(* CODESYS project T620X_HMI_CR1076_SP19p4.project
   Author: AW
   Version: 3.0.0.7
   Description: T620X/Radial
   Title: MAIN_HMI
   Company: MTech
   CompileDateTime: 09:01:42,04-04-2025

Project tree, tasks and I/O mapping:
  Device : ecomatDisplay_64bit, ifm electronic, order no. 
      , version 3.5.16.55
    application Application
      libraries: CmpBitmapPool, * (System); MGSE_CAS_Common, 0.0.0.1 (MGSE); ifm_ecomatDisplay43inch_Cnt, 1.0.0.0 (ifm electronic); MemoryUtils, * (3S - Smart Software Solutions GmbH); SysSocket, * (System); Util, 3.5.19.0 (System); VisuDialogs, * (System); SysTimeRtc, * (System); ifmIOcommon, 2.4.0.0 (ifm electronic); ifmOutGroup, 2.1.3.0 (ifm electronic); ifmDevice_ecomatDisplay43inch, * (ifm electronic); SysProcess Implementation, * (System); CAA Memory, * (CAA Technical Workgroup); SysMem, * (System); StringUtils, 3.5.18.0 (System); MGSE_CAS_Common, 0.0.0.1 (MGSE); SysTarget, * (System); MGSE_CAS_Common, 0.0.0.1 (MGSE); UDP, * (3S - Smart Software Solutions GmbH); MGSE_CAS_Common, 0.0.0.1 (MGSE); CAA Net Base Services, * (CAA Technical Workgroup); SysDir, * (System); SysFile, * (System); MGSE_CAS_Common, 0.0.0.1 (MGSE); CmpIecTask, * (System); SLL Common, 0.0.0.1 (SLL); SLL_IFM_CRXXXX, 0.0.0.1 (SLL); SLL_IFM_Version, 0.0.0.2 (SLL); MGSE_CAS_Common, 0.0.0.1 (MGSE); PIL Master Library, 1.0.0 (Powerhouse IRL Ltd); SLL_IFM_IO, 0.0.1.0 (SLL); VisuDialogs Template, 4.3.0.1 (Examples)
      task MainTask (cyclic, interval 5 ms, priority 3, watchdog T#500MS x 1) calls HMI_KEYPAD, HMI_IO, PLC_PRG_MAIN, Nav, SECURITY_COM
      task AlarmManagerTask (cyclic, interval 50 ms, priority 31) calls Alarms_Task
      task VISU_TASK (cyclic, interval 50 ms, priority 15) calls Viz_Common, VisuElems.Visu_Prg
      task UDP_COMS_TX (cyclic, interval 10 ms, priority 1, watchdog T#500MS x 1) calls UDP_COMS_TX
      task UDP_COMS_RX (cyclic, interval 10 ms, priority 1, watchdog T#500MS x 1) calls UDP_COMS_RX
      App_Common/
        Alarms/
          program Alarms_Monitor [FBD]
          program Alarms_Task [FBD]
        System/
          program PLC_SYSTEM [FBD]: LoggerFilename, HeaderTimeUpdate
          program PLC_Setup_Info [FBD]
          program PLC_GET_SET_IP_ADDRESS [FBD]
          program SECURITY_COM [FBD]
          program PLC_LOGGING [FBD]
          program PLC_COMMON [FBD]: VersionsUpdate
        UDP/
          program UDP_COMS_RX [FBD]
          program UDP_COMS_TX [FBD]
        Vizualisations/
          Manager/
            image pool ImagePool
            image pool ifmImagePool
            text list TL_eKeyMapCodes
          DIAG_IO/
            visualisation Visualization_DIAG_IO_Op_G0
            visualisation Visualization_DIAG_IO_Ip_G1
            visualisation Visualization_DIAG_IO_Ip_G2
            visualisation Visualization_DIAG_IO_Op_G1
            visualisation Visualization_DIAG_IO_Op_G2
            visualisation Visualization_DIAG_IO_Ip_G0
            visualisation Visualization_DIAG_IO_AUX
            CR0403/
              visualisation Output_IFM_PLC_CR0403
              visualisation Visualization_CR0403_Op
              function block CR0403_Output_Display [ST]: Init
              function block OpCom_CR0403 [FBD]: uValue, Init
              data type CR0403_OUTPUTS_STATES
          Viz_Structures/
            data type Viz_Footer_Struct
            data type Viz_Misc_Status_Struct
            data type Viz_Sections
            data type Viz_Options_Struct
          Main/
            visualisation Visualization_Settings_Main
            visualisation Visualization_Alarms_Main
            visualisation Visualization_PLC_Versions
            Layout/
              visualisation Visualization_Footer
              visualisation Visualization_Keypad_PC_SIM
              visualisation Visualization_Template
              visualisation Visualization_Net_Background
              Simulation/
                visualisation Visualization_SIM_IO
                visualisation Visualization_SIM_IO_AUX
              visualisation Visualization_Main_Status_Common
              visualisation Visualization_Main_Status_Radial
              visualisation Visualization_Main_Status_Standard
            visualisation Visualization_Net_Status_Adv
            visualisation Visualization_Net_Status
            visualisation Visualization_Settings_Misc
            visualisation Visualization_PLC_Status
            visualisation Visualization_Settings_RTC
            visualisation Visualization_Settings_IO_Log
            visualisation Visualization_Settings_1
            visualisation Visualization_Main_1
            visualisation Visualization_Engine_1
            visualisation Visualization_Engine_2
            visualisation Visualization_Settings_2
            visualisation Visualization_Settings_4
            visualisation Visualization_Settings_3
            visualisation Visualization_Engine_3
        Nav/
          program Nav [FBD]: CLEAR_RET_STACK, HOME_RETURN, GOTO_PAGE, PUSH_RET_STACK, POP_RET_STACK
          data type TX_TO_MAIN_HMI_STRUCT
          Page Control/
            function block MoveArrow_1 [ST]
            function block MoveArrow_2 [ST]
            program Page_Ctrl [FBD]
            function block RotatingArrow [ST]
            program LED_Ctrl [ST]
            program AutoManSelButtons [FBD]
            function block RectIcon [FBD]
            function block PWM_Op_Status_FB [FBD]
            function block MoveArrow_Angle [ST]
            function block LED_Control_FB [ST]
        Machine/
          program Safety_Common [FBD]
          program SIREN_BEACONS [FBD]
          program APP_WARNINGS_ERRORS [ST]
        GVLS/
          Net UDP RX TX/
            declarations NVL_IO_CHASSIS
            global variables NVL_Outputs_States_Chassis
          global variables GVL_Versions
          global variables GVL_System
          global variables Machine_IO
          Viz/
            global variables GVL_Viz
            global variables NVL_Viz
          data type NV_Sys_Settings_Struct
          global variables GVL_Persistant_Defaults
          global variables GVL_Persistant
          global variables GVL_Machine
          data type T620X_SETTINGS
          global variables GVL_Engine
          global variables GVL_CAN_TX_AUX
          global variables GVL_J1939
          data type T620X_Running_Varaibles
        VIZ/
          program Viz_Common [FBD]
          program Viz_Footer [FBD]
          program Viz_Header [FBD]
      LIBS/
        IO Diagnostics/
          IO Page Templates/
            UDP/
              visualisation PLC_UDP_Info
            PLC_Status/
              visualisation PLC_Status_Info
            PLC_Version_Info/
              visualisation PLC_Version_Info
            CR0709/
              visualisation Visualization_CR0709_Op_G1
              visualisation Visualization_CR0709_Ip_G2
              visualisation Visualization_CR0709_Op_G0
              visualisation Visualization_CR0709_Op_G2
              visualisation Visualization_CR0709_Ip_G0
              visualisation Visualization_CR0709_Ip_G1
          function block CRXXXX_Input_Display [ST]: Init
          data type HMI_PLC_CR721S_IO
          data type HMI_PLC_CR0709_IO
          IO Page Objects/
            visualisation Output_Force
            visualisation Output_IFM_PLC_CRXXXX_TITLE
            visualisation Output_IFM_PLC_CRXXXX
            visualisation Input_IFM_PLC_CRXXXX
            visualisation Input_IFM_PLC_CRXXXX_TITLE
            visualisation Output_Group_IFM_PLC_CRXXXX
          function block CRXXXX_Output_Display [ST]: Init
          function block Diag_Ip_Freq_Pulse_FB [FBD]
          function block CRXXXX_Output_Group_Display [ST]: Init
          data type HMI_PLC_CR0403_IO
        Alarms/
          Functions/
            function Alarm_Log_Test_PRIME [ST]
            function block SLL_AlarmBit [ST]
            function Alarm_Log_Add [ST]
            function Alarm_ID_GetText [ST]
            function Alarm_Log_Clear_ALL [ST]
            function Alarm_Log_File_Write [ST]
            function block Alarm_Logger_Line_FB [ST]
            program Alarm_Table_Main [ST]
            function Alarm_Log_Count_Errors [ST]
            function Alarm_Log_Count_Warnings [ST]
            function Alarm_Log_Clear_ALL_Inactive [ST]
            function Alarm_Log_Count_Active_Hush [ST]
            function Alarm_Log_Update [ST]
            program Alarm_Log_Count_Errors_Hush [FBD]
          Viz/
            visualisation Alarm_Logger_Title
            visualisation Alarm_Logger_Line
            visualisation Alarm_Logger_Table
          Struct/
            data type SLL_LOGGER_ITEM_GROUP
            data type SLL_LOGGER_MAIN_SRUCT
            data type SLL_LOGGER_ITEM_UDP
            data type SLL_LOGGER_ITEM_FLAGS
            data type SLL_LOGGER_ITEM
            data type SENSOR_SCALE
        UDP/
          function block UDP_Info_Viz [ST]
        function print_formated_DINT_func [FBD]
        function block Convert_mm_to_in_ft [ST]
        Logging/
          function block Log_File_Read_Lines [ST]
          global variables GVL_Logging
          function Log_File_Append [ST]
        IO Common/
          function block OpCom [FBD]: Init
          function block IO_LogCom [ST]
          function block IpCom [FBD]: Init
          text list TextList_IFM_Diag_Codes
          function block OpGrpCom [FBD]: Dig, Init
          function block NodeComFB [FBD]
          function IFM_CODE_Text_Get [ST]
        function block SIMPLE_HB_CHECK_ONLINE [FBD]
        function print_BOOL_func [FBD]
        function TextList_GetText_Default [ST]
        function Mimic_IO_GetText [ST]
        HMI/
          data type HMI_TASKS_INFO_STRUCT
          global variables GVL_KeyList_RT
          data type HMI_TASK_INFO_STRUCT
          program Nav_SetupHalo [ST]
          global variables GVL_KeyList
          program RunLinuxCommand [FBD]
          program Nav_Get_Page_Name [FBD]
          global variables GVL_KeyList_FT
          function block Nav_Pages_Group_FB [FBD]
          program LCD_Brighness_Control [FBD]
          program HMI_Task_Info [ST]
          program CR1140_RTC_Edit [FBD]: ZonesDump
          program HMI_KEYPAD [FBD]: ACT_KeyList_FT, ACT_KeyList_RT
          program CloseDlgs [ST]
          program CheckDlgsOpen [ST]
        function print_formated_REAL_func [FBD]
        function block Convert_inches_to_in_ft [ST]
        function block Override_Timed [FBD]
      Symbols
      App_CODE_GEN/
        MAIN_CODE_GEN/
          App_CODE_GEN/
            Alarms/
              program Alarms_Monitor_App [ST]
              global variables GVL_Alarms
              program Alarms_Monitor_IO [ST]
            Diag_IO/
              program HMI_IO [FBD]: Update_Outputs, Init_Input_Links, Init_Output_Links, Update_Inputs
            Machine IO/
              Funcs/
                program Machine_Link_Outputs_Init [ST]
                program Machine_Link_Outputs [ST]
                program Machine_Scale_Inputs [FBD]
                program Machine_Link_Inputs_Init [ST]
                program Machine_Link_Inputs [ST]
              Structs/
                data type T620X_Radial_Outputs
                data type T620X_Radial_Inputs
        TEXT_LIST/
          text list AlarmGroup_IO
          text list AlarmGroup_App
          text list TextList_IO_Diag
      App_PLC/
        program PLC_EngineRun [FBD]
        program PLC_Alarms [FBD]
        function block fbSmoothing [ST]
        program PLC_FanCtrl [FBD]
        program PLC_SIM_MAIN [FBD]
        global variables SIM_APP
        global variables GVL_APP
        Control/
          program PLC_Auto_Sequence [FBD]
          program PLC_ManualSequence [FBD]
          program PLC_JackLegs_SideConv [FBD]
          program PLC_Tracking [FBD]
          program PLC_RadialMode [FBD]
          program PLC_Functions [FBD]
        Set Points/
          function block SP_Count_VAR [FBD]
        CAN Comms/
          Engine Comms/
            function block CounterChecksum [ST]
            function block PLC_DM1_Condition [FBD]
            function block fb_Extract_SPN [FBD]
            function block Pack2bits [ST]
            program PLC_J1939_COMS [FBD]: SCAN
            program PLC_J1939_TX_CUSTOM [FBD]
            program PLC_J1939_RX_DM1 [FBD]
            function HMI_Time_Remain_HHMM_Secs_In [ST]
          program CAN_TX_AUX_IO [FBD]
        program PLC_PRG_MAIN [FBD]
    Communication : Communication, ifm electronic, version 3.5.16.55
      Ethernet : Ethernet, ifm electronic, version 3.5.16.55
        Ethernet_ecomatDisplay4_3 : Ethernet_ecomatDisplay4.3, ifm electronic, version 1.0.0.0
            settings: IPAddress = [192,168,82,245]; SubnetMask = [255,255,255,0]; GatewayAddress = [192,168,82,1]; MACAddress = [16#00,16#02,16#01,16#10,16#3D,16#7D]; NetworkInterfaceName = 'eth0'; NetworkInterfaceName = "eth0"; SaveCommunicationSettings = FALSE
      CAN : CAN, ifm electronic, version 3.5.16.55
        CANbus_ecomatDisplay4_3 : CANbus_ecomatDisplay4.3, ifm electronic, version 1.0.0.0
            settings: NetID = 1
          J1939_Manager : J1939_Manager, 3S - Smart Software Solutions GmbH, version 4.1.0.0
            J1939_ECU : J1939_ECU, 3S - Smart Software Solutions GmbH, version 4.1.0.0
                settings: NAME = 16#0000000000000000; Communication Watchdog Timeout Period = 16#05DC ms; Activated PGs = 23; PG Offline Data.Name = "EEC1"; PG Offline Data.Description = "Electronic Engine Controller 1"; PG Online Data.PGN = 61444; PG Online Data.Length (Bytes) = 8; PG Transmission Settings.Destination Address = 255; PG Transmission Settings.CycleTimeFactor = 1; Signal Offline Data.SPN = 899; Signal Offline Data.Name = "EngTorqueMode"; Signal Offline Data.Description = "State signal which indicates which engine torque mode is currently generating, limiting, or controlling the torque."; Signal Offline Data.Unit = ""; Signal Offline Data.Min = 0; Signal Offline Data.Max = 15; Signal Online Data.BitSize = 4; Signal Online Data.BitPosition = 0; Convert Data.Flags = 3; Convert Data.pSigValue = 0; Convert Data.Scaling = 4607182418800017408; Convert Data.Offset = 0; Signal Offline Data.SPN = 4154; Signal Offline Data.Name = "ActlEngPrcntTrqueHighResolution"; Signal Offline Data.Description = "This parameter displays an additional torque in percent of the reference engine torque."; Signal Offline Data.Unit = "%"; Signal Offline Data.Min = 0; Signal Offline Data.Max = 0.875; Signal Online Data.BitSize = 4; Signal Online Data.BitPosition = 4; Convert Data.Flags = 3; Convert Data.pSigValue = 0; Convert Data.Scaling = 4593671619917905920; Convert Data.Offset = 0; Signal Offline Data.SPN = 512; Signal Offline Data.Name = "DriversDemandEngPercentTorque"; Signal Offline Data.Description = "The requested torque output of the engine by the driver."; Signal Offline Data.Unit = "%"; Signal Offline Data.Min = -125; Signal Offline Data.Max = 125; Signal Online Data.BitSize = 8;
                  Signal Online Data.BitPosition = 8; Convert Data.Flags = 3; Convert Data.pSigValue = 0; Convert Data.Scaling = 4607182418800017408; Convert Data.Offset = 13861868546813853696; Signal Offline Data.SPN = 513; Signal Offline Data.Name = "ActualEngPercentTorque"; Signal Offline Data.Description = "The calculated output torque of the engine."; Signal Offline Data.Unit = "%"; Signal Offline Data.Min = -125; Signal Offline Data.Max = 125; Signal Online Data.BitSize = 8; Signal Online Data.BitPosition = 16; Convert Data.Flags = 3; Convert Data.pSigValue = 0; Convert Data.Scaling = 4607182418800017408; Convert Data.Offset = 13861868546813853696; Signal Offline Data.SPN = 190; Signal Offline Data.Name = "EngSpeed"; Signal Offline Data.Unit = "rpm"; Signal Offline Data.Min = 0; Signal Offline Data.Max = 8031.875; Signal Online Data.BitSize = 16; Signal Online Data.BitPosition = 24; Convert Data.Flags = 3; Convert Data.pSigValue = 0; Convert Data.Scaling = 4593671619917905920; Convert Data.Offset = 0; Signal Offline Data.SPN = 1483; Signal Offline Data.Name = "SrcAddrssOfCtrllngDvcFrEngCntrl"; Signal Offline Data.Description = "The source address of the SAE J1939 device currently controlling the engine."; Signal Offline Data.Unit = ""; Signal Offline Data.Min = 0; Signal Offline Data.Max = 255; Signal Online Data.BitSize = 8; Signal Online Data.BitPosition = 40; Convert Data.Flags = 3; Convert Data.pSigValue = 0; Convert Data.Scaling = 4607182418800017408; Convert Data.Offset = 0;
                  Signal Offline Data.SPN = 1675; Signal Offline Data.Name = "EngStarterMode"; Signal Offline Data.Description = "There are several phases in a starting action and different reasons why a start cannot take place."; Signal Offline Data.Unit = ""; Signal Offline Data.Min = 0; Signal Offline Data.Max = 15; Signal Online Data.BitSize = 4; Signal Online Data.BitPosition = 48; Convert Data.Flags = 3; Convert Data.pSigValue = 0; Convert Data.Scaling = 4607182418800017408; Convert Data.Offset = 0; Signal Offline Data.SPN = 2432; Signal Offline Data.Name = "EngDemandPercentTorque"; Signal Offline Data.Unit = "%"; Signal Offline Data.Min = -125; Signal Offline Data.Max = 125; Signal Online Data.BitSize = 8; Signal Online Data.BitPosition = 56; Convert Data.Flags = 3; Convert Data.pSigValue = 0; Convert Data.Scaling = 4607182418800017408; Convert Data.Offset = 13861868546813853696; PG Offline Data.Name = "EEC2"; PG Offline Data.Description = "Electronic Engine Controller 2"; PG Online Data.PGN = 61443; PG Online Data.Length (Bytes) = 8; PG Transmission Settings.Destination Address = 255; PG Transmission Settings.CycleTimeFactor = 1; Signal Offline Data.SPN = 558; Signal Offline Data.Name = "AccelPedal1LowIdleSwitch"; Signal Offline Data.Description = "Switch signal which indicates the state of the accelerator pedal 1 low idle switch."; Signal Offline Data.Unit = ""; Signal Offline Data.Min = 0; Signal Offline Data.Max = 3; Signal Online Data.BitSize = 2; Signal Online Data.BitPosition = 0; Convert Data.Flags = 3; Convert Data.pSigValue = 0; Convert Data.Scaling = 4607182418800017408;
                  Convert Data.Offset = 0; Signal Offline Data.SPN = 559; Signal Offline Data.Name = "AccelPedalKickdownSwitch"; Signal Offline Data.Description = "Switch signal which indicates whether the accelerator pedal kickdown switch is opened or closed."; Signal Offline Data.Unit = ""; Signal Offline Data.Min = 0; Signal Offline Data.Max = 3; Signal Online Data.BitSize = 2; Signal Online Data.BitPosition = 2; Convert Data.Flags = 3; Convert Data.pSigValue = 0; Convert Data.Scaling = 4607182418800017408; Convert Data.Offset = 0; Signal Offline Data.SPN = 1437; Signal Offline Data.Name = "RoadSpeedLimitStatus"; Signal Offline Data.Description = "Status (active or not active) of the system used to limit maximum vehicle velocity."; Signal Offline Data.Unit = ""; Signal Offline Data.Min = 0; Signal Offline Data.Max = 3; Signal Online Data.BitSize = 2; Signal Online Data.BitPosition = 4; Convert Data.Flags = 3; Convert Data.pSigValue = 0; Convert Data.Scaling = 4607182418800017408; Convert Data.Offset = 0; Signal Offline Data.SPN = 2970; Signal Offline Data.Name = "AccelPedal2LowIdleSwitch"; Signal Offline Data.Description = "Switch signal which indicates the state of the accelerator pedal 2 low idle switch."; Signal Offline Data.Unit = ""; Signal Offline Data.Min = 0; Signal Offline Data.Max = 3; Signal Online Data.BitSize = 2; Signal Online Data.BitPosition = 6; Convert Data.Flags = 3; Convert Data.pSigValue = 0; Convert Data.Scaling = 4607182418800017408; Convert Data.Offset = 0; Signal Offline Data.SPN = 91; Signal Offline Data.Name = "AccelPedalPos1"; Signal Offline Data.Description = "The ratio of actual position of the analog engine speed/torque request input device (such as an accelerator pedal or";
                  Signal Offline Data.Unit = "%"; Signal Offline Data.Min = 0; Signal Offline Data.Max = 100; Signal Online Data.BitSize = 8; Signal Online Data.BitPosition = 8; Convert Data.Flags = 3; Convert Data.pSigValue = 0; Convert Data.Scaling = 4600877379321698714; Convert Data.Offset = 0; Signal Offline Data.SPN = 92; Signal Offline Data.Name = "EngPercentLoadAtCurrentSpeed"; Signal Offline Data.Unit = "%"; Signal Offline Data.Min = 0; Signal Offline Data.Max = 250; Signal Online Data.BitSize = 8; Signal Online Data.BitPosition = 16; Convert Data.Flags = 3; Convert Data.pSigValue = 0; Convert Data.Scaling = 4607182418800017408; Convert Data.Offset = 0; Signal Offline Data.SPN = 974; Signal Offline Data.Name = "RemoteAccelPedalPos"; Signal Offline Data.Unit = "%"; Signal Offline Data.Min = 0; Signal Offline Data.Max = 100; Signal Online Data.BitSize = 8; Signal Online Data.BitPosition = 24; Convert Data.Flags = 3; Convert Data.pSigValue = 0; Convert Data.Scaling = 4600877379321698714; Convert Data.Offset = 0; Signal Offline Data.SPN = 29; Signal Offline Data.Name = "AccelPedalPos2"; Signal Offline Data.Unit = "%"; Signal Offline Data.Min = 0; Signal Offline Data.Max = 100; Signal Online Data.BitSize = 8; Signal Online Data.BitPosition = 32; Convert Data.Flags = 3; Convert Data.pSigValue = 0;
                  Convert Data.Scaling = 4600877379321698714; Convert Data.Offset = 0; Signal Offline Data.SPN = 2979; Signal Offline Data.Name = "VhclAccelerationRateLimitStatus"; Signal Offline Data.Description = "Status (active or not active) of the system used to limit maximum forward vehicle acceleration."; Signal Offline Data.Unit = ""; Signal Offline Data.Min = 0; Signal Offline Data.Max = 3; Signal Online Data.BitSize = 2; Signal Online Data.BitPosition = 40; Convert Data.Flags = 3; Convert Data.pSigValue = 0; Convert Data.Scaling = 4607182418800017408; Convert Data.Offset = 0; Signal Offline Data.SPN = 5021; Signal Offline Data.Name = "MmntryEngMaxPowerEnableFeedback"; Signal Offline Data.Description = "Momentarily requesting Engine Maximum Power Enable - feature support feedback"; Signal Offline Data.Unit = ""; Signal Offline Data.Min = 0; Signal Offline Data.Max = 3; Signal Online Data.BitSize = 2; Signal Online Data.BitPosition = 42; Convert Data.Flags = 3; Convert Data.pSigValue = 0; Convert Data.Scaling = 4607182418800017408; Convert Data.Offset = 0; Signal Offline Data.SPN = 5399; Signal Offline Data.Name = "DPFThermalManagementActive"; Signal Offline Data.Unit = ""; Signal Offline Data.Min = 0; Signal Offline Data.Max = 3; Signal Online Data.BitSize = 2; Signal Online Data.BitPosition = 44; Convert Data.Flags = 3; Convert Data.pSigValue = 0; Convert Data.Scaling = 4607182418800017408; Convert Data.Offset = 0; Signal Offline Data.SPN = 5400; Signal Offline Data.Name = "SCRThermalManagementActive"; Signal Offline Data.Description = "Indicates that the exhaust temperatures have been elevated for regeneration of the SCR aftertreatment system or in";
                  Signal Offline Data.Unit = ""; Signal Offline Data.Min = 0; Signal Offline Data.Max = 3; Signal Online Data.BitSize = 2; Signal Online Data.BitPosition = 46; Convert Data.Flags = 3; Convert Data.pSigValue = 0; Convert Data.Scaling = 4607182418800017408; Convert Data.Offset = 0; Signal Offline Data.SPN = 3357; Signal Offline Data.Name = "ActlMxAvailableEngPercentTorque"; Signal Offline Data.Description = "This is the maximum amount of torque that the engine can immediately deliver as a percentage of the reference engine"; Signal Offline Data.Unit = "%"; Signal Offline Data.Min = 0; Signal Offline Data.Max = 100; Signal Online Data.BitSize = 8; Signal Online Data.BitPosition = 48; Convert Data.Flags = 3; Convert Data.pSigValue = 0; Convert Data.Scaling = 4600877379321698714; Convert Data.Offset = 0; Signal Offline Data.SPN = 5398; Signal Offline Data.Name = "EstPumpingPercentTorque"; Signal Offline Data.Description = "The calculated torque that indicates the estimated amount of torque loss due to the engine air handling system."; Signal Offline Data.Unit = "%"; Signal Offline Data.Min = -125; Signal Offline Data.Max = 125; Signal Online Data.BitSize = 8; Signal Online Data.BitPosition = 56; Convert Data.Flags = 3; Convert Data.pSigValue = 0; Convert Data.Scaling = 4607182418800017408; Convert Data.Offset = 13861868546813853696; PG Offline Data.Name = "EEC3"; PG Offline Data.Description = "Electronic Engine Controller 3"; PG Online Data.PGN = 65247; PG Online Data.Length (Bytes) = 8; PG Transmission Settings.Destination Address = 255; PG Transmission Settings.CycleTimeFactor = 1; Signal Offline Data.SPN = 514;
                  Signal Offline Data.Name = "NominalFrictionPercentTorque"; Signal Offline Data.Unit = "%"; Signal Offline Data.Min = -125; Signal Offline Data.Max = 125; Signal Online Data.BitSize = 8; Signal Online Data.BitPosition = 0; Convert Data.Flags = 3; Convert Data.pSigValue = 0; Convert Data.Scaling = 4607182418800017408; Convert Data.Offset = 13861868546813853696; Signal Offline Data.SPN = 515; Signal Offline Data.Name = "EngsDesiredOperatingSpeed"; Signal Offline Data.Description = "An indication by the engine of the optimal operating speed of the engine for the current existing conditions."; Signal Offline Data.Unit = "rpm"; Signal Offline Data.Min = 0; Signal Offline Data.Max = 8031.875; Signal Online Data.BitSize = 16; Signal Online Data.BitPosition = 8; Convert Data.Flags = 3; Convert Data.pSigValue = 0; Convert Data.Scaling = 4593671619917905920; Convert Data.Offset = 0; Signal Offline Data.SPN = 519; Signal Offline Data.Name = "EngsDsrdOprtngSpdAsymmtryAdjstmn"; Signal Offline Data.Unit = ""; Signal Offline Data.Min = 0; Signal Offline Data.Max = 250; Signal Online Data.BitSize = 8; Signal Online Data.BitPosition = 24; Convert Data.Flags = 3; Convert Data.pSigValue = 0; Convert Data.Scaling = 4607182418800017408; Convert Data.Offset = 0; Signal Offline Data.SPN = 2978; Signal Offline Data.Name = "EstEngPrsticLossesPercentTorque"; Signal Offline Data.Unit = "%"; Signal Offline Data.Min = -125; Signal Offline Data.Max = 125; Signal Online Data.BitSize = 8; Signal Online Data.BitPosition = 32;
                  Convert Data.Flags = 3; Convert Data.pSigValue = 0; Convert Data.Scaling = 4607182418800017408; Convert Data.Offset = 13861868546813853696; Signal Offline Data.SPN = 3236; Signal Offline Data.Name = "Aftrtratment1ExhaustGasMassFlow"; Signal Offline Data.Description = "Measured/calculated exhaust gas mass upstream of the aftertreatment system in exhaust bank 1 and 2."; Signal Offline Data.Unit = "kg/h"; Signal Offline Data.Min = 0; Signal Offline Data.Max = 12851; Signal Online Data.BitSize = 16; Signal Online Data.BitPosition = 40; Convert Data.Flags = 3; Convert Data.pSigValue = 0; Convert Data.Scaling = 4596373779694328218; Convert Data.Offset = 0; Signal Offline Data.SPN = 3237; Signal Offline Data.Name = "Aftertreatment1IntakeDewPoint"; Signal Offline Data.Unit = ""; Signal Offline Data.Min = 0; Signal Offline Data.Max = 3; Signal Online Data.BitSize = 2; Signal Online Data.BitPosition = 56; Convert Data.Flags = 3; Convert Data.pSigValue = 0; Convert Data.Scaling = 4607182418800017408; Convert Data.Offset = 0; Signal Offline Data.SPN = 3238; Signal Offline Data.Name = "Aftertreatment1ExhaustDewPoint"; Signal Offline Data.Unit = ""; Signal Offline Data.Min = 0; Signal Offline Data.Max = 3; Signal Online Data.BitSize = 2; Signal Online Data.BitPosition = 58; Convert Data.Flags = 3; Convert Data.pSigValue = 0; Convert Data.Scaling = 4607182418800017408; Convert Data.Offset = 0; Signal Offline Data.SPN = 3239; Signal Offline Data.Name = "Aftertreatment2IntakeDewPoint";
                  Signal Offline Data.Unit = ""; Signal Offline Data.Min = 0; Signal Offline Data.Max = 3; Signal Online Data.BitSize = 2; Signal Online Data.BitPosition = 60; Convert Data.Flags = 3; Convert Data.pSigValue = 0; Convert Data.Scaling = 4607182418800017408; Convert Data.Offset = 0; Signal Offline Data.SPN = 3240; Signal Offline Data.Name = "Aftertreatment2ExhaustDewPoint"; Signal Offline Data.Unit = ""; Signal Offline Data.Min = 0; Signal Offline Data.Max = 3; Signal Online Data.BitSize = 2; Signal Online Data.BitPosition = 62; Convert Data.Flags = 3; Convert Data.pSigValue = 0; Convert Data.Scaling = 4607182418800017408; Convert Data.Offset = 0; PG Offline Data.Name = "EEC5"; PG Offline Data.Description = "Electronic Engine Controller 5"; PG Online Data.PGN = 64981; PG Online Data.Length (Bytes) = 8; PG Transmission Settings.Destination Address = 255; PG Transmission Settings.CycleTimeFactor = 1; Signal Offline Data.SPN = 2789; Signal Offline Data.Name = "EngTrb1ClcltedTurbineIntakeTemp"; Signal Offline Data.Description = "Calculated value of turbine intake temperature based on engine operating conditions, such as intake manifold"; Signal Offline Data.Unit = "deg C"; Signal Offline Data.Min = -273; Signal Offline Data.Max = 1734.96875; Signal Online Data.BitSize = 16; Signal Online Data.BitPosition = 0; Convert Data.Flags = 3; Convert Data.pSigValue = 0; Convert Data.Scaling = 4584664420663164928; Convert Data.Offset = 13866882319836512256; Signal Offline Data.SPN = 2790; Signal Offline Data.Name = "EngTrb1ClcltedTurbineOutletTemp";
                  Signal Offline Data.Description = "Calculated value of turbocharger compressor outlet air temperature."; Signal Offline Data.Unit = "deg C"; Signal Offline Data.Min = -273; Signal Offline Data.Max = 1734.96875; Signal Online Data.BitSize = 16; Signal Online Data.BitPosition = 16; Convert Data.Flags = 3; Convert Data.pSigValue = 0; Convert Data.Scaling = 4584664420663164928; Convert Data.Offset = 13866882319836512256; Signal Offline Data.SPN = 2791; Signal Offline Data.Name = "EngExhstGsRcrculation1ValveCtrl"; Signal Offline Data.Description = "Desired percentage of maximum Exhaust Gas Recirculation (EGR) valve opening."; Signal Offline Data.Unit = "%"; Signal Offline Data.Min = 0; Signal Offline Data.Max = 160.6375; Signal Online Data.BitSize = 16; Signal Online Data.BitPosition = 32; Convert Data.Flags = 3; Convert Data.pSigValue = 0; Convert Data.Scaling = 4567911030049346683; Convert Data.Offset = 0; Signal Offline Data.SPN = 2792; Signal Offline Data.Name = "EngVrblGmtryTrbArCtrlShtffValve"; Signal Offline Data.Description = "Isolates vehicle brake air from the Variable Geometry Turbocharger (VGT) system when engine is not running."; Signal Offline Data.Unit = ""; Signal Offline Data.Min = 0; Signal Offline Data.Max = 3; Signal Online Data.BitSize = 2; Signal Online Data.BitPosition = 48; Convert Data.Flags = 3; Convert Data.pSigValue = 0; Convert Data.Scaling = 4607182418800017408; Convert Data.Offset = 0; Signal Offline Data.SPN = 5457; Signal Offline Data.Name = "EngVrableGeometryTurbo1CtrlMode"; Signal Offline Data.Description = "Indicates if the variable geometry turbocharger control status is either open loop or closed loop."; Signal Offline Data.Unit = ""; Signal Offline Data.Min = 0; Signal Offline Data.Max = 3;
                  Signal Online Data.BitSize = 2; Signal Online Data.BitPosition = 52; Convert Data.Flags = 3; Convert Data.pSigValue = 0; Convert Data.Scaling = 4607182418800017408; Convert Data.Offset = 0; Signal Offline Data.SPN = 2795; Signal Offline Data.Name = "EngVrblGometryTurbo1ActuatorPos"; Signal Offline Data.Description = "Sensor that measures the position of the variable geometry turbocharger actuator."; Signal Offline Data.Unit = "%"; Signal Offline Data.Min = 0; Signal Offline Data.Max = 100; Signal Online Data.BitSize = 8; Signal Online Data.BitPosition = 56; Convert Data.Flags = 3; Convert Data.pSigValue = 0; Convert Data.Scaling = 4600877379321698714; Convert Data.Offset = 0; PG Offline Data.Name = "ET1"; PG Offline Data.Description = "Engine Temperature 1"; PG Online Data.PGN = 65262; PG Online Data.Length (Bytes) = 8; PG Transmission Settings.Destination Address = 255; PG Transmission Settings.CycleTimeFactor = 1; Signal Offline Data.SPN = 110; Signal Offline Data.Name = "EngCoolantTemp"; Signal Offline Data.Description = "Temperature of liquid found in engine cooling system."; Signal Offline Data.Unit = "deg C"; Signal Offline Data.Min = -40; Signal Offline Data.Max = 210; Signal Online Data.BitSize = 8; Signal Online Data.BitPosition = 0; Convert Data.Flags = 3; Convert Data.pSigValue = 0; Convert Data.Scaling = 4607182418800017408; Convert Data.Offset = 13854198353698488320; Signal Offline Data.SPN = 174; Signal Offline Data.Name = "EngFuelTemp1"; Signal Offline Data.Description = "Temperature of fuel (or gas) passing through the first fuel control system."; Signal Offline Data.Unit = "deg C";
                  Signal Offline Data.Min = -40; Signal Offline Data.Max = 210; Signal Online Data.BitSize = 8; Signal Online Data.BitPosition = 8; Convert Data.Flags = 3; Convert Data.pSigValue = 0; Convert Data.Scaling = 4607182418800017408; Convert Data.Offset = 13854198353698488320; Signal Offline Data.SPN = 175; Signal Offline Data.Name = "EngOilTemp1"; Signal Offline Data.Description = "Temperature of the engine lubricant."; Signal Offline Data.Unit = "deg C"; Signal Offline Data.Min = -273; Signal Offline Data.Max = 1734.96875; Signal Online Data.BitSize = 16; Signal Online Data.BitPosition = 16; Convert Data.Flags = 3; Convert Data.pSigValue = 0; Convert Data.Scaling = 4584664420663164928; Convert Data.Offset = 13866882319836512256; Signal Offline Data.SPN = 176; Signal Offline Data.Name = "EngTurboOilTemp"; Signal Offline Data.Description = "Temperature of the turbocharger lubricant."; Signal Offline Data.Unit = "deg C"; Signal Offline Data.Min = -273; Signal Offline Data.Max = 1734.96875; Signal Online Data.BitSize = 16; Signal Online Data.BitPosition = 32; Convert Data.Flags = 3; Convert Data.pSigValue = 0; Convert Data.Scaling = 4584664420663164928; Convert Data.Offset = 13866882319836512256; Signal Offline Data.SPN = 52; Signal Offline Data.Name = "EngIntercoolerTemp"; Signal Offline Data.Description = "Temperature of liquid found in the intercooler located after the turbocharger."; Signal Offline Data.Unit = "deg C"; Signal Offline Data.Min = -40; Signal Offline Data.Max = 210; Signal Online Data.BitSize = 8; Signal Online Data.BitPosition = 48;
                  Convert Data.Flags = 3; Convert Data.pSigValue = 0; Convert Data.Scaling = 4607182418800017408; Convert Data.Offset = 13854198353698488320; Signal Offline Data.SPN = 1134; Signal Offline Data.Name = "EngIntercoolerThermostatOpening"; Signal Offline Data.Description = "The current position of the thermostat used to regulate the temperature of the engine intercooler."; Signal Offline Data.Unit = "%"; Signal Offline Data.Min = 0; Signal Offline Data.Max = 100; Signal Online Data.BitSize = 8; Signal Online Data.BitPosition = 56; Convert Data.Flags = 3; Convert Data.pSigValue = 0; Convert Data.Scaling = 4600877379321698714; Convert Data.Offset = 0; PG Offline Data.Name = "EFL_P1"; PG Offline Data.Description = "Engine Fluid Level/Pressure 1"; PG Online Data.PGN = 65263; PG Online Data.Length (Bytes) = 8; PG Transmission Settings.Destination Address = 255; PG Transmission Settings.CycleTimeFactor = 1; Signal Offline Data.SPN = 94; Signal Offline Data.Name = "EngFuelDeliveryPress"; Signal Offline Data.Description = "Gage pressure of fuel in system as delivered from supply pump to the injection pump."; Signal Offline Data.Unit = "kPa"; Signal Offline Data.Min = 0; Signal Offline Data.Max = 1000; Signal Online Data.BitSize = 8; Signal Online Data.BitPosition = 0; Convert Data.Flags = 3; Convert Data.pSigValue = 0; Convert Data.Scaling = 4616189618054758400; Convert Data.Offset = 0; Signal Offline Data.SPN = 22; Signal Offline Data.Name = "EngExCrankcaseBlowbyPress"; Signal Offline Data.Description = "Differential crankcase blow-by pressure as measured through a tube with a venturi."; Signal Offline Data.Unit = "kPa"; Signal Offline Data.Min = 0; Signal Offline Data.Max = 12.5;
                  Signal Online Data.BitSize = 8; Signal Online Data.BitPosition = 8; Convert Data.Flags = 3; Convert Data.pSigValue = 0; Convert Data.Scaling = 4587366580439587226; Convert Data.Offset = 0; Signal Offline Data.SPN = 98; Signal Offline Data.Name = "EngOilLevel"; Signal Offline Data.Description = "Ratio of current volume of engine sump oil to maximum required volume."; Signal Offline Data.Unit = "%"; Signal Offline Data.Min = 0; Signal Offline Data.Max = 100; Signal Online Data.BitSize = 8; Signal Online Data.BitPosition = 16; Convert Data.Flags = 3; Convert Data.pSigValue = 0; Convert Data.Scaling = 4600877379321698714; Convert Data.Offset = 0; Signal Offline Data.SPN = 100; Signal Offline Data.Name = "EngOilPress"; Signal Offline Data.Description = "Gage pressure of oil in engine lubrication system as provided by oil pump."; Signal Offline Data.Unit = "kPa"; Signal Offline Data.Min = 0; Signal Offline Data.Max = 1000; Signal Online Data.BitSize = 8; Signal Online Data.BitPosition = 24; Convert Data.Flags = 3; Convert Data.pSigValue = 0; Convert Data.Scaling = 4616189618054758400; Convert Data.Offset = 0; Signal Offline Data.SPN = 101; Signal Offline Data.Name = "EngCrankcasePress"; Signal Offline Data.Description = "Gage pressure inside engine crankcase."; Signal Offline Data.Unit = "kPa"; Signal Offline Data.Min = -250; Signal Offline Data.Max = 251.99; Signal Online Data.BitSize = 16; Signal Online Data.BitPosition = 32; Convert Data.Flags = 3; Convert Data.pSigValue = 0;
                  Convert Data.Scaling = 4575657221408423936; Convert Data.Offset = 13866372146441224192; Signal Offline Data.SPN = 109; Signal Offline Data.Name = "EngCoolantPress"; Signal Offline Data.Description = "Gage pressure of liquid found in engine cooling system."; Signal Offline Data.Unit = "kPa"; Signal Offline Data.Min = 0; Signal Offline Data.Max = 500; Signal Online Data.BitSize = 8; Signal Online Data.BitPosition = 48; Convert Data.Flags = 3; Convert Data.pSigValue = 0; Convert Data.Scaling = 4611686018427387904; Convert Data.Offset = 0; Signal Offline Data.SPN = 111; Signal Offline Data.Name = "EngCoolantLevel"; Signal Offline Data.Description = "Ratio of volume of liquid found in engine cooling system to total cooling system volume."; Signal Offline Data.Unit = "%"; Signal Offline Data.Min = 0; Signal Offline Data.Max = 100; Signal Online Data.BitSize = 8; Signal Online Data.BitPosition = 56; Convert Data.Flags = 3; Convert Data.pSigValue = 0; Convert Data.Scaling = 4600877379321698714; Convert Data.Offset = 0; PG Offline Data.Name = "EFL_P2"; PG Offline Data.Description = "Engine Fluid Level/Pressure 2"; PG Online Data.PGN = 65243; PG Online Data.Length (Bytes) = 8; PG Transmission Settings.Destination Address = 255; PG Transmission Settings.CycleTimeFactor = 1; Signal Offline Data.SPN = 164; Signal Offline Data.Name = "EngInjectionCtrlPress"; Signal Offline Data.Description = "The gage pressure of the engine oil in the hydraulic accumulator that powers an intensifier used for fuel injection."; Signal Offline Data.Unit = "MPa"; Signal Offline Data.Min = 0; Signal Offline Data.Max = 251; Signal Online Data.BitSize = 16; Signal Online Data.BitPosition = 0;
                  Convert Data.Flags = 3; Convert Data.pSigValue = 0; Convert Data.Scaling = 4571153621781053440; Convert Data.Offset = 0; Signal Offline Data.SPN = 157; Signal Offline Data.Name = "EngInjectorMeteringRail1Press"; Signal Offline Data.Unit = "MPa"; Signal Offline Data.Min = 0; Signal Offline Data.Max = 251; Signal Online Data.BitSize = 16; Signal Online Data.BitPosition = 16; Convert Data.Flags = 3; Convert Data.pSigValue = 0; Convert Data.Scaling = 4571153621781053440; Convert Data.Offset = 0; Signal Offline Data.SPN = 156; Signal Offline Data.Name = "EngInjectorTimingRail1Press"; Signal Offline Data.Description = "The gage pressure of fuel in the timing rail delivered from the supply pump to the injector timing intake."; Signal Offline Data.Unit = "MPa"; Signal Offline Data.Min = 0; Signal Offline Data.Max = 251; Signal Online Data.BitSize = 16; Signal Online Data.BitPosition = 32; Convert Data.Flags = 3; Convert Data.pSigValue = 0; Convert Data.Scaling = 4571153621781053440; Convert Data.Offset = 0; Signal Offline Data.SPN = 1349; Signal Offline Data.Name = "EngInjectorMeteringRail2Press"; Signal Offline Data.Description = "The gage pressure of fuel in the metering rail #2 as delivered from the supply pump to the injector metering intake."; Signal Offline Data.Unit = "MPa"; Signal Offline Data.Min = 0; Signal Offline Data.Max = 251; Signal Online Data.BitSize = 16; Signal Online Data.BitPosition = 48; Convert Data.Flags = 3; Convert Data.pSigValue = 0; Convert Data.Scaling = 4571153621781053440; Convert Data.Offset = 0; PG Offline Data.Name = "LFC";
                  PG Offline Data.Description = "Fuel Consumption (Liquid)"; PG Online Data.PGN = 65257; PG Online Data.Length (Bytes) = 8; PG Transmission Settings.Destination Address = 255; PG Transmission Settings.CycleTimeFactor = 1; Signal Offline Data.SPN = 182; Signal Offline Data.Name = "EngTripFuel"; Signal Offline Data.Description = "Fuel consumed during all or part of a journey."; Signal Offline Data.Unit = "L"; Signal Offline Data.Min = 0; Signal Offline Data.Max = 2105540607.5; Signal Online Data.BitSize = 32; Signal Online Data.BitPosition = 0; Convert Data.Flags = 3; Convert Data.pSigValue = 0; Convert Data.Scaling = 4602678819172646912; Convert Data.Offset = 0; Signal Offline Data.SPN = 250; Signal Offline Data.Name = "EngTotalFuelUsed"; Signal Offline Data.Description = "Accumulated amount of fuel used during vehicle operation."; Signal Offline Data.Unit = "L"; Signal Offline Data.Min = 0; Signal Offline Data.Max = 2105540607.5; Signal Online Data.BitSize = 32; Signal Online Data.BitPosition = 32; Convert Data.Flags = 3; Convert Data.pSigValue = 0; Convert Data.Scaling = 4602678819172646912; Convert Data.Offset = 0; PG Offline Data.Name = "AMB"; PG Offline Data.Description = "Ambient Conditions"; PG Online Data.PGN = 65269; PG Online Data.Length (Bytes) = 8; PG Transmission Settings.Destination Address = 255; PG Transmission Settings.CycleTimeFactor = 1; Signal Offline Data.SPN = 108; Signal Offline Data.Name = "BarometricPress"; Signal Offline Data.Description = "Absolute air pressure of the atmosphere."; Signal Offline Data.Unit = "kPa"; Signal Offline Data.Min = 0;
                  Signal Offline Data.Max = 125; Signal Online Data.BitSize = 8; Signal Online Data.BitPosition = 0; Convert Data.Flags = 3; Convert Data.pSigValue = 0; Convert Data.Scaling = 4602678819172646912; Convert Data.Offset = 0; Signal Offline Data.SPN = 170; Signal Offline Data.Name = "CabInteriorTemp"; Signal Offline Data.Description = "Temperature of air inside the part of the vehicle that encloses the driver and vehicle operating controls."; Signal Offline Data.Unit = "deg C"; Signal Offline Data.Min = -273; Signal Offline Data.Max = 1734.96875; Signal Online Data.BitSize = 16; Signal Online Data.BitPosition = 8; Convert Data.Flags = 3; Convert Data.pSigValue = 0; Convert Data.Scaling = 4584664420663164928; Convert Data.Offset = 13866882319836512256; Signal Offline Data.SPN = 171; Signal Offline Data.Name = "AmbientAirTemp"; Signal Offline Data.Description = "Temperature of air surrounding vehicle."; Signal Offline Data.Unit = "deg C"; Signal Offline Data.Min = -273; Signal Offline Data.Max = 1734.96875; Signal Online Data.BitSize = 16; Signal Online Data.BitPosition = 24; Convert Data.Flags = 3; Convert Data.pSigValue = 0; Convert Data.Scaling = 4584664420663164928; Convert Data.Offset = 13866882319836512256; Signal Offline Data.SPN = 172; Signal Offline Data.Name = "EngAirIntakeTemp"; Signal Offline Data.Description = "Temperature of air entering vehicle air induction system."; Signal Offline Data.Unit = "deg C"; Signal Offline Data.Min = -40; Signal Offline Data.Max = 210; Signal Online Data.BitSize = 8; Signal Online Data.BitPosition = 40; Convert Data.Flags = 3;
                  Convert Data.pSigValue = 0; Convert Data.Scaling = 4607182418800017408; Convert Data.Offset = 13854198353698488320; Signal Offline Data.SPN = 79; Signal Offline Data.Name = "RoadSurfaceTemp"; Signal Offline Data.Description = "Indicated temperature of road surface over which vehicle is operating."; Signal Offline Data.Unit = "deg C"; Signal Offline Data.Min = -273; Signal Offline Data.Max = 1734.96875; Signal Online Data.BitSize = 16; Signal Online Data.BitPosition = 48; Convert Data.Flags = 3; Convert Data.pSigValue = 0; Convert Data.Scaling = 4584664420663164928; Convert Data.Offset = 13866882319836512256; PG Offline Data.Name = "IC1"; PG Offline Data.Description = "Intake/Exhaust Conditions 1"; PG Online Data.PGN = 65270; PG Online Data.Length (Bytes) = 8; PG Transmission Settings.Destination Address = 255; PG Transmission Settings.CycleTimeFactor = 1; Signal Offline Data.SPN = 81; Signal Offline Data.Name = "EngDslPrtclateFilterIntakePress"; Signal Offline Data.Description = "Exhaust back pressure as a result of particle accumulation on filter media placed in the exhaust stream."; Signal Offline Data.Unit = "kPa"; Signal Offline Data.Min = 0; Signal Offline Data.Max = 125; Signal Online Data.BitSize = 8; Signal Online Data.BitPosition = 0; Convert Data.Flags = 3; Convert Data.pSigValue = 0; Convert Data.Scaling = 4602678819172646912; Convert Data.Offset = 0; Signal Offline Data.SPN = 102; Signal Offline Data.Name = "EngIntakeManifold1Press"; Signal Offline Data.Description = "The gage pressure measurement of the air intake manifold."; Signal Offline Data.Unit = "kPa"; Signal Offline Data.Min = 0; Signal Offline Data.Max = 500; Signal Online Data.BitSize = 8;
                  Signal Online Data.BitPosition = 8; Convert Data.Flags = 3; Convert Data.pSigValue = 0; Convert Data.Scaling = 4611686018427387904; Convert Data.Offset = 0; Signal Offline Data.SPN = 105; Signal Offline Data.Name = "EngIntakeManifold1Temp"; Signal Offline Data.Description = "Temperature of pre-combustion air found in intake manifold of engine air supply system."; Signal Offline Data.Unit = "deg C"; Signal Offline Data.Min = -40; Signal Offline Data.Max = 210; Signal Online Data.BitSize = 8; Signal Online Data.BitPosition = 16; Convert Data.Flags = 3; Convert Data.pSigValue = 0; Convert Data.Scaling = 4607182418800017408; Convert Data.Offset = 13854198353698488320; Signal Offline Data.SPN = 106; Signal Offline Data.Name = "EngAirIntakePress"; Signal Offline Data.Description = "Absolute air pressure at input port to intake manifold or air box."; Signal Offline Data.Unit = "kPa"; Signal Offline Data.Min = 0; Signal Offline Data.Max = 500; Signal Online Data.BitSize = 8; Signal Online Data.BitPosition = 24; Convert Data.Flags = 3; Convert Data.pSigValue = 0; Convert Data.Scaling = 4611686018427387904; Convert Data.Offset = 0; Signal Offline Data.SPN = 107; Signal Offline Data.Name = "EngAirFilter1DiffPress"; Signal Offline Data.Unit = "kPa"; Signal Offline Data.Min = 0; Signal Offline Data.Max = 12.5; Signal Online Data.BitSize = 8; Signal Online Data.BitPosition = 32; Convert Data.Flags = 3; Convert Data.pSigValue = 0; Convert Data.Scaling = 4587366580439587226; Convert Data.Offset = 0;
                  Signal Offline Data.SPN = 173; Signal Offline Data.Name = "EngExhaustGasTemp"; Signal Offline Data.Description = "Temperature of combustion byproducts leaving the engine."; Signal Offline Data.Unit = "deg C"; Signal Offline Data.Min = -273; Signal Offline Data.Max = 1734.96875; Signal Online Data.BitSize = 16; Signal Online Data.BitPosition = 40; Convert Data.Flags = 3; Convert Data.pSigValue = 0; Convert Data.Scaling = 4584664420663164928; Convert Data.Offset = 13866882319836512256; Signal Offline Data.SPN = 112; Signal Offline Data.Name = "EngCoolantFilterDiffPress"; Signal Offline Data.Unit = "kPa"; Signal Offline Data.Min = 0; Signal Offline Data.Max = 125; Signal Online Data.BitSize = 8; Signal Online Data.BitPosition = 56; Convert Data.Flags = 3; Convert Data.pSigValue = 0; Convert Data.Scaling = 4602678819172646912; Convert Data.Offset = 0; PG Offline Data.Name = "VEP1"; PG Offline Data.Description = "Vehicle Electrical Power 1"; PG Online Data.PGN = 65271; PG Online Data.Length (Bytes) = 8; PG Transmission Settings.Destination Address = 255; PG Transmission Settings.CycleTimeFactor = 1; Signal Offline Data.SPN = 114; Signal Offline Data.Name = "NetBatteryCurrent"; Signal Offline Data.Description = "Net flow of electrical current into/out of the battery or batteries."; Signal Offline Data.Unit = "A"; Signal Offline Data.Min = -125; Signal Offline Data.Max = 125; Signal Online Data.BitSize = 8; Signal Online Data.BitPosition = 0; Convert Data.Flags = 3; Convert Data.pSigValue = 0; Convert Data.Scaling = 4607182418800017408;
                  Convert Data.Offset = 13861868546813853696; Signal Offline Data.SPN = 115; Signal Offline Data.Name = "AltCurrent"; Signal Offline Data.Description = "Measure of electrical current flow from the alternator."; Signal Offline Data.Unit = "A"; Signal Offline Data.Min = 0; Signal Offline Data.Max = 250; Signal Online Data.BitSize = 8; Signal Online Data.BitPosition = 8; Convert Data.Flags = 3; Convert Data.pSigValue = 0; Convert Data.Scaling = 4607182418800017408; Convert Data.Offset = 0; Signal Offline Data.SPN = 167; Signal Offline Data.Name = "ChargingSystemPotential"; Signal Offline Data.Description = "Electrical potential measured at the charging system output."; Signal Offline Data.Unit = "V"; Signal Offline Data.Min = 0; Signal Offline Data.Max = 3212.75; Signal Online Data.BitSize = 16; Signal Online Data.BitPosition = 16; Convert Data.Flags = 3; Convert Data.pSigValue = 0; Convert Data.Scaling = 4587366580439587226; Convert Data.Offset = 0; Signal Offline Data.SPN = 168; Signal Offline Data.Name = "BatteryPotential_PowerInput1"; Signal Offline Data.Description = "This parameter measures the first source of battery potential as measured at the input of the ECM/actuator etc."; Signal Offline Data.Unit = "V"; Signal Offline Data.Min = 0; Signal Offline Data.Max = 3212.75; Signal Online Data.BitSize = 16; Signal Online Data.BitPosition = 32; Convert Data.Flags = 3; Convert Data.pSigValue = 0; Convert Data.Scaling = 4587366580439587226; Convert Data.Offset = 0; Signal Offline Data.SPN = 158; Signal Offline Data.Name = "KeyswitchBatteryPotential"; Signal Offline Data.Unit = "V";
                  Signal Offline Data.Min = 0; Signal Offline Data.Max = 3212.75; Signal Online Data.BitSize = 16; Signal Online Data.BitPosition = 48; Convert Data.Flags = 3; Convert Data.pSigValue = 0; Convert Data.Scaling = 4587366580439587226; Convert Data.Offset = 0; PG Offline Data.Name = "EFS"; PG Offline Data.Description = "Engine Fuel/lube systems"; PG Online Data.PGN = 65130; PG Online Data.Length (Bytes) = 7; PG Transmission Settings.Destination Address = 255; PG Transmission Settings.CycleTimeFactor = 1; Signal Offline Data.SPN = 1380; Signal Offline Data.Name = "EngOilLevelRemoteReservoir"; Signal Offline Data.Description = "Ratio of current volume of engine oil in a remote reservoir to the maximum required volume."; Signal Offline Data.Unit = "%"; Signal Offline Data.Min = 0; Signal Offline Data.Max = 100; Signal Online Data.BitSize = 8; Signal Online Data.BitPosition = 0; Convert Data.Flags = 3; Convert Data.pSigValue = 0; Convert Data.Scaling = 4600877379321698714; Convert Data.Offset = 0; Signal Offline Data.SPN = 1381; Signal Offline Data.Name = "EngFuelSupplyPumpIntakePress"; Signal Offline Data.Description = "Absolute pressure of fuel at the fuel supply pump intake."; Signal Offline Data.Unit = "kPa"; Signal Offline Data.Min = 0; Signal Offline Data.Max = 500; Signal Online Data.BitSize = 8; Signal Online Data.BitPosition = 8; Convert Data.Flags = 3; Convert Data.pSigValue = 0; Convert Data.Scaling = 4611686018427387904; Convert Data.Offset = 0; Signal Offline Data.SPN = 1382; Signal Offline Data.Name = "EngFuelFilterDiffPress";
                  Signal Offline Data.Description = "Differential pressure measured across the fuel filter located between the fuel tank and the supply pump."; Signal Offline Data.Unit = "kPa"; Signal Offline Data.Min = 0; Signal Offline Data.Max = 500; Signal Online Data.BitSize = 8; Signal Online Data.BitPosition = 16; Convert Data.Flags = 3; Convert Data.pSigValue = 0; Convert Data.Scaling = 4611686018427387904; Convert Data.Offset = 0; Signal Offline Data.SPN = 3548; Signal Offline Data.Name = "EngWasteOilReservoirLevel"; Signal Offline Data.Description = "Level of crankcase blowby emulsion collected by a container."; Signal Offline Data.Unit = "%"; Signal Offline Data.Min = 0; Signal Offline Data.Max = 100; Signal Online Data.BitSize = 8; Signal Online Data.BitPosition = 24; Convert Data.Flags = 3; Convert Data.pSigValue = 0; Convert Data.Scaling = 4600877379321698714; Convert Data.Offset = 0; Signal Offline Data.SPN = 3549; Signal Offline Data.Name = "EngOilFilterOutletPress"; Signal Offline Data.Description = "Oil pressure (gauge) measured just downstream of oil filter."; Signal Offline Data.Unit = "kPa"; Signal Offline Data.Min = 0; Signal Offline Data.Max = 1000; Signal Online Data.BitSize = 8; Signal Online Data.BitPosition = 32; Convert Data.Flags = 3; Convert Data.pSigValue = 0; Convert Data.Scaling = 4616189618054758400; Convert Data.Offset = 0; Signal Offline Data.SPN = 3550; Signal Offline Data.Name = "EngOilPrimingPumpSwitch"; Signal Offline Data.Description = "Switch input for activating the engine oil priming pump."; Signal Offline Data.Unit = ""; Signal Offline Data.Min = 0; Signal Offline Data.Max = 3;
                  Signal Online Data.BitSize = 2; Signal Online Data.BitPosition = 40; Convert Data.Flags = 3; Convert Data.pSigValue = 0; Convert Data.Scaling = 4607182418800017408; Convert Data.Offset = 0; Signal Offline Data.SPN = 3551; Signal Offline Data.Name = "EngOilPrimingState"; Signal Offline Data.Description = "Determination of whether or not the engine is (or has recently been) sufficiently lubricated for starting purposes."; Signal Offline Data.Unit = ""; Signal Offline Data.Min = 0; Signal Offline Data.Max = 3; Signal Online Data.BitSize = 2; Signal Online Data.BitPosition = 42; Convert Data.Flags = 3; Convert Data.pSigValue = 0; Convert Data.Scaling = 4607182418800017408; Convert Data.Offset = 0; Signal Offline Data.SPN = 3552; Signal Offline Data.Name = "EngOilPreHeatedState"; Signal Offline Data.Description = "Indicates whether the engine oil pre-heated sufficiently for starting purposes."; Signal Offline Data.Unit = ""; Signal Offline Data.Min = 0; Signal Offline Data.Max = 3; Signal Online Data.BitSize = 2; Signal Online Data.BitPosition = 44; Convert Data.Flags = 3; Convert Data.pSigValue = 0; Convert Data.Scaling = 4607182418800017408; Convert Data.Offset = 0; Signal Offline Data.SPN = 3553; Signal Offline Data.Name = "EngCoolantPreheatedState"; Signal Offline Data.Description = "Indicates whether the engine coolant is pre-heated sufficiently for starting purposes."; Signal Offline Data.Unit = ""; Signal Offline Data.Min = 0; Signal Offline Data.Max = 3; Signal Online Data.BitSize = 2; Signal Online Data.BitPosition = 46; Convert Data.Flags = 3; Convert Data.pSigValue = 0;
                  Convert Data.Scaling = 4607182418800017408; Convert Data.Offset = 0; Signal Offline Data.SPN = 3554; Signal Offline Data.Name = "EngVentilationStatus"; Signal Offline Data.Description = "Engine ventilation control states."; Signal Offline Data.Unit = ""; Signal Offline Data.Min = 0; Signal Offline Data.Max = 7; Signal Online Data.BitSize = 3; Signal Online Data.BitPosition = 48; Convert Data.Flags = 3; Convert Data.pSigValue = 0; Convert Data.Scaling = 4607182418800017408; Convert Data.Offset = 0; Signal Offline Data.SPN = 4083; Signal Offline Data.Name = "FuelPumpPrimerStatus"; Signal Offline Data.Description = "Parameter used to transmit the actual status of the fuel priming system."; Signal Offline Data.Unit = ""; Signal Offline Data.Min = 0; Signal Offline Data.Max = 3; Signal Online Data.BitSize = 2; Signal Online Data.BitPosition = 51; Convert Data.Flags = 3; Convert Data.pSigValue = 0; Convert Data.Scaling = 4607182418800017408; Convert Data.Offset = 0; PG Offline Data.Name = "DPFC1"; PG Offline Data.Description = "Diesel Particulate Filter Control 1"; PG Online Data.PGN = 64892; PG Online Data.Length (Bytes) = 8; PG Transmission Settings.Destination Address = 255; PG Transmission Settings.CycleTimeFactor = 1; Signal Offline Data.SPN = 3697; Signal Offline Data.Name = "DieselParticulateFilterLampCmd"; Signal Offline Data.Description = "Command to control the diesel particulate filter lamp."; Signal Offline Data.Unit = ""; Signal Offline Data.Min = 0; Signal Offline Data.Max = 7; Signal Online Data.BitSize = 3; Signal Online Data.BitPosition = 0;
                  Convert Data.Flags = 3; Convert Data.pSigValue = 0; Convert Data.Scaling = 4607182418800017408; Convert Data.Offset = 0; Signal Offline Data.SPN = 3699; Signal Offline Data.Name = "DslPrtcltFltrPssvRgnrtionStatus"; Signal Offline Data.Description = "Indicates the state of diesel particulate filter passive regeneration."; Signal Offline Data.Unit = ""; Signal Offline Data.Min = 0; Signal Offline Data.Max = 3; Signal Online Data.BitSize = 2; Signal Online Data.BitPosition = 8; Convert Data.Flags = 3; Convert Data.pSigValue = 0; Convert Data.Scaling = 4607182418800017408; Convert Data.Offset = 0; Signal Offline Data.SPN = 3700; Signal Offline Data.Name = "DslPrtcltFltrActvRgnrtionStatus"; Signal Offline Data.Description = "Indicates the state of diesel particulate filter active regeneration."; Signal Offline Data.Unit = ""; Signal Offline Data.Min = 0; Signal Offline Data.Max = 3; Signal Online Data.BitSize = 2; Signal Online Data.BitPosition = 10; Convert Data.Flags = 3; Convert Data.pSigValue = 0; Convert Data.Scaling = 4607182418800017408; Convert Data.Offset = 0; Signal Offline Data.SPN = 3701; Signal Offline Data.Name = "DieselParticulateFilterStatus"; Signal Offline Data.Description = "Indicates the state of the diesel particulate filter regeneration need and urgency."; Signal Offline Data.Unit = ""; Signal Offline Data.Min = 0; Signal Offline Data.Max = 7; Signal Online Data.BitSize = 3; Signal Online Data.BitPosition = 12; Convert Data.Flags = 3; Convert Data.pSigValue = 0; Convert Data.Scaling = 4607182418800017408; Convert Data.Offset = 0;
                  Signal Offline Data.SPN = 3702; Signal Offline Data.Name = "DslPrtcltFltrActvRgnrtnInhbtdStt"; Signal Offline Data.Description = "Indicates the state of diesel particulate filter active regeneration inhibition."; Signal Offline Data.Unit = ""; Signal Offline Data.Min = 0; Signal Offline Data.Max = 3; Signal Online Data.BitSize = 2; Signal Online Data.BitPosition = 16; Convert Data.Flags = 3; Convert Data.pSigValue = 0; Convert Data.Scaling = 4607182418800017408; Convert Data.Offset = 0; Signal Offline Data.SPN = 3703; Signal Offline Data.Name = "DslPrtcltFltrActvRgnrtnInhbtdDTI"; Signal Offline Data.Unit = ""; Signal Offline Data.Min = 0; Signal Offline Data.Max = 3; Signal Online Data.BitSize = 2; Signal Online Data.BitPosition = 18; Convert Data.Flags = 3; Convert Data.pSigValue = 0; Convert Data.Scaling = 4607182418800017408; Convert Data.Offset = 0; Signal Offline Data.SPN = 3704; Signal Offline Data.Name = "DslPrtcltFltrActvRgnrtnInhbtdDTC"; Signal Offline Data.Description = "Indicates the state of diesel particulate filter active regeneration inhibition due to the clutch being disengaged."; Signal Offline Data.Unit = ""; Signal Offline Data.Min = 0; Signal Offline Data.Max = 3; Signal Online Data.BitSize = 2; Signal Online Data.BitPosition = 20; Convert Data.Flags = 3; Convert Data.pSigValue = 0; Convert Data.Scaling = 4607182418800017408; Convert Data.Offset = 0; Signal Offline Data.SPN = 3705; Signal Offline Data.Name = "DslPrtcltFltrActvRgnrtnInhb_0004"; Signal Offline Data.Unit = ""; Signal Offline Data.Min = 0; Signal Offline Data.Max = 3;
                  Signal Online Data.BitSize = 2; Signal Online Data.BitPosition = 22; Convert Data.Flags = 3; Convert Data.pSigValue = 0; Convert Data.Scaling = 4607182418800017408; Convert Data.Offset = 0; Signal Offline Data.SPN = 3706; Signal Offline Data.Name = "DslPrtcltFltrActvRgnrtnInhb_0003"; Signal Offline Data.Description = "Indicates the state of diesel particulate filter active regeneration inhibition due to the PTO being active."; Signal Offline Data.Unit = ""; Signal Offline Data.Min = 0; Signal Offline Data.Max = 3; Signal Online Data.BitSize = 2; Signal Online Data.BitPosition = 24; Convert Data.Flags = 3; Convert Data.pSigValue = 0; Convert Data.Scaling = 4607182418800017408; Convert Data.Offset = 0; Signal Offline Data.SPN = 3707; Signal Offline Data.Name = "DslPrtcltFltrActvRgnrtnInhbtdDTA"; Signal Offline Data.Unit = ""; Signal Offline Data.Min = 0; Signal Offline Data.Max = 3; Signal Online Data.BitSize = 2; Signal Online Data.BitPosition = 26; Convert Data.Flags = 3; Convert Data.pSigValue = 0; Convert Data.Scaling = 4607182418800017408; Convert Data.Offset = 0; Signal Offline Data.SPN = 3708; Signal Offline Data.Name = "DslPrtcltFltrActvRgnrtnInhbtdDTO"; Signal Offline Data.Unit = ""; Signal Offline Data.Min = 0; Signal Offline Data.Max = 3; Signal Online Data.BitSize = 2; Signal Online Data.BitPosition = 28; Convert Data.Flags = 3; Convert Data.pSigValue = 0; Convert Data.Scaling = 4607182418800017408; Convert Data.Offset = 0;
                  Signal Offline Data.SPN = 3709; Signal Offline Data.Name = "DslPrtcltFltrActvRgnrtnInhb_0002"; Signal Offline Data.Description = "Speed"; Signal Offline Data.Unit = ""; Signal Offline Data.Min = 0; Signal Offline Data.Max = 3; Signal Online Data.BitSize = 2; Signal Online Data.BitPosition = 30; Convert Data.Flags = 3; Convert Data.pSigValue = 0; Convert Data.Scaling = 4607182418800017408; Convert Data.Offset = 0; Signal Offline Data.SPN = 3710; Signal Offline Data.Name = "DslPrtcltFltrActvRgnrtnInhb_0001"; Signal Offline Data.Unit = ""; Signal Offline Data.Min = 0; Signal Offline Data.Max = 3; Signal Online Data.BitSize = 2; Signal Online Data.BitPosition = 32; Convert Data.Flags = 3; Convert Data.pSigValue = 0; Convert Data.Scaling = 4607182418800017408; Convert Data.Offset = 0; Signal Offline Data.SPN = 3711; Signal Offline Data.Name = "DslPrtcltFltrActvRgnrtnInhbtdDTL"; Signal Offline Data.Unit = ""; Signal Offline Data.Min = 0; Signal Offline Data.Max = 3; Signal Online Data.BitSize = 2; Signal Online Data.BitPosition = 34; Convert Data.Flags = 3; Convert Data.pSigValue = 0; Convert Data.Scaling = 4607182418800017408; Convert Data.Offset = 0; Signal Offline Data.SPN = 3712; Signal Offline Data.Name = "DslPrtcltFltrActvRgnrtnInhb_0000"; Signal Offline Data.Description = "Indicates the state of diesel particulate filter active regeneration inhibition due to a system fault being active."; Signal Offline Data.Unit = ""; Signal Offline Data.Min = 0; Signal Offline Data.Max = 3;
                  Signal Online Data.BitSize = 2; Signal Online Data.BitPosition = 36; Convert Data.Flags = 3; Convert Data.pSigValue = 0; Convert Data.Scaling = 4607182418800017408; Convert Data.Offset = 0; Signal Offline Data.SPN = 3713; Signal Offline Data.Name = "DslPrtcltFltrActvRgnrtnInhbtdDTS"; Signal Offline Data.Description = "Indicates the state of diesel particulate filter active regeneration inhibition due to a system timeout."; Signal Offline Data.Unit = ""; Signal Offline Data.Min = 0; Signal Offline Data.Max = 3; Signal Online Data.BitSize = 2; Signal Online Data.BitPosition = 38; Convert Data.Flags = 3; Convert Data.pSigValue = 0; Convert Data.Scaling = 4607182418800017408; Convert Data.Offset = 0; Signal Offline Data.SPN = 3714; Signal Offline Data.Name = "DslPrtcltFltrActvRgnrtnInhbtdDTT"; Signal Offline Data.Description = "Indicates the state of diesel particulate filter active regeneration inhibition due to a temporary system lockout."; Signal Offline Data.Unit = ""; Signal Offline Data.Min = 0; Signal Offline Data.Max = 3; Signal Online Data.BitSize = 2; Signal Online Data.BitPosition = 40; Convert Data.Flags = 3; Convert Data.pSigValue = 0; Convert Data.Scaling = 4607182418800017408; Convert Data.Offset = 0; Signal Offline Data.SPN = 3715; Signal Offline Data.Name = "DslPrtcltFltrActvRgnrtnInhbtdDTP"; Signal Offline Data.Description = "Indicates the state of diesel particulate filter active regeneration inhibition due to a permanent system lockout."; Signal Offline Data.Unit = ""; Signal Offline Data.Min = 0; Signal Offline Data.Max = 3; Signal Online Data.BitSize = 2; Signal Online Data.BitPosition = 42; Convert Data.Flags = 3; Convert Data.pSigValue = 0;
                  Convert Data.Scaling = 4607182418800017408; Convert Data.Offset = 0; Signal Offline Data.SPN = 3716; Signal Offline Data.Name = "DslPrtcltFltrActvRgnrtnInhbtdDTE"; Signal Offline Data.Unit = ""; Signal Offline Data.Min = 0; Signal Offline Data.Max = 3; Signal Online Data.BitSize = 2; Signal Online Data.BitPosition = 44; Convert Data.Flags = 3; Convert Data.pSigValue = 0; Convert Data.Scaling = 4607182418800017408; Convert Data.Offset = 0; Signal Offline Data.SPN = 3717; Signal Offline Data.Name = "DslPrtcltFltrActvRgnrtnInhbtdDTV"; Signal Offline Data.Description = "Speed"; Signal Offline Data.Unit = ""; Signal Offline Data.Min = 0; Signal Offline Data.Max = 3; Signal Online Data.BitSize = 2; Signal Online Data.BitPosition = 46; Convert Data.Flags = 3; Convert Data.pSigValue = 0; Convert Data.Scaling = 4607182418800017408; Convert Data.Offset = 0; Signal Offline Data.SPN = 3718; Signal Offline Data.Name = "DslPrtcltFltrAtmtcActvRgnrtnIntt"; Signal Offline Data.Description = "Indicates the configuration of diesel particulate filter active regeneration automatic initiation."; Signal Offline Data.Unit = ""; Signal Offline Data.Min = 0; Signal Offline Data.Max = 3; Signal Online Data.BitSize = 2; Signal Online Data.BitPosition = 48; Convert Data.Flags = 3; Convert Data.pSigValue = 0; Convert Data.Scaling = 4607182418800017408; Convert Data.Offset = 0; Signal Offline Data.SPN = 3698; Signal Offline Data.Name = "ExhaustSystemHighTempLampCmd"; Signal Offline Data.Description = "Command to control the exhaust system high temperature lamp.";
                  Signal Offline Data.Unit = ""; Signal Offline Data.Min = 0; Signal Offline Data.Max = 7; Signal Online Data.BitSize = 3; Signal Online Data.BitPosition = 50; Convert Data.Flags = 3; Convert Data.pSigValue = 0; Convert Data.Scaling = 4607182418800017408; Convert Data.Offset = 0; Signal Offline Data.SPN = 4175; Signal Offline Data.Name = "DslPrtcltFltrActvRgnrtnFrcdStts"; Signal Offline Data.Description = "Indicates the forced execution status of diesel particulate filter regeneration."; Signal Offline Data.Unit = ""; Signal Offline Data.Min = 0; Signal Offline Data.Max = 7; Signal Online Data.BitSize = 3; Signal Online Data.BitPosition = 53; Convert Data.Flags = 3; Convert Data.pSigValue = 0; Convert Data.Scaling = 4607182418800017408; Convert Data.Offset = 0; PG Offline Data.Name = "AT1IG2"; PG Offline Data.Description = "Aftertreatment 1 Intake Gas 2"; PG Online Data.PGN = 64948; PG Online Data.Length (Bytes) = 8; PG Transmission Settings.Destination Address = 255; PG Transmission Settings.CycleTimeFactor = 1; Signal Offline Data.SPN = 3241; Signal Offline Data.Name = "Aftertreatment1ExhaustGasTemp1"; Signal Offline Data.Unit = "deg C"; Signal Offline Data.Min = -273; Signal Offline Data.Max = 1734.96875; Signal Online Data.BitSize = 16; Signal Online Data.BitPosition = 0; Convert Data.Flags = 3; Convert Data.pSigValue = 0; Convert Data.Scaling = 4584664420663164928; Convert Data.Offset = 13866882319836512256; Signal Offline Data.SPN = 3242; Signal Offline Data.Name = "Aftrtrtmnt1DslPrtcltFltrInt_0000";
                  Signal Offline Data.Description = "Temperature of engine combustion byproducts entering the diesel particulate filter in exhaust bank 1."; Signal Offline Data.Unit = "deg C"; Signal Offline Data.Min = -273; Signal Offline Data.Max = 1734.96875; Signal Online Data.BitSize = 16; Signal Online Data.BitPosition = 16; Convert Data.Flags = 3; Convert Data.pSigValue = 0; Convert Data.Scaling = 4584664420663164928; Convert Data.Offset = 13866882319836512256; Signal Offline Data.SPN = 3243; Signal Offline Data.Name = "Aftrtrtmnt1ExhstGsTmp1PrlmnryFMI"; Signal Offline Data.Description = "Used to identify the applicable J1939-73 FMI detected in the exhaust gas temperature 1 sensor by the manufacturer$'s"; Signal Offline Data.Unit = ""; Signal Offline Data.Min = 0; Signal Offline Data.Max = 31; Signal Online Data.BitSize = 5; Signal Online Data.BitPosition = 32; Convert Data.Flags = 3; Convert Data.pSigValue = 0; Convert Data.Scaling = 4607182418800017408; Convert Data.Offset = 0; Signal Offline Data.SPN = 3244; Signal Offline Data.Name = "Aftrtrtmnt1DslPrtcltFltrIntkGsTm"; Signal Offline Data.Unit = ""; Signal Offline Data.Min = 0; Signal Offline Data.Max = 31; Signal Online Data.BitSize = 5; Signal Online Data.BitPosition = 40; Convert Data.Flags = 3; Convert Data.pSigValue = 0; Convert Data.Scaling = 4607182418800017408; Convert Data.Offset = 0; PG Offline Data.Name = "AT1T1I"; PG Offline Data.Description = "Aftertreatment 1 SCR Reagent Tank 1 Information"; PG Online Data.PGN = 65110; PG Online Data.Length (Bytes) = 8; PG Transmission Settings.Destination Address = 255; PG Transmission Settings.CycleTimeFactor = 1; Signal Offline Data.SPN = 1761;
                  Signal Offline Data.Name = "Aftrtrtmnt1SCRCatalystTankLevel"; Signal Offline Data.Description = "A special catalyst uses a chemical reagent to reach legal requirement for NOX emissions."; Signal Offline Data.Unit = "%"; Signal Offline Data.Min = 0; Signal Offline Data.Max = 100; Signal Online Data.BitSize = 8; Signal Online Data.BitPosition = 0; Convert Data.Flags = 3; Convert Data.pSigValue = 0; Convert Data.Scaling = 4600877379321698714; Convert Data.Offset = 0; Signal Offline Data.SPN = 3031; Signal Offline Data.Name = "Aftrtrtment1SCRCatalystTankTemp"; Signal Offline Data.Description = "Temperature of the reagent in the storage tank."; Signal Offline Data.Unit = "deg C"; Signal Offline Data.Min = -40; Signal Offline Data.Max = 210; Signal Online Data.BitSize = 8; Signal Online Data.BitPosition = 8; Convert Data.Flags = 3; Convert Data.pSigValue = 0; Convert Data.Scaling = 4607182418800017408; Convert Data.Offset = 13854198353698488320; Signal Offline Data.SPN = 3517; Signal Offline Data.Name = "Aftrtrtmnt1SCRCtalystTankLevel2"; Signal Offline Data.Description = "The measure of the reagent level in the catalyst tank."; Signal Offline Data.Unit = "mm"; Signal Offline Data.Min = 0; Signal Offline Data.Max = 6425.5; Signal Online Data.BitSize = 16; Signal Online Data.BitPosition = 16; Convert Data.Flags = 3; Convert Data.pSigValue = 0; Convert Data.Scaling = 4591870180066957722; Convert Data.Offset = 0; Signal Offline Data.SPN = 3532; Signal Offline Data.Name = "Aftrtrtmnt1SCRCtlystTnkLvlPrlmnr"; Signal Offline Data.Unit = ""; Signal Offline Data.Min = 0; Signal Offline Data.Max = 31;
                  Signal Online Data.BitSize = 5; Signal Online Data.BitPosition = 32; Convert Data.Flags = 3; Convert Data.pSigValue = 0; Convert Data.Scaling = 4607182418800017408; Convert Data.Offset = 0; Signal Offline Data.SPN = 5245; Signal Offline Data.Name = "Aftrtrtmnt1DEFTnkLwLvlIndicator"; Signal Offline Data.Description = "The desired illumination of the driver$'s warning indicator for diesel exhaust fluid (DEF) tank low level."; Signal Offline Data.Unit = ""; Signal Offline Data.Min = 0; Signal Offline Data.Max = 7; Signal Online Data.BitSize = 3; Signal Online Data.BitPosition = 37; Convert Data.Flags = 3; Convert Data.pSigValue = 0; Convert Data.Scaling = 4607182418800017408; Convert Data.Offset = 0; Signal Offline Data.SPN = 4365; Signal Offline Data.Name = "Aftrtrtmnt1SCRCtlystRgntTnk1TmpP"; Signal Offline Data.Description = "Used to identify the applicable J1939-73 FMI detected in the SCR catalyst reagent tank 1 temperature, by the"; Signal Offline Data.Unit = ""; Signal Offline Data.Min = 0; Signal Offline Data.Max = 31; Signal Online Data.BitSize = 5; Signal Online Data.BitPosition = 40; Convert Data.Flags = 3; Convert Data.pSigValue = 0; Convert Data.Scaling = 4607182418800017408; Convert Data.Offset = 0; Signal Offline Data.SPN = 5246; Signal Offline Data.Name = "AftrtrtmntSCROprtrIndcmntSvrity"; Signal Offline Data.Description = "The severity of operator inducement for anomolies with the SCR system, such as tampering, low DEF quality, and DEF"; Signal Offline Data.Unit = ""; Signal Offline Data.Min = 0; Signal Offline Data.Max = 7; Signal Online Data.BitSize = 3; Signal Online Data.BitPosition = 45; Convert Data.Flags = 3; Convert Data.pSigValue = 0;
                  Convert Data.Scaling = 4607182418800017408; Convert Data.Offset = 0; Signal Offline Data.SPN = 3363; Signal Offline Data.Name = "Aftrtrtmnt1SCRCtalystTankHeater"; Signal Offline Data.Description = "Percentage of heating applied to the aftertreatment 1 catalyst tank heater."; Signal Offline Data.Unit = "%"; Signal Offline Data.Min = 0; Signal Offline Data.Max = 100; Signal Online Data.BitSize = 8; Signal Online Data.BitPosition = 48; Convert Data.Flags = 3; Convert Data.pSigValue = 0; Convert Data.Scaling = 4600877379321698714; Convert Data.Offset = 0; Signal Offline Data.SPN = 4366; Signal Offline Data.Name = "Aftrtrtmnt1SCRCtlystRgntTnk1HtrP"; Signal Offline Data.Unit = ""; Signal Offline Data.Min = 0; Signal Offline Data.Max = 31; Signal Online Data.BitSize = 5; Signal Online Data.BitPosition = 56; Convert Data.Flags = 3; Convert Data.pSigValue = 0; Convert Data.Scaling = 4607182418800017408; Convert Data.Offset = 0; PG Offline Data.Name = "A1SCRDSI1"; PG Offline Data.Description = "Aftertreatment 1 SCR Dosing System Information 1"; PG Online Data.PGN = 61475; PG Online Data.Length (Bytes) = 8; PG Transmission Settings.Destination Address = 255; PG Transmission Settings.CycleTimeFactor = 1; Signal Offline Data.SPN = 4331; Signal Offline Data.Name = "Aftrtrtmnt1SCRActlDsngRgntQntty"; Signal Offline Data.Description = "Actual reducing agent quantity of SCR-system"; Signal Offline Data.Unit = "g/h"; Signal Offline Data.Min = 0; Signal Offline Data.Max = 19276.5; Signal Online Data.BitSize = 16; Signal Online Data.BitPosition = 0; Convert Data.Flags = 3;
                  Convert Data.pSigValue = 0; Convert Data.Scaling = 4599075939470750515; Convert Data.Offset = 0; Signal Offline Data.SPN = 4332; Signal Offline Data.Name = "Aftertreatment1SCRSystemState"; Signal Offline Data.Description = "Actual state of SCR system"; Signal Offline Data.Unit = ""; Signal Offline Data.Min = 0; Signal Offline Data.Max = 15; Signal Online Data.BitSize = 4; Signal Online Data.BitPosition = 16; Convert Data.Flags = 3; Convert Data.pSigValue = 0; Convert Data.Scaling = 4607182418800017408; Convert Data.Offset = 0; Signal Offline Data.SPN = 4333; Signal Offline Data.Name = "Aftrtrtmnt1SCRActlRgntQnttyOfInt"; Signal Offline Data.Description = "The SCR requested reagent integrator total quantity for aftertreatment system 1 (exhaust bank 1)."; Signal Offline Data.Unit = "g"; Signal Offline Data.Min = 0; Signal Offline Data.Max = 6425.5; Signal Online Data.BitSize = 16; Signal Online Data.BitPosition = 24; Convert Data.Flags = 3; Convert Data.pSigValue = 0; Convert Data.Scaling = 4591870180066957722; Convert Data.Offset = 0; Signal Offline Data.SPN = 4334; Signal Offline Data.Name = "Aftrtrtmnt1SCRDsngRgentAbsPress"; Signal Offline Data.Description = "The SCR dosing reagent absolute pressure (measured closest to dosing valve) for aftertreatment system 1 (exhaust bank"; Signal Offline Data.Unit = "kPa"; Signal Offline Data.Min = 0; Signal Offline Data.Max = 2000; Signal Online Data.BitSize = 8; Signal Online Data.BitPosition = 40; Convert Data.Flags = 3; Convert Data.pSigValue = 0; Convert Data.Scaling = 4620693217682128896; Convert Data.Offset = 0; PG Offline Data.Name = "AT1T1I";
                  PG Offline Data.Description = "Aftertreatment 1 SCR Reagent Tank 1 Information"; PG Online Data.PGN = 65110; PG Online Data.Length (Bytes) = 8; PG Transmission Settings.Destination Address = 255; PG Transmission Settings.CycleTimeFactor = 1; Signal Offline Data.SPN = 1761; Signal Offline Data.Name = "Aftrtrtmnt1SCRCatalystTankLevel"; Signal Offline Data.Description = "A special catalyst uses a chemical reagent to reach legal requirement for NOX emissions."; Signal Offline Data.Unit = "%"; Signal Offline Data.Min = 0; Signal Offline Data.Max = 100; Signal Online Data.BitSize = 8; Signal Online Data.BitPosition = 0; Convert Data.Flags = 3; Convert Data.pSigValue = 0; Convert Data.Scaling = 4600877379321698714; Convert Data.Offset = 0; Signal Offline Data.SPN = 3031; Signal Offline Data.Name = "Aftrtrtment1SCRCatalystTankTemp"; Signal Offline Data.Description = "Temperature of the reagent in the storage tank."; Signal Offline Data.Unit = "deg C"; Signal Offline Data.Min = -40; Signal Offline Data.Max = 210; Signal Online Data.BitSize = 8; Signal Online Data.BitPosition = 8; Convert Data.Flags = 3; Convert Data.pSigValue = 0; Convert Data.Scaling = 4607182418800017408; Convert Data.Offset = 13854198353698488320; Signal Offline Data.SPN = 3517; Signal Offline Data.Name = "Aftrtrtmnt1SCRCtalystTankLevel2"; Signal Offline Data.Description = "The measure of the reagent level in the catalyst tank."; Signal Offline Data.Unit = "mm"; Signal Offline Data.Min = 0; Signal Offline Data.Max = 6425.5; Signal Online Data.BitSize = 16; Signal Online Data.BitPosition = 16; Convert Data.Flags = 3; Convert Data.pSigValue = 0; Convert Data.Scaling = 4591870180066957722;
                  Convert Data.Offset = 0; Signal Offline Data.SPN = 3532; Signal Offline Data.Name = "Aftrtrtmnt1SCRCtlystTnkLvlPrlmnr"; Signal Offline Data.Unit = ""; Signal Offline Data.Min = 0; Signal Offline Data.Max = 31; Signal Online Data.BitSize = 5; Signal Online Data.BitPosition = 32; Convert Data.Flags = 3; Convert Data.pSigValue = 0; Convert Data.Scaling = 4607182418800017408; Convert Data.Offset = 0; Signal Offline Data.SPN = 5245; Signal Offline Data.Name = "Aftrtrtmnt1DEFTnkLwLvlIndicator"; Signal Offline Data.Description = "The desired illumination of the driver$'s warning indicator for diesel exhaust fluid (DEF) tank low level."; Signal Offline Data.Unit = ""; Signal Offline Data.Min = 0; Signal Offline Data.Max = 7; Signal Online Data.BitSize = 3; Signal Online Data.BitPosition = 37; Convert Data.Flags = 3; Convert Data.pSigValue = 0; Convert Data.Scaling = 4607182418800017408; Convert Data.Offset = 0; Signal Offline Data.SPN = 4365; Signal Offline Data.Name = "Aftrtrtmnt1SCRCtlystRgntTnk1TmpP"; Signal Offline Data.Description = "Used to identify the applicable J1939-73 FMI detected in the SCR catalyst reagent tank 1 temperature, by the"; Signal Offline Data.Unit = ""; Signal Offline Data.Min = 0; Signal Offline Data.Max = 31; Signal Online Data.BitSize = 5; Signal Online Data.BitPosition = 40; Convert Data.Flags = 3; Convert Data.pSigValue = 0; Convert Data.Scaling = 4607182418800017408; Convert Data.Offset = 0; Signal Offline Data.SPN = 5246; Signal Offline Data.Name = "AftrtrtmntSCROprtrIndcmntSvrity"; Signal Offline Data.Description = "The severity of operator inducement for anomolies with the SCR system, such as tampering, low DEF quality, and DEF"; Signal Offline Data.Unit = "";
                  Signal Offline Data.Min = 0; Signal Offline Data.Max = 7; Signal Online Data.BitSize = 3; Signal Online Data.BitPosition = 45; Convert Data.Flags = 3; Convert Data.pSigValue = 0; Convert Data.Scaling = 4607182418800017408; Convert Data.Offset = 0; Signal Offline Data.SPN = 3363; Signal Offline Data.Name = "Aftrtrtmnt1SCRCtalystTankHeater"; Signal Offline Data.Description = "Percentage of heating applied to the aftertreatment 1 catalyst tank heater."; Signal Offline Data.Unit = "%"; Signal Offline Data.Min = 0; Signal Offline Data.Max = 100; Signal Online Data.BitSize = 8; Signal Online Data.BitPosition = 48; Convert Data.Flags = 3; Convert Data.pSigValue = 0; Convert Data.Scaling = 4600877379321698714; Convert Data.Offset = 0; Signal Offline Data.SPN = 4366; Signal Offline Data.Name = "Aftrtrtmnt1SCRCtlystRgntTnk1HtrP"; Signal Offline Data.Unit = ""; Signal Offline Data.Min = 0; Signal Offline Data.Max = 31; Signal Online Data.BitSize = 5; Signal Online Data.BitPosition = 56; Convert Data.Flags = 3; Convert Data.pSigValue = 0; Convert Data.Scaling = 4607182418800017408; Convert Data.Offset = 0; PG Offline Data.Name = "A1SCREGT"; PG Offline Data.Description = "Aftertreatment 1 SCR Exhaust Gas Temperature"; PG Online Data.PGN = 64830; PG Online Data.Length (Bytes) = 8; PG Transmission Settings.Destination Address = 255; PG Transmission Settings.CycleTimeFactor = 1; Signal Offline Data.SPN = 4360; Signal Offline Data.Name = "Aftrtrtmnt1SCRCtlystIntkGasTemp"; Signal Offline Data.Description = "Temperature of engine combustion byproducts entering the SCR catalyst in exhaust bank 1.";
                  Signal Offline Data.Unit = "deg C"; Signal Offline Data.Min = -273; Signal Offline Data.Max = 1734.96875; Signal Online Data.BitSize = 16; Signal Online Data.BitPosition = 0; Convert Data.Flags = 3; Convert Data.pSigValue = 0; Convert Data.Scaling = 4584664420663164928; Convert Data.Offset = 13866882319836512256; Signal Offline Data.SPN = 4361; Signal Offline Data.Name = "Aftrtrtmnt1SCRCtlystIntkGsTmpPrl"; Signal Offline Data.Description = "Used to identify the applicable J1939-73 FMI detected in the SCR catalyst intake gas temperature sensor by the"; Signal Offline Data.Unit = ""; Signal Offline Data.Min = 0; Signal Offline Data.Max = 31; Signal Online Data.BitSize = 5; Signal Online Data.BitPosition = 16; Convert Data.Flags = 3; Convert Data.pSigValue = 0; Convert Data.Scaling = 4607182418800017408; Convert Data.Offset = 0; Signal Offline Data.SPN = 4363; Signal Offline Data.Name = "Aftrtrtmnt1SCRCtlystOtltGasTemp"; Signal Offline Data.Description = "Temperature of engine combustion byproducts leaving the SCR catalyst exhaust in exhaust bank 1."; Signal Offline Data.Unit = "deg C"; Signal Offline Data.Min = -273; Signal Offline Data.Max = 1734.96875; Signal Online Data.BitSize = 16; Signal Online Data.BitPosition = 24; Convert Data.Flags = 3; Convert Data.pSigValue = 0; Convert Data.Scaling = 4584664420663164928; Convert Data.Offset = 13866882319836512256; Signal Offline Data.SPN = 4362; Signal Offline Data.Name = "Aftrtrtmnt1SCRCtlystOtltGsTmpPrl"; Signal Offline Data.Description = "Used to identify the applicable J1939-73 FMI detected in the SCR catalyst outlet gas temperature sensor by the"; Signal Offline Data.Unit = ""; Signal Offline Data.Min = 0; Signal Offline Data.Max = 31; Signal Online Data.BitSize = 5;
                  Signal Online Data.BitPosition = 40; Convert Data.Flags = 3; Convert Data.pSigValue = 0; Convert Data.Scaling = 4607182418800017408; Convert Data.Offset = 0; PG Offline Data.Name = "A1DOC"; PG Offline Data.Description = "Aftertreatment 1 Diesel Oxidation Catalyst"; PG Online Data.PGN = 64800; PG Online Data.Length (Bytes) = 8; PG Transmission Settings.Destination Address = 255; PG Transmission Settings.CycleTimeFactor = 1; Signal Offline Data.SPN = 4765; Signal Offline Data.Name = "Aftrtrtmnt1DslOxdtnCtlystIn_0000"; Signal Offline Data.Description = "Temperature of engine combustion byproducts entering the diesel oxidation catalyst in exhaust bank 1."; Signal Offline Data.Unit = "deg C"; Signal Offline Data.Min = -273; Signal Offline Data.Max = 1734.96875; Signal Online Data.BitSize = 16; Signal Online Data.BitPosition = 0; Convert Data.Flags = 3; Convert Data.pSigValue = 0; Convert Data.Scaling = 4584664420663164928; Convert Data.Offset = 13866882319836512256; Signal Offline Data.SPN = 4766; Signal Offline Data.Name = "Aftrtrtmnt1DslOxdtnCtlystOt_0000"; Signal Offline Data.Description = "Temperature of engine combustion byproducts leaving the diesel oxidation catalyst exhaust in exhaust bank 1."; Signal Offline Data.Unit = "deg C"; Signal Offline Data.Min = -273; Signal Offline Data.Max = 1734.96875; Signal Online Data.BitSize = 16; Signal Online Data.BitPosition = 16; Convert Data.Flags = 3; Convert Data.pSigValue = 0; Convert Data.Scaling = 4584664420663164928; Convert Data.Offset = 13866882319836512256; Signal Offline Data.SPN = 4767; Signal Offline Data.Name = "Aftrtrtmnt1DslOxdtnCtlystDffPrss"; Signal Offline Data.Unit = "kPa"; Signal Offline Data.Min = 0; Signal Offline Data.Max = 6425.5;
                  Signal Online Data.BitSize = 16; Signal Online Data.BitPosition = 32; Convert Data.Flags = 3; Convert Data.pSigValue = 0; Convert Data.Scaling = 4591870180066957722; Convert Data.Offset = 0; Signal Offline Data.SPN = 4768; Signal Offline Data.Name = "Aftrtrtmnt1DslOxdtnCtlystIntkGsT"; Signal Offline Data.Unit = ""; Signal Offline Data.Min = 0; Signal Offline Data.Max = 31; Signal Online Data.BitSize = 5; Signal Online Data.BitPosition = 48; Convert Data.Flags = 3; Convert Data.pSigValue = 0; Convert Data.Scaling = 4607182418800017408; Convert Data.Offset = 0; Signal Offline Data.SPN = 4769; Signal Offline Data.Name = "Aftrtrtmnt1DslOxdtnCtlystOtltGsT"; Signal Offline Data.Unit = ""; Signal Offline Data.Min = 0; Signal Offline Data.Max = 31; Signal Online Data.BitSize = 5; Signal Online Data.BitPosition = 53; Convert Data.Flags = 3; Convert Data.pSigValue = 0; Convert Data.Scaling = 4607182418800017408; Convert Data.Offset = 0; Signal Offline Data.SPN = 4770; Signal Offline Data.Name = "Aftrtrtmnt1DslOxdtnCtlystDf_0000"; Signal Offline Data.Unit = ""; Signal Offline Data.Min = 0; Signal Offline Data.Max = 31; Signal Online Data.BitSize = 5; Signal Online Data.BitPosition = 58; Convert Data.Flags = 3; Convert Data.pSigValue = 0; Convert Data.Scaling = 4607182418800017408; Convert Data.Offset = 0; PG Offline Data.Name = "WFI";
                  PG Offline Data.Description = "Water in Fuel Indicator"; PG Online Data.PGN = 65279; PG Online Data.Length (Bytes) = 8; PG Transmission Settings.Destination Address = 255; PG Transmission Settings.CycleTimeFactor = 1; Signal Offline Data.SPN = 97; Signal Offline Data.Name = "WaterInFuelIndicator"; Signal Offline Data.Description = "Signal which indicates the presence of water in the fuel."; Signal Offline Data.Unit = ""; Signal Offline Data.Min = 0; Signal Offline Data.Max = 3; Signal Online Data.BitSize = 2; Signal Online Data.BitPosition = 0; Convert Data.Flags = 3; Convert Data.pSigValue = 0; Convert Data.Scaling = 4607182418800017408; Convert Data.Offset = 0; PG Offline Data.Name = "DLCC1"; PG Offline Data.Description = "Direct Lamp Control Command 1"; PG Online Data.PGN = 64775; PG Online Data.Length (Bytes) = 8; PG Transmission Settings.Destination Address = 255; PG Transmission Settings.CycleTimeFactor = 1; Signal Offline Data.SPN = 5077; Signal Offline Data.Name = "EngProtectLampCmd"; Signal Offline Data.Description = "Command signal directly controlling the Engine Protect Lamp"; Signal Offline Data.Unit = ""; Signal Offline Data.Min = 0; Signal Offline Data.Max = 3; Signal Online Data.BitSize = 2; Signal Online Data.BitPosition = 0; Convert Data.Flags = 3; Convert Data.pSigValue = 0; Convert Data.Scaling = 4607182418800017408; Convert Data.Offset = 0; Signal Offline Data.SPN = 5078; Signal Offline Data.Name = "EngAmberWarningLampCmd"; Signal Offline Data.Description = "Command signal directly controlling the Engine Amber Warning Lamp"; Signal Offline Data.Unit = ""; Signal Offline Data.Min = 0;
                  Signal Offline Data.Max = 3; Signal Online Data.BitSize = 2; Signal Online Data.BitPosition = 2; Convert Data.Flags = 3; Convert Data.pSigValue = 0; Convert Data.Scaling = 4607182418800017408; Convert Data.Offset = 0; Signal Offline Data.SPN = 5079; Signal Offline Data.Name = "EngRedStopLampCmd"; Signal Offline Data.Description = "Command signal directly controlling the Engine Red Stop Lamp"; Signal Offline Data.Unit = ""; Signal Offline Data.Min = 0; Signal Offline Data.Max = 3; Signal Online Data.BitSize = 2; Signal Online Data.BitPosition = 4; Convert Data.Flags = 3; Convert Data.pSigValue = 0; Convert Data.Scaling = 4607182418800017408; Convert Data.Offset = 0; Signal Offline Data.SPN = 5080; Signal Offline Data.Name = "OBDMalfunctionIndicatorLampCmd"; Signal Offline Data.Description = "Command signal directly controlling the OBD Malfunction Indicator Lamp"; Signal Offline Data.Unit = ""; Signal Offline Data.Min = 0; Signal Offline Data.Max = 3; Signal Online Data.BitSize = 2; Signal Online Data.BitPosition = 6; Convert Data.Flags = 3; Convert Data.pSigValue = 0; Convert Data.Scaling = 4607182418800017408; Convert Data.Offset = 0; Signal Offline Data.SPN = 5081; Signal Offline Data.Name = "EngBrakeActiveLampCmd"; Signal Offline Data.Description = "Command signal directly controlling the Engine Brake Active Lamp"; Signal Offline Data.Unit = ""; Signal Offline Data.Min = 0; Signal Offline Data.Max = 3; Signal Online Data.BitSize = 2; Signal Online Data.BitPosition = 8; Convert Data.Flags = 3;
                  Convert Data.pSigValue = 0; Convert Data.Scaling = 4607182418800017408; Convert Data.Offset = 0; Signal Offline Data.SPN = 3987; Signal Offline Data.Name = "CmprssnBrkEnblSwtchIndctrLmpCmd"; Signal Offline Data.Description = "Command signal directly controlling Compression Brake Enable Switch Indicator Lamp."; Signal Offline Data.Unit = ""; Signal Offline Data.Min = 0; Signal Offline Data.Max = 3; Signal Online Data.BitSize = 2; Signal Online Data.BitPosition = 10; Convert Data.Flags = 3; Convert Data.pSigValue = 0; Convert Data.Scaling = 4607182418800017408; Convert Data.Offset = 0; Signal Offline Data.SPN = 5082; Signal Offline Data.Name = "EngOilPressLowLampCmd"; Signal Offline Data.Description = "Command signal directly controlling the Engine Oil Pressure Low Lamp"; Signal Offline Data.Unit = ""; Signal Offline Data.Min = 0; Signal Offline Data.Max = 3; Signal Online Data.BitSize = 2; Signal Online Data.BitPosition = 12; Convert Data.Flags = 3; Convert Data.pSigValue = 0; Convert Data.Scaling = 4607182418800017408; Convert Data.Offset = 0; Signal Offline Data.SPN = 5083; Signal Offline Data.Name = "EngCoolantTempHighLampCmd"; Signal Offline Data.Description = "Command signal directly controlling the Engine Coolant Temperature High Lamp"; Signal Offline Data.Unit = ""; Signal Offline Data.Min = 0; Signal Offline Data.Max = 3; Signal Online Data.BitSize = 2; Signal Online Data.BitPosition = 14; Convert Data.Flags = 3; Convert Data.pSigValue = 0; Convert Data.Scaling = 4607182418800017408; Convert Data.Offset = 0; Signal Offline Data.SPN = 5084;
                  Signal Offline Data.Name = "EngCoolantLevelLowLampCmd"; Signal Offline Data.Description = "Command signal directly controlling the Engine Coolant Level Low Lamp"; Signal Offline Data.Unit = ""; Signal Offline Data.Min = 0; Signal Offline Data.Max = 3; Signal Online Data.BitSize = 2; Signal Online Data.BitPosition = 16; Convert Data.Flags = 3; Convert Data.pSigValue = 0; Convert Data.Scaling = 4607182418800017408; Convert Data.Offset = 0; Signal Offline Data.SPN = 5085; Signal Offline Data.Name = "EngIdleManagementActiveLampCmd"; Signal Offline Data.Description = "Command signal directly controlling the Engine Idle Management Active Lamp"; Signal Offline Data.Unit = ""; Signal Offline Data.Min = 0; Signal Offline Data.Max = 3; Signal Online Data.BitSize = 2; Signal Online Data.BitPosition = 18; Convert Data.Flags = 3; Convert Data.pSigValue = 0; Convert Data.Scaling = 4607182418800017408; Convert Data.Offset = 0; Signal Offline Data.SPN = 5086; Signal Offline Data.Name = "EngAirFilterRestrictionLampCmd"; Signal Offline Data.Description = "Command signal directly controlling the Engine Air Filter Restriction Lamp."; Signal Offline Data.Unit = ""; Signal Offline Data.Min = 0; Signal Offline Data.Max = 3; Signal Online Data.BitSize = 2; Signal Online Data.BitPosition = 20; Convert Data.Flags = 3; Convert Data.pSigValue = 0; Convert Data.Scaling = 4607182418800017408; Convert Data.Offset = 0; Signal Offline Data.SPN = 5469; Signal Offline Data.Name = "EngFuelFilterRestrictedLampCmd"; Signal Offline Data.Description = "Command signal directly controlling the Vehicle Fuel Filter Restricted Lamp."; Signal Offline Data.Unit = ""; Signal Offline Data.Min = 0;
                  Signal Offline Data.Max = 3; Signal Online Data.BitSize = 2; Signal Online Data.BitPosition = 22; Convert Data.Flags = 3; Convert Data.pSigValue = 0; Convert Data.Scaling = 4607182418800017408; Convert Data.Offset = 0; PG Offline Data.Name = "DLCD1"; PG Offline Data.Description = "Direct Lamp Control Data 1"; PG Online Data.PGN = 64773; PG Online Data.Length (Bytes) = 8; PG Transmission Settings.Destination Address = 255; PG Transmission Settings.CycleTimeFactor = 1; Signal Offline Data.SPN = 5093; Signal Offline Data.Name = "EngProtectLampData"; Signal Offline Data.Description = "This parameter provides measured data from the Engine Protect Lamp."; Signal Offline Data.Unit = ""; Signal Offline Data.Min = 0; Signal Offline Data.Max = 3; Signal Online Data.BitSize = 2; Signal Online Data.BitPosition = 0; Convert Data.Flags = 3; Convert Data.pSigValue = 0; Convert Data.Scaling = 4607182418800017408; Convert Data.Offset = 0; Signal Offline Data.SPN = 5094; Signal Offline Data.Name = "EngAmberWarningLampData"; Signal Offline Data.Description = "This parameter provides measured data from the Engine Amber Warning Lamp."; Signal Offline Data.Unit = ""; Signal Offline Data.Min = 0; Signal Offline Data.Max = 3; Signal Online Data.BitSize = 2; Signal Online Data.BitPosition = 2; Convert Data.Flags = 3; Convert Data.pSigValue = 0; Convert Data.Scaling = 4607182418800017408; Convert Data.Offset = 0; Signal Offline Data.SPN = 5095; Signal Offline Data.Name = "EngRedStopLampData"; Signal Offline Data.Description = "This parameter provides measured data from the Engine Red Stop Lamp.";
                  Signal Offline Data.Unit = ""; Signal Offline Data.Min = 0; Signal Offline Data.Max = 3; Signal Online Data.BitSize = 2; Signal Online Data.BitPosition = 4; Convert Data.Flags = 3; Convert Data.pSigValue = 0; Convert Data.Scaling = 4607182418800017408; Convert Data.Offset = 0; Signal Offline Data.SPN = 5096; Signal Offline Data.Name = "OBDMalfunctionIndicatorLampData"; Signal Offline Data.Description = "This parameter provides measured data from the OBD Malfunction Indicator Lamp."; Signal Offline Data.Unit = ""; Signal Offline Data.Min = 0; Signal Offline Data.Max = 3; Signal Online Data.BitSize = 2; Signal Online Data.BitPosition = 6; Convert Data.Flags = 3; Convert Data.pSigValue = 0; Convert Data.Scaling = 4607182418800017408; Convert Data.Offset = 0; Signal Offline Data.SPN = 5097; Signal Offline Data.Name = "EngBrakeActiveLampData"; Signal Offline Data.Description = "This parameter provides measured data from the Engine Brake Active Lamp."; Signal Offline Data.Unit = ""; Signal Offline Data.Min = 0; Signal Offline Data.Max = 3; Signal Online Data.BitSize = 2; Signal Online Data.BitPosition = 8; Convert Data.Flags = 3; Convert Data.pSigValue = 0; Convert Data.Scaling = 4607182418800017408; Convert Data.Offset = 0; Signal Offline Data.SPN = 5098; Signal Offline Data.Name = "CmprssnBrkEnblSwtchIndctrLmpDta"; Signal Offline Data.Description = "This parameter provides measured data from the Compression Brake Enable Switch Indicator Lamp."; Signal Offline Data.Unit = ""; Signal Offline Data.Min = 0; Signal Offline Data.Max = 3; Signal Online Data.BitSize = 2;
                  Signal Online Data.BitPosition = 10; Convert Data.Flags = 3; Convert Data.pSigValue = 0; Convert Data.Scaling = 4607182418800017408; Convert Data.Offset = 0; Signal Offline Data.SPN = 5099; Signal Offline Data.Name = "EngOilPressLowLampData"; Signal Offline Data.Description = "This parameter provides measured data from the Engine Oil Pressure Low Lamp."; Signal Offline Data.Unit = ""; Signal Offline Data.Min = 0; Signal Offline Data.Max = 3; Signal Online Data.BitSize = 2; Signal Online Data.BitPosition = 12; Convert Data.Flags = 3; Convert Data.pSigValue = 0; Convert Data.Scaling = 4607182418800017408; Convert Data.Offset = 0; Signal Offline Data.SPN = 5100; Signal Offline Data.Name = "EngCoolantTempHighLampData"; Signal Offline Data.Description = "This parameter provides measured data from the Engine Coolant Temperature High Lamp."; Signal Offline Data.Unit = ""; Signal Offline Data.Min = 0; Signal Offline Data.Max = 3; Signal Online Data.BitSize = 2; Signal Online Data.BitPosition = 14; Convert Data.Flags = 3; Convert Data.pSigValue = 0; Convert Data.Scaling = 4607182418800017408; Convert Data.Offset = 0; Signal Offline Data.SPN = 5101; Signal Offline Data.Name = "EngCoolantLevelLowLampData"; Signal Offline Data.Description = "This parameter provides measured data from the Engine Coolant Level Low Lamp."; Signal Offline Data.Unit = ""; Signal Offline Data.Min = 0; Signal Offline Data.Max = 3; Signal Online Data.BitSize = 2; Signal Online Data.BitPosition = 16; Convert Data.Flags = 3; Convert Data.pSigValue = 0; Convert Data.Scaling = 4607182418800017408;
                  Convert Data.Offset = 0; Signal Offline Data.SPN = 5102; Signal Offline Data.Name = "EngIdleManagementActiveLampData"; Signal Offline Data.Description = "This parameter provides measured data from the Engine Idle Management Active Lamp."; Signal Offline Data.Unit = ""; Signal Offline Data.Min = 0; Signal Offline Data.Max = 3; Signal Online Data.BitSize = 2; Signal Online Data.BitPosition = 18; Convert Data.Flags = 3; Convert Data.pSigValue = 0; Convert Data.Scaling = 4607182418800017408; Convert Data.Offset = 0; Signal Offline Data.SPN = 5103; Signal Offline Data.Name = "EngAirFilterRestrictionLampData"; Signal Offline Data.Description = "This parameter provides measured data from the Engine Air Filter Restriction Lamp."; Signal Offline Data.Unit = ""; Signal Offline Data.Min = 0; Signal Offline Data.Max = 3; Signal Online Data.BitSize = 2; Signal Online Data.BitPosition = 20; Convert Data.Flags = 3; Convert Data.pSigValue = 0; Convert Data.Scaling = 4607182418800017408; Convert Data.Offset = 0; Signal Offline Data.SPN = 5470; Signal Offline Data.Name = "EngFuelFilterRestrictedLampData"; Signal Offline Data.Description = "Command signal directly controlling the Vehicle Fuel Filter Restricted Lamp."; Signal Offline Data.Unit = ""; Signal Offline Data.Min = 0; Signal Offline Data.Max = 3; Signal Online Data.BitSize = 2; Signal Online Data.BitPosition = 22; Convert Data.Flags = 3; Convert Data.pSigValue = 0; Convert Data.Scaling = 4607182418800017408; Convert Data.Offset = 0; Signal Offline Data.SPN = 5416; Signal Offline Data.Name = "EngWaitToStartLampData"; Signal Offline Data.Description = "This parameter provides measured data from the Engine Wait To Start Lamp.";
                  Signal Offline Data.Unit = ""; Signal Offline Data.Min = 0; Signal Offline Data.Max = 3; Signal Online Data.BitSize = 2; Signal Online Data.BitPosition = 62; Convert Data.Flags = 3; Convert Data.pSigValue = 0; Convert Data.Scaling = 4607182418800017408; Convert Data.Offset = 0; PG Offline Data.Name = "HOURS"; PG Offline Data.Description = "Engine Hours, Revolutions"; PG Online Data.PGN = 65253; PG Online Data.Length (Bytes) = 8; PG Transmission Settings.Destination Address = 255; PG Transmission Settings.CycleTimeFactor = 1; Signal Offline Data.SPN = 247; Signal Offline Data.Name = "EngTotalHoursOfOperation"; Signal Offline Data.Description = "Accumulated time of operation of engine."; Signal Offline Data.Unit = "hr"; Signal Offline Data.Min = 0; Signal Offline Data.Max = 210554060.75; Signal Online Data.BitSize = 32; Signal Online Data.BitPosition = 0; Convert Data.Flags = 3; Convert Data.pSigValue = 0; Convert Data.Scaling = 4587366580439587226; Convert Data.Offset = 0; Signal Offline Data.SPN = 249; Signal Offline Data.Name = "EngTotalRevolutions"; Signal Offline Data.Description = "Accumulated number of revolutions of engine crankshaft during its operation."; Signal Offline Data.Unit = "r"; Signal Offline Data.Min = 0; Signal Offline Data.Max = 4211081215000; Signal Online Data.BitSize = 32; Signal Online Data.BitPosition = 32; Convert Data.Flags = 3; Convert Data.pSigValue = 0; Convert Data.Scaling = 4652007308841189376; Convert Data.Offset = 0; Activated PGs = 0
                input  Application.GVL_J1939.EEC1_ActualEngPercentTorque : INT  // ActualEngPercentTorque
                input  Application.GVL_J1939.EEC1_EngSpeed : REAL  // EngSpeed
                input  Application.GVL_J1939.EEC2_EngPercentLoadAtCurrentSpeed : USINT  // EngPercentLoadAtCurrentSpeed
                input  Application.GVL_J1939.EEC2_SCRThermalManagementActive : USINT  // SCRThermalManagementActive
                input  Application.GVL_J1939.EEC2_ActlMxAvailableEngPercentTorque : REAL  // ActlMxAvailableEngPercentTorque
                input  Application.GVL_J1939.EEC3_NominalFrictionPercentTorque : INT  // NominalFrictionPercentTorque
                input  Application.GVL_J1939.EEC3_EngsDesiredOperatingSpeed : REAL  // EngsDesiredOperatingSpeed
                input  Application.GVL_J1939.EEC5_EngExhstGsRcrculation1ValveCtrl : REAL  // EngExhstGsRcrculation1ValveCtrl
                input  Application.GVL_J1939.ET1_EngCoolantTemp : INT  // EngCoolantTemp
                input  Application.GVL_J1939.ET1_EngFuelTemp1 : INT  // EngFuelTemp1
                input  Application.GVL_J1939.EFL_P1_EngOilPress : UINT  // EngOilPress
                input  Application.GVL_J1939.EFL_P1_EngCoolantLevel : REAL  // EngCoolantLevel
                input  Application.GVL_J1939.EFL_P2_EngInjectorMeteringRail1Press : LREAL  // EngInjectorMeteringRail1Press
                input  Application.GVL_J1939.LFC_EngTotalFuelUsed : REAL  // EngTotalFuelUsed
                input  Application.GVL_J1939.AMB_BarometricPress : REAL  // BarometricPress
                input  Application.GVL_J1939.AMB_AmbientAirTemp : REAL  // AmbientAirTemp
                input  Application.GVL_J1939.AMB_EngAirIntakeTemp : INT  // EngAirIntakeTemp
                input  Application.GVL_J1939.IC1_EngIntakeManifold1Press : UINT  // EngIntakeManifold1Press
                input  Application.GVL_J1939.IC1_EngIntakeManifold1Temp : INT  // EngIntakeManifold1Temp
                input  Application.GVL_J1939.IC1_EngAirIntakePress : UINT  // EngAirIntakePress
                input  Application.GVL_J1939.VEP1_BatteryPotential_PowerInput1 : REAL  // BatteryPotential_PowerInput1
                input  Application.GVL_J1939.VEP1_KeyswitchBatteryPotential : REAL  // KeyswitchBatteryPotential
                input  Application.GVL_J1939.EFS_EngOilPrimingState : USINT  // EngOilPrimingState
                input  Application.GVL_J1939.EFS_FuelPumpPrimerStatus : USINT  // FuelPumpPrimerStatus
                input  Application.GVL_J1939.DPFC1_DieselParticulateFilterLampCmd : USINT  // DieselParticulateFilterLampCmd
                input  Application.GVL_J1939.DPFC1_DslPrtcltFltrActvRgnrtionStatus : USINT  // DslPrtcltFltrActvRgnrtionStatus
                input  Application.GVL_J1939.DPFC1_DieselParticulateFilterStatus : USINT  // DieselParticulateFilterStatus
                input  Application.GVL_J1939.DPFC1_DslPrtcltFltrActvRgnrtnInhbtdDTI : USINT  // DslPrtcltFltrActvRgnrtnInhbtdDTI
                input  Application.GVL_J1939.DPFC1_DslPrtcltFltrActvRgnrtnInhbtdDTT : USINT  // DslPrtcltFltrActvRgnrtnInhbtdDTT
                input  Application.GVL_J1939.DPFC1_DslPrtcltFltrActvRgnrtnInhbtdDTP : USINT  // DslPrtcltFltrActvRgnrtnInhbtdDTP
                input  Application.GVL_J1939.AT1IG2_Aftrtrtmnt1DslPrtcltFltrInt_0000 : REAL  // Aftrtrtmnt1DslPrtcltFltrInt_0000
                input  Application.GVL_J1939.AT1T1I_Aftrtrtmnt1SCRCatalystTankLevel : REAL  // Aftrtrtmnt1SCRCatalystTankLevel
                input  Application.GVL_J1939.AT1T1I_Aftrtrtment1SCRCatalystTankTemp : INT  // Aftrtrtment1SCRCatalystTankTemp
                input  Application.GVL_J1939.AT1T1I_Aftrtrtmnt1DEFTnkLwLvlIndicator : USINT  // Aftrtrtmnt1DEFTnkLwLvlIndicator
                input  Application.GVL_J1939.AT1T1I_AftrtrtmntSCROprtrIndcmntSvrity : USINT  // AftrtrtmntSCROprtrIndcmntSvrity
                input  Application.GVL_J1939.A1SCRDSI1_Aftertreatment1SCRSystemState : USINT  // Aftertreatment1SCRSystemState
                input  Application.GVL_J1939.A1SCREGT_Aftrtrtmnt1SCRCtlystIntkGasTemp : REAL  // Aftrtrtmnt1SCRCtlystIntkGasTemp
                input  Application.GVL_J1939.A1DOC_Aftrtrtmnt1DslOxdtnCtlystIn_0000 : REAL  // Aftrtrtmnt1DslOxdtnCtlystIn_0000
                input  Application.GVL_J1939.WFI_WaterInFuelIndicator : USINT  // WaterInFuelIndicator
                input  Application.GVL_J1939.DLCC1_EngAirFilterRestrictionLampCmd : USINT  // EngAirFilterRestrictionLampCmd
                input  Application.GVL_J1939.DLCD1_EngOilPressLowLampData : USINT  // EngOilPressLowLampData
                input  Application.GVL_J1939.DLCD1_EngCoolantLevelLowLampData : USINT  // EngCoolantLevelLowLampData
                input  Application.GVL_J1939.HOURS_EngTotalHoursOfOperation : REAL  // EngTotalHoursOfOperation
                unmapped channels: EngTorqueMode, ActlEngPrcntTrqueHighResolution, DriversDemandEngPercentTorque, SrcAddrssOfCtrllngDvcFrEngCntrl, EngStarterMode, EngDemandPercentTorque, AccelPedal1LowIdleSwitch, AccelPedalKickdownSwitch, RoadSpeedLimitStatus, AccelPedal2LowIdleSwitch, AccelPedalPos1, RemoteAccelPedalPos, AccelPedalPos2, VhclAccelerationRateLimitStatus, MmntryEngMaxPowerEnableFeedback, DPFThermalManagementActive, EstPumpingPercentTorque, EngsDsrdOprtngSpdAsymmtryAdjstmn, EstEngPrsticLossesPercentTorque, Aftrtratment1ExhaustGasMassFlow, Aftertreatment1IntakeDewPoint, Aftertreatment1ExhaustDewPoint, Aftertreatment2IntakeDewPoint, Aftertreatment2ExhaustDewPoint, EngTrb1ClcltedTurbineIntakeTemp, EngTrb1ClcltedTurbineOutletTemp, EngVrblGmtryTrbArCtrlShtffValve, EngVrableGeometryTurbo1CtrlMode, EngVrblGometryTurbo1ActuatorPos, EngOilTemp1, EngTurboOilTemp, EngIntercoolerTemp, EngIntercoolerThermostatOpening, EngFuelDeliveryPress, EngExCrankcaseBlowbyPress, EngOilLevel, EngCrankcasePress, EngCoolantPress, EngInjectionCtrlPress, EngInjectorTimingRail1Press,
                  EngInjectorMeteringRail2Press, EngTripFuel, CabInteriorTemp, RoadSurfaceTemp, EngDslPrtclateFilterIntakePress, EngAirFilter1DiffPress, EngExhaustGasTemp, EngCoolantFilterDiffPress, NetBatteryCurrent, AltCurrent, ChargingSystemPotential, EngOilLevelRemoteReservoir, EngFuelSupplyPumpIntakePress, EngFuelFilterDiffPress, EngWasteOilReservoirLevel, EngOilFilterOutletPress, EngOilPrimingPumpSwitch, EngOilPreHeatedState, EngCoolantPreheatedState, EngVentilationStatus, DslPrtcltFltrPssvRgnrtionStatus, DslPrtcltFltrActvRgnrtnInhbtdStt, DslPrtcltFltrActvRgnrtnInhbtdDTC, DslPrtcltFltrActvRgnrtnInhb_0004, DslPrtcltFltrActvRgnrtnInhb_0003, DslPrtcltFltrActvRgnrtnInhbtdDTA, DslPrtcltFltrActvRgnrtnInhbtdDTO, DslPrtcltFltrActvRgnrtnInhb_0002, DslPrtcltFltrActvRgnrtnInhb_0001, DslPrtcltFltrActvRgnrtnInhbtdDTL, DslPrtcltFltrActvRgnrtnInhb_0000, DslPrtcltFltrActvRgnrtnInhbtdDTS, DslPrtcltFltrActvRgnrtnInhbtdDTE, DslPrtcltFltrActvRgnrtnInhbtdDTV, DslPrtcltFltrAtmtcActvRgnrtnIntt, ExhaustSystemHighTempLampCmd, DslPrtcltFltrActvRgnrtnFrcdStts, Aftertreatment1ExhaustGasTemp1, Aftrtrtmnt1ExhstGsTmp1PrlmnryFMI, Aftrtrtmnt1DslPrtcltFltrIntkGsTm,
                  Aftrtrtmnt1SCRCtalystTankLevel2, Aftrtrtmnt1SCRCtlystTnkLvlPrlmnr, Aftrtrtmnt1SCRCtlystRgntTnk1TmpP, Aftrtrtmnt1SCRCtalystTankHeater, Aftrtrtmnt1SCRCtlystRgntTnk1HtrP, Aftrtrtmnt1SCRActlDsngRgntQntty, Aftrtrtmnt1SCRActlRgntQnttyOfInt, Aftrtrtmnt1SCRDsngRgentAbsPress, Aftrtrtmnt1SCRCatalystTankLevel, Aftrtrtment1SCRCatalystTankTemp, Aftrtrtmnt1SCRCtalystTankLevel2, Aftrtrtmnt1SCRCtlystTnkLvlPrlmnr, Aftrtrtmnt1DEFTnkLwLvlIndicator, Aftrtrtmnt1SCRCtlystRgntTnk1TmpP, AftrtrtmntSCROprtrIndcmntSvrity, Aftrtrtmnt1SCRCtalystTankHeater, Aftrtrtmnt1SCRCtlystRgntTnk1HtrP, Aftrtrtmnt1SCRCtlystIntkGsTmpPrl, Aftrtrtmnt1SCRCtlystOtltGasTemp, Aftrtrtmnt1SCRCtlystOtltGsTmpPrl, Aftrtrtmnt1DslOxdtnCtlystOt_0000, Aftrtrtmnt1DslOxdtnCtlystDffPrss, Aftrtrtmnt1DslOxdtnCtlystIntkGsT, Aftrtrtmnt1DslOxdtnCtlystOtltGsT, Aftrtrtmnt1DslOxdtnCtlystDf_0000, EngProtectLampCmd, EngAmberWarningLampCmd, EngRedStopLampCmd, OBDMalfunctionIndicatorLampCmd, EngBrakeActiveLampCmd, CmprssnBrkEnblSwtchIndctrLmpCmd, EngOilPressLowLampCmd, EngCoolantTempHighLampCmd, EngCoolantLevelLowLampCmd, EngIdleManagementActiveLampCmd, EngFuelFilterRestrictedLampCmd, EngProtectLampData, EngAmberWarningLampData, EngRedStopLampData, OBDMalfunctionIndicatorLampData,
                  EngBrakeActiveLampData, CmprssnBrkEnblSwtchIndctrLmpDta, EngCoolantTempHighLampData, EngIdleManagementActiveLampData, EngAirFilterRestrictionLampData, EngFuelFilterRestrictedLampData, EngWaitToStartLampData, EngTotalRevolutions
  libraries: AlarmManager, * (Intern)
  global variables GVL
  text list GlobalTextList
  GlobalImagePool
  5ce3da45-db07-42e7-a21c-a00fff4ed8f6|C:\Users\a.werner\Documents\background.jpg
  5ce3da45-db07-42e7-a21c-a00fff4ed8f6|..\LIBS\images\Page_nav_right.png
  5ce3da45-db07-42e7-a21c-a00fff4ed8f6|warning_32_32.bmp
  5ce3da45-db07-42e7-a21c-a00fff4ed8f6|D:\dev_plc\SLL\SLL_Truck_Demo\LIBS\images\CR1076_240_200.png
  5ce3da45-db07-42e7-a21c-a00fff4ed8f6|..\LIBS\images\home_32_32_white.png
  5ce3da45-db07-42e7-a21c-a00fff4ed8f6|C:\Dev\Boeing_CT6000\Software\LIBS\images\circle_34_32.png
  5ce3da45-db07-42e7-a21c-a00fff4ed8f6|images\settings_32_32_white.png
  5ce3da45-db07-42e7-a21c-a00fff4ed8f6|..\LIBS\images\Page_nav_left.png
  5ce3da45-db07-42e7-a21c-a00fff4ed8f6|..\LIBS\images\settings_32_32_white.png
  5ce3da45-db07-42e7-a21c-a00fff4ed8f6|C:\Dev\Boeing_Rnd\Software\LIBS\images\Truck_iso_rl.png
  5ce3da45-db07-42e7-a21c-a00fff4ed8f6|C:\Dev\Boeing_Rnd\Software\LIBS\images\Truck_iso_rl_inv.png
  5ce3da45-db07-42e7-a21c-a00fff4ed8f6|C:\Dev\Boeing_Rnd\Software\LIBS\images\Truck_iso_rr_inv.png
  5ce3da45-db07-42e7-a21c-a00fff4ed8f6|C:\Dev\Boeing_Rnd\Software\LIBS\images\Truck_iso_fl_inv.png
  5ce3da45-db07-42e7-a21c-a00fff4ed8f6|C:\Dev\Boeing_Rnd\Software\LIBS\images\Truck_iso_fr_inv.png
  5ce3da45-db07-42e7-a21c-a00fff4ed8f6|C:\Dev\Boeing_Rnd\Software\LIBS\images\Truck_iso_rl_inv_better.png
  5ce3da45-db07-42e7-a21c-a00fff4ed8f6|C:\Dev\Boeing_Rnd\Software\LIBS\images\Page_nav_left.png
  5ce3da45-db07-42e7-a21c-a00fff4ed8f6|C:\Dev\Boeing_Rnd\Software\LIBS\images\Page_nav_right.png
  text list System
  5ce3da45-db07-42e7-a21c-a00fff4ed8f6|images\radial_50_50.png
  5ce3da45-db07-42e7-a21c-a00fff4ed8f6|..\LIBS\images\settings_32_32_white.png
  5ce3da45-db07-42e7-a21c-a00fff4ed8f6|..\LIBS\images\Truck_iso_fl_inv.png
  5ce3da45-db07-42e7-a21c-a00fff4ed8f6|..\LIBS\images\home_32_32_white.png
  5ce3da45-db07-42e7-a21c-a00fff4ed8f6|..\LIBS\images\Hazard_31_28.png
  5ce3da45-db07-42e7-a21c-a00fff4ed8f6|C:\Dev\Boeing_Rnd\Software\LIBS\images\net_switch.png
  5ce3da45-db07-42e7-a21c-a00fff4ed8f6|..\LIBS\images\home_32_32_white.png
  5ce3da45-db07-42e7-a21c-a00fff4ed8f6|C:\Dev\Boeing_Rnd\Software\LIBS\images\scissor_B_170_125.png
  5ce3da45-db07-42e7-a21c-a00fff4ed8f6|C:\Dev\Boeing_Rnd\Software\LIBS\images\net_cr721s.png
  splash
  5ce3da45-db07-42e7-a21c-a00fff4ed8f6|C:\Dev\Boeing_Rnd\Software\LIBS\images\net_cr0709.png
  5ce3da45-db07-42e7-a21c-a00fff4ed8f6|C:\Dev\Boeing_Rnd\Software\LIBS\images\net_o3m.png
  Project Information/
    function GetCompany [ST]
    function GetTitle [ST]
    function GetVersion [ST]
    function GetTextProperty [ST]
    function GetTextProperty2 [ST]
    function GetNumberProperty [ST]
    function GetBooleanProperty [ST]
    function GetVersionProperty [ST]
  5ce3da45-db07-42e7-a21c-a00fff4ed8f6|C:\Dev\Boeing_CT6000\Software\LIBS\images\circle.png
  5ce3da45-db07-42e7-a21c-a00fff4ed8f6|C:\Dev\Boeing_Rnd\Software\LIBS\images\main_truck_613_404.png
  5ce3da45-db07-42e7-a21c-a00fff4ed8f6|..\LIBS\images\settings_32_32_white.png
  5ce3da45-db07-42e7-a21c-a00fff4ed8f6|..\LIBS\images\settings_32_32_white.png
  5ce3da45-db07-42e7-a21c-a00fff4ed8f6|C:\Dev\Boeing_Rnd\Software\LIBS\images\main_truck_400_264.png
  5ce3da45-db07-42e7-a21c-a00fff4ed8f6|C:\Dev\Boeing_Rnd\Software\LIBS\images\scissor_A_170_125.png
  5ce3da45-db07-42e7-a21c-a00fff4ed8f6|C:\Dev\Boeing_Rnd\Software\LIBS\images\net_cr1140.png
  5ce3da45-db07-42e7-a21c-a00fff4ed8f6|C:\Dev\Boeing_Rnd\Software\LIBS\images\settings_32_32_green.png
  5ce3da45-db07-42e7-a21c-a00fff4ed8f6|C:\Dev\Boeing_Rnd\Software\LIBS\images\main_cabin.png
  5ce3da45-db07-42e7-a21c-a00fff4ed8f6|C:\Dev\Boeing_Rnd\Software\LIBS\images\main_cabin_platform_out.png
  5ce3da45-db07-42e7-a21c-a00fff4ed8f6|C:\Dev\Boeing_Rnd\Software\LIBS\images\main_cabin_platform_in.png
  5ce3da45-db07-42e7-a21c-a00fff4ed8f6|..\LIBS\images\warning_28_28.png
  5ce3da45-db07-42e7-a21c-a00fff4ed8f6|C:\Users\adam.watson\Downloads\Codesys_Logo.svg
  5ce3da45-db07-42e7-a21c-a00fff4ed8f6|..\LIBS\images\website.bmp
  5ce3da45-db07-42e7-a21c-a00fff4ed8f6|C:\Dev\Boeing_CT6000\Software\LIBS\images\Header_Beacon.png
  5ce3da45-db07-42e7-a21c-a00fff4ed8f6|C:\Dev\Boeing_CT6000\Software\LIBS\images\Header_Siren.png
  5ce3da45-db07-42e7-a21c-a00fff4ed8f6|C:\Dev\CT6000_Flex_MAIN\Software\LIBS\images\home_32_32_green.png
  00000000-0000-0000-0000-000000000000|D:\dev_plc\SLL\SLL_Truck_Demo\DASH_CR1140_HMI\splash.png
  5ce3da45-db07-42e7-a21c-a00fff4ed8f6|C:\Dev\Boeing_CT6000\Software\LIBS\images\red-cross.png
  5ce3da45-db07-42e7-a21c-a00fff4ed8f6|..\LIBS\images\Page_nav_left.png
  5ce3da45-db07-42e7-a21c-a00fff4ed8f6|..\LIBS\images\Truck_iso_fr_inv.png
  5ce3da45-db07-42e7-a21c-a00fff4ed8f6|..\LIBS\images\Truck_iso_rl_inv.png
  5ce3da45-db07-42e7-a21c-a00fff4ed8f6|..\LIBS\images\Truck_iso_rl_inv_better.png
  5ce3da45-db07-42e7-a21c-a00fff4ed8f6|..\LIBS\images\Truck_iso_rr_inv.png
  5ce3da45-db07-42e7-a21c-a00fff4ed8f6|..\LIBS\images\Page_nav_left.png
  5ce3da45-db07-42e7-a21c-a00fff4ed8f6|..\LIBS\images\Page_nav_right.png
  5ce3da45-db07-42e7-a21c-a00fff4ed8f6|..\LIBS\images\Hazard_31_28.png
  5ce3da45-db07-42e7-a21c-a00fff4ed8f6|..\LIBS\images\warning_28_28.png
  5ce3da45-db07-42e7-a21c-a00fff4ed8f6|..\LIBS\images\CAS Demo.png
  5ce3da45-db07-42e7-a21c-a00fff4ed8f6|..\LIBS\images\CAS Demo2.png
  5ce3da45-db07-42e7-a21c-a00fff4ed8f6|..\LIBS\images\website.bmp
  5ce3da45-db07-42e7-a21c-a00fff4ed8f6|C:\Dev\Boeing_Rnd\Software\LIBS\images\net_cr0709.png
  5ce3da45-db07-42e7-a21c-a00fff4ed8f6|C:\Dev\Boeing_Rnd\Software\LIBS\images\net_cr721s.png
  5ce3da45-db07-42e7-a21c-a00fff4ed8f6|C:\Dev\Boeing_Rnd\Software\LIBS\images\net_o3m.png
  5ce3da45-db07-42e7-a21c-a00fff4ed8f6|C:\Dev\Boeing_Rnd\Software\LIBS\images\net_switch.png
  5ce3da45-db07-42e7-a21c-a00fff4ed8f6|C:\Dev\Boeing_Rnd\Software\LIBS\images\net_cr1140.png
  5ce3da45-db07-42e7-a21c-a00fff4ed8f6|C:\Dev\Boeing_Rnd\Software\LIBS\images\settings_32_32_green.png
  5ce3da45-db07-42e7-a21c-a00fff4ed8f6|C:\Dev\Boeing_Rnd\Software\LIBS\images\main_truck.png
  5ce3da45-db07-42e7-a21c-a00fff4ed8f6|C:\Dev\Boeing_Rnd\Software\LIBS\images\scissor_A_208_15.png
  5ce3da45-db07-42e7-a21c-a00fff4ed8f6|C:\Dev\Boeing_Rnd\Software\LIBS\images\scissor_B_208_15.png
  5ce3da45-db07-42e7-a21c-a00fff4ed8f6|C:\Dev\Boeing_Rnd\Software\LIBS\images\power_ac.png
  5ce3da45-db07-42e7-a21c-a00fff4ed8f6|C:\Dev\Boeing_Rnd\Software\LIBS\images\power_dc.png
  5ce3da45-db07-42e7-a21c-a00fff4ed8f6|C:\Dev\Boeing_Rnd\Software\LIBS\images\power_pto.png
  5ce3da45-db07-42e7-a21c-a00fff4ed8f6|C:\Users\adam.watson\Downloads\Codesys_Logo.svg
  5ce3da45-db07-42e7-a21c-a00fff4ed8f6|C:\Dev\Boeing_Rnd\Software\LIBS\images\CAS_Red_Arrow_Down.png
  5ce3da45-db07-42e7-a21c-a00fff4ed8f6|C:\Dev\Boeing_Rnd\Software\LIBS\images\CAS_Red_Arrow_Up.png
  5ce3da45-db07-42e7-a21c-a00fff4ed8f6|C:\Dev\Boeing_Rnd\Software\LIBS\images\CAS_Red_Circle.png
  5ce3da45-db07-42e7-a21c-a00fff4ed8f6|C:\Dev\Boeing_Rnd\Software\LIBS\images\CAS_Red_Square.png
  5ce3da45-db07-42e7-a21c-a00fff4ed8f6|C:\Dev\Boeing_Rnd\Software\LIBS\images\CAS_Error.png
  5ce3da45-db07-42e7-a21c-a00fff4ed8f6|C:\Dev\Boeing_Rnd\Software\LIBS\images\CAS_Hazard.png
  5ce3da45-db07-42e7-a21c-a00fff4ed8f6|C:\Dev\Boeing_Rnd\Software\LIBS\images\CAS_Key.png
  5ce3da45-db07-42e7-a21c-a00fff4ed8f6|C:\Dev\Boeing_Rnd\Software\LIBS\images\CAS_LockOut.png
  5ce3da45-db07-42e7-a21c-a00fff4ed8f6|C:\Dev\Boeing_Rnd\Software\LIBS\images\CAS_Snail.png
  5ce3da45-db07-42e7-a21c-a00fff4ed8f6|C:\Dev\Boeing_Rnd\Software\LIBS\images\CAS_Buzzer.png
  5ce3da45-db07-42e7-a21c-a00fff4ed8f6|C:\Dev\Boeing_Rnd\Software\LIBS\images\CAS_Buzzer_Black.png
  5ce3da45-db07-42e7-a21c-a00fff4ed8f6|C:\Dev\Boeing_CT6000\Software\LIBS\images\Header_Beacon.png
  5ce3da45-db07-42e7-a21c-a00fff4ed8f6|C:\Dev\Boeing_CT6000\Software\LIBS\images\Header_Siren.png
  5ce3da45-db07-42e7-a21c-a00fff4ed8f6|C:\Dev\Boeing_CT6000\Software\LIBS\images\red-cross.png
  5ce3da45-db07-42e7-a21c-a00fff4ed8f6|C:\Dev\Boeing_CT6000\Software\LIBS\images\main_cabin_platform_only.png
  5ce3da45-db07-42e7-a21c-a00fff4ed8f6|C:\Dev\Boeing_CT6000\Software\LIBS\images\main_cabin_no_platform.png
  5ce3da45-db07-42e7-a21c-a00fff4ed8f6|C:\Dev\Boeing_CT6000\Software\LIBS\images\circle.png
  5ce3da45-db07-42e7-a21c-a00fff4ed8f6|C:\Dev\Boeing_CT6000\Software\LIBS\images\circle_34_32.png
  5ce3da45-db07-42e7-a21c-a00fff4ed8f6|C:\Dev\Boeing_CT6000\Software\LIBS\images\main_pump_running_ok.png
  5ce3da45-db07-42e7-a21c-a00fff4ed8f6|C:\Dev\Boeing_CT6000\Software\LIBS\images\mains_phases_ok.png
  5ce3da45-db07-42e7-a21c-a00fff4ed8f6|C:\Dev\Boeing_CT6000\Software\LIBS\images\ac_mains_lead_ok.png
  5ce3da45-db07-42e7-a21c-a00fff4ed8f6|C:\Dev\Boeing_CT6000\Software\LIBS\images\power_pto_engine_green.png
  5ce3da45-db07-42e7-a21c-a00fff4ed8f6|C:\Dev\Boeing_CT6000\Software\LIBS\images\power_dc_green.png
  5ce3da45-db07-42e7-a21c-a00fff4ed8f6|..\LIBS\images\settings_32_32_white.png
  5ce3da45-db07-42e7-a21c-a00fff4ed8f6|..\LIBS\images\home_32_32_white.png
  5ce3da45-db07-42e7-a21c-a00fff4ed8f6|..\LIBS\images\Truck_iso_fl_inv.png
  5ce3da45-db07-42e7-a21c-a00fff4ed8f6|..\LIBS\images\Truck_iso_fr_inv.png
  5ce3da45-db07-42e7-a21c-a00fff4ed8f6|..\LIBS\images\Truck_iso_rl_inv.png
  5ce3da45-db07-42e7-a21c-a00fff4ed8f6|..\LIBS\images\Truck_iso_rl_inv_better.png
  5ce3da45-db07-42e7-a21c-a00fff4ed8f6|..\LIBS\images\Truck_iso_rr_inv.png
  5ce3da45-db07-42e7-a21c-a00fff4ed8f6|..\LIBS\images\Page_nav_left.png
  5ce3da45-db07-42e7-a21c-a00fff4ed8f6|..\LIBS\images\Page_nav_right.png
  5ce3da45-db07-42e7-a21c-a00fff4ed8f6|..\LIBS\images\Hazard_31_28.png
  5ce3da45-db07-42e7-a21c-a00fff4ed8f6|..\LIBS\images\warning_28_28.png
  5ce3da45-db07-42e7-a21c-a00fff4ed8f6|..\LIBS\images\CAS Demo.png
  5ce3da45-db07-42e7-a21c-a00fff4ed8f6|..\LIBS\images\CAS Demo2.png
  5ce3da45-db07-42e7-a21c-a00fff4ed8f6|..\LIBS\images\website.bmp
  5ce3da45-db07-42e7-a21c-a00fff4ed8f6|C:\Dev\Boeing_Rnd\Software\LIBS\images\net_cr0709.png
  5ce3da45-db07-42e7-a21c-a00fff4ed8f6|C:\Dev\Boeing_Rnd\Software\LIBS\images\net_cr721s.png
  5ce3da45-db07-42e7-a21c-a00fff4ed8f6|C:\Dev\Boeing_Rnd\Software\LIBS\images\net_o3m.png
  5ce3da45-db07-42e7-a21c-a00fff4ed8f6|C:\Dev\Boeing_Rnd\Software\LIBS\images\net_switch.png
  5ce3da45-db07-42e7-a21c-a00fff4ed8f6|C:\Dev\Boeing_Rnd\Software\LIBS\images\net_cr1140.png
  5ce3da45-db07-42e7-a21c-a00fff4ed8f6|C:\Dev\Boeing_Rnd\Software\LIBS\images\settings_32_32_green.png
  5ce3da45-db07-42e7-a21c-a00fff4ed8f6|C:\Dev\Boeing_Rnd\Software\LIBS\images\main_truck.png
  5ce3da45-db07-42e7-a21c-a00fff4ed8f6|C:\Dev\Boeing_Rnd\Software\LIBS\images\scissor_A_208_15.png
  5ce3da45-db07-42e7-a21c-a00fff4ed8f6|C:\Dev\Boeing_Rnd\Software\LIBS\images\scissor_B_208_15.png
  5ce3da45-db07-42e7-a21c-a00fff4ed8f6|C:\Dev\Boeing_Rnd\Software\LIBS\images\power_ac.png
  5ce3da45-db07-42e7-a21c-a00fff4ed8f6|C:\Dev\Boeing_Rnd\Software\LIBS\images\power_dc.png
  5ce3da45-db07-42e7-a21c-a00fff4ed8f6|C:\Dev\Boeing_Rnd\Software\LIBS\images\power_pto.png
  5ce3da45-db07-42e7-a21c-a00fff4ed8f6|C:\Users\adam.watson\Downloads\Codesys_Logo.svg
  5ce3da45-db07-42e7-a21c-a00fff4ed8f6|C:\Dev\Boeing_Rnd\Software\LIBS\images\CAS_Red_Arrow_Down.png
  5ce3da45-db07-42e7-a21c-a00fff4ed8f6|C:\Dev\Boeing_Rnd\Software\LIBS\images\CAS_Red_Arrow_Up.png
  5ce3da45-db07-42e7-a21c-a00fff4ed8f6|C:\Dev\Boeing_Rnd\Software\LIBS\images\CAS_Red_Circle.png
  5ce3da45-db07-42e7-a21c-a00fff4ed8f6|C:\Dev\Boeing_Rnd\Software\LIBS\images\CAS_Red_Square.png
  5ce3da45-db07-42e7-a21c-a00fff4ed8f6|C:\Dev\Boeing_Rnd\Software\LIBS\images\CAS_Error.png
  5ce3da45-db07-42e7-a21c-a00fff4ed8f6|C:\Dev\Boeing_Rnd\Software\LIBS\images\CAS_Hazard.png
  5ce3da45-db07-42e7-a21c-a00fff4ed8f6|C:\Dev\Boeing_Rnd\Software\LIBS\images\CAS_Key.png
  5ce3da45-db07-42e7-a21c-a00fff4ed8f6|C:\Dev\Boeing_Rnd\Software\LIBS\images\CAS_LockOut.png
  5ce3da45-db07-42e7-a21c-a00fff4ed8f6|C:\Dev\Boeing_Rnd\Software\LIBS\images\CAS_Snail.png
  5ce3da45-db07-42e7-a21c-a00fff4ed8f6|C:\Dev\Boeing_Rnd\Software\LIBS\images\CAS_Tortoise.png
  5ce3da45-db07-42e7-a21c-a00fff4ed8f6|C:\Dev\Boeing_Rnd\Software\LIBS\images\CAS_Buzzer.png
  5ce3da45-db07-42e7-a21c-a00fff4ed8f6|C:\Dev\Boeing_Rnd\Software\LIBS\images\CAS_Buzzer_Black.png
  5ce3da45-db07-42e7-a21c-a00fff4ed8f6|C:\Dev\Boeing_CT6000\Software\LIBS\images\Header_Beacon.png
  5ce3da45-db07-42e7-a21c-a00fff4ed8f6|C:\Dev\Boeing_CT6000\Software\LIBS\images\Header_Siren.png
  5ce3da45-db07-42e7-a21c-a00fff4ed8f6|C:\Dev\Boeing_CT6000\Software\LIBS\images\red-cross.png
  5ce3da45-db07-42e7-a21c-a00fff4ed8f6|C:\Dev\Boeing_CT6000\Software\LIBS\images\main_cabin_platform_only.png
  5ce3da45-db07-42e7-a21c-a00fff4ed8f6|C:\Dev\Boeing_CT6000\Software\LIBS\images\main_cabin_no_platform.png
  5ce3da45-db07-42e7-a21c-a00fff4ed8f6|C:\Dev\Boeing_CT6000\Software\LIBS\images\circle.png
  5ce3da45-db07-42e7-a21c-a00fff4ed8f6|C:\Dev\Boeing_CT6000\Software\LIBS\images\circle_34_32.png
  5ce3da45-db07-42e7-a21c-a00fff4ed8f6|C:\Dev\Boeing_CT6000\Software\LIBS\images\main_pump_running_ok.png
  5ce3da45-db07-42e7-a21c-a00fff4ed8f6|C:\Dev\Boeing_CT6000\Software\LIBS\images\mains_phases_ok.png
  5ce3da45-db07-42e7-a21c-a00fff4ed8f6|C:\Dev\Boeing_CT6000\Software\LIBS\images\ac_mains_lead_ok.png
  5ce3da45-db07-42e7-a21c-a00fff4ed8f6|C:\Dev\Boeing_CT6000\Software\LIBS\images\power_pto_engine_green.png
  5ce3da45-db07-42e7-a21c-a00fff4ed8f6|C:\Dev\Boeing_CT6000\Software\LIBS\images\power_dc_green.png
  5ce3da45-db07-42e7-a21c-a00fff4ed8f6|..\LIBS\images\home_32_32_white.png
  5ce3da45-db07-42e7-a21c-a00fff4ed8f6|..\LIBS\images\Truck_iso_fl_inv.png
  5ce3da45-db07-42e7-a21c-a00fff4ed8f6|..\LIBS\images\Truck_iso_fr_inv.png
  5ce3da45-db07-42e7-a21c-a00fff4ed8f6|..\LIBS\images\Truck_iso_rl_inv.png
  5ce3da45-db07-42e7-a21c-a00fff4ed8f6|..\LIBS\images\Truck_iso_rl_inv_better.png
  5ce3da45-db07-42e7-a21c-a00fff4ed8f6|..\LIBS\images\Truck_iso_rr_inv.png
  5ce3da45-db07-42e7-a21c-a00fff4ed8f6|..\LIBS\images\Page_nav_left.png
  5ce3da45-db07-42e7-a21c-a00fff4ed8f6|..\LIBS\images\Page_nav_right.png
  5ce3da45-db07-42e7-a21c-a00fff4ed8f6|..\LIBS\images\Hazard_31_28.png
  5ce3da45-db07-42e7-a21c-a00fff4ed8f6|..\LIBS\images\warning_28_28.png
  5ce3da45-db07-42e7-a21c-a00fff4ed8f6|..\LIBS\images\CAS Demo.png
  5ce3da45-db07-42e7-a21c-a00fff4ed8f6|..\LIBS\images\CAS Demo2.png
  5ce3da45-db07-42e7-a21c-a00fff4ed8f6|..\LIBS\images\website.bmp
  5ce3da45-db07-42e7-a21c-a00fff4ed8f6|C:\Dev\Boeing_Rnd\Software\LIBS\images\net_cr0709.png
  5ce3da45-db07-42e7-a21c-a00fff4ed8f6|C:\Dev\Boeing_Rnd\Software\LIBS\images\net_cr721s.png
  5ce3da45-db07-42e7-a21c-a00fff4ed8f6|C:\Dev\Boeing_Rnd\Software\LIBS\images\net_o3m.png
  5ce3da45-db07-42e7-a21c-a00fff4ed8f6|C:\Dev\Boeing_Rnd\Software\LIBS\images\net_switch.png
  5ce3da45-db07-42e7-a21c-a00fff4ed8f6|C:\Dev\Boeing_Rnd\Software\LIBS\images\net_cr1140.png
  5ce3da45-db07-42e7-a21c-a00fff4ed8f6|C:\Dev\Boeing_Rnd\Software\LIBS\images\settings_32_32_green.png
  5ce3da45-db07-42e7-a21c-a00fff4ed8f6|C:\Dev\Boeing_Rnd\Software\LIBS\images\main_truck.png
  5ce3da45-db07-42e7-a21c-a00fff4ed8f6|C:\Dev\Boeing_Rnd\Software\LIBS\images\scissor_A_208_15.png
  5ce3da45-db07-42e7-a21c-a00fff4ed8f6|C:\Dev\Boeing_Rnd\Software\LIBS\images\scissor_B_208_15.png
  5ce3da45-db07-42e7-a21c-a00fff4ed8f6|C:\Dev\Boeing_Rnd\Software\LIBS\images\power_ac.png
  5ce3da45-db07-42e7-a21c-a00fff4ed8f6|C:\Dev\Boeing_Rnd\Software\LIBS\images\power_dc.png
  5ce3da45-db07-42e7-a21c-a00fff4ed8f6|C:\Dev\Boeing_Rnd\Software\LIBS\images\power_pto.png
  5ce3da45-db07-42e7-a21c-a00fff4ed8f6|C:\Users\adam.watson\Downloads\Codesys_Logo.svg
  5ce3da45-db07-42e7-a21c-a00fff4ed8f6|C:\Dev\Boeing_Rnd\Software\LIBS\images\CAS_Red_Arrow_Down.png
  5ce3da45-db07-42e7-a21c-a00fff4ed8f6|C:\Dev\Boeing_Rnd\Software\LIBS\images\CAS_Red_Arrow_Up.png
  5ce3da45-db07-42e7-a21c-a00fff4ed8f6|C:\Dev\Boeing_Rnd\Software\LIBS\images\CAS_Red_Circle.png
  5ce3da45-db07-42e7-a21c-a00fff4ed8f6|C:\Dev\Boeing_Rnd\Software\LIBS\images\CAS_Red_Square.png
  5ce3da45-db07-42e7-a21c-a00fff4ed8f6|C:\Dev\Boeing_Rnd\Software\LIBS\images\CAS_Error.png
  5ce3da45-db07-42e7-a21c-a00fff4ed8f6|C:\Dev\Boeing_Rnd\Software\LIBS\images\CAS_Hazard.png
  5ce3da45-db07-42e7-a21c-a00fff4ed8f6|C:\Dev\Boeing_Rnd\Software\LIBS\images\CAS_Key.png
  5ce3da45-db07-42e7-a21c-a00fff4ed8f6|C:\Dev\Boeing_Rnd\Software\LIBS\images\CAS_LockOut.png
  5ce3da45-db07-42e7-a21c-a00fff4ed8f6|C:\Dev\Boeing_Rnd\Software\LIBS\images\CAS_Snail.png
  5ce3da45-db07-42e7-a21c-a00fff4ed8f6|C:\Dev\Boeing_Rnd\Software\LIBS\images\CAS_Tortoise.png
  5ce3da45-db07-42e7-a21c-a00fff4ed8f6|C:\Dev\Boeing_Rnd\Software\LIBS\images\CAS_Buzzer.png
  5ce3da45-db07-42e7-a21c-a00fff4ed8f6|C:\Dev\Boeing_Rnd\Software\LIBS\images\CAS_Buzzer_Black.png
  5ce3da45-db07-42e7-a21c-a00fff4ed8f6|C:\Dev\Boeing_CT6000\Software\LIBS\images\Header_Beacon.png
  5ce3da45-db07-42e7-a21c-a00fff4ed8f6|C:\Dev\Boeing_CT6000\Software\LIBS\images\Header_Siren.png
  5ce3da45-db07-42e7-a21c-a00fff4ed8f6|C:\Dev\Boeing_CT6000\Software\LIBS\images\red-cross.png
  5ce3da45-db07-42e7-a21c-a00fff4ed8f6|C:\Dev\Boeing_CT6000\Software\LIBS\images\main_cabin_platform_only.png
  5ce3da45-db07-42e7-a21c-a00fff4ed8f6|C:\Dev\Boeing_CT6000\Software\LIBS\images\main_cabin_no_platform.png
  5ce3da45-db07-42e7-a21c-a00fff4ed8f6|C:\Dev\Boeing_CT6000\Software\LIBS\images\circle.png
  5ce3da45-db07-42e7-a21c-a00fff4ed8f6|C:\Dev\Boeing_CT6000\Software\LIBS\images\circle_34_32.png
  5ce3da45-db07-42e7-a21c-a00fff4ed8f6|C:\Dev\Boeing_CT6000\Software\LIBS\images\main_pump_running_ok.png
  5ce3da45-db07-42e7-a21c-a00fff4ed8f6|C:\Dev\Boeing_CT6000\Software\LIBS\images\mains_phases_ok.png
  5ce3da45-db07-42e7-a21c-a00fff4ed8f6|C:\Dev\Boeing_CT6000\Software\LIBS\images\ac_mains_lead_ok.png
  5ce3da45-db07-42e7-a21c-a00fff4ed8f6|C:\Dev\Boeing_CT6000\Software\LIBS\images\power_pto_engine_green.png
  5ce3da45-db07-42e7-a21c-a00fff4ed8f6|C:\Dev\Boeing_CT6000\Software\LIBS\images\power_dc_green.png
  5ce3da45-db07-42e7-a21c-a00fff4ed8f6|..\LIBS\images\Page_nav_right.png
  5ce3da45-db07-42e7-a21c-a00fff4ed8f6|..\LIBS\images\Hazard_31_28.png
  5ce3da45-db07-42e7-a21c-a00fff4ed8f6|images\Track_50_50.png
  5ce3da45-db07-42e7-a21c-a00fff4ed8f6|C:\Dev\Boeing_CT6000\Software\LIBS\images\Hazard_31_28_dull.png
  5ce3da45-db07-42e7-a21c-a00fff4ed8f6|C:\Dev\CT6000_Flex_Compare\Software\LIBS\images\hydraulic_oil_0_0.png
  5ce3da45-db07-42e7-a21c-a00fff4ed8f6|C:\Dev\CT6000_Flex_Compare\Software\LIBS\images\hydraulic_oil_0_1.png
  5ce3da45-db07-42e7-a21c-a00fff4ed8f6|C:\Users\indongpa\Downloads\Visu_Global_BG_ecomatDisplay43Inch_V1\Visu_Global_BG_WithKeys_ecomatDisplay43Inch.png
  5ce3da45-db07-42e7-a21c-a00fff4ed8f6|\\DESKTOP-U06DLQD\Projects\Project Bitmaps\2024_Images\batteryREDonBlack60pixel.png
  5ce3da45-db07-42e7-a21c-a00fff4ed8f6|\\DESKTOP-U06DLQD\Projects\Project Bitmaps\2024_Images\HOL60pixel.png
  5ce3da45-db07-42e7-a21c-a00fff4ed8f6|\\DESKTOP-U06DLQD\Projects\Project Bitmaps\2024_Images\HydOilTemp60pixel.png
  5ce3da45-db07-42e7-a21c-a00fff4ed8f6|\\DESKTOP-U06DLQD\Projects\Project Bitmaps\2024_Images\temperatureREDonBlack60pixel.png
  5ce3da45-db07-42e7-a21c-a00fff4ed8f6|\\DESKTOP-U06DLQD\Projects\Project Bitmaps\2024_Images\OilCanREDonBlack60pixel.png
  5ce3da45-db07-42e7-a21c-a00fff4ed8f6|\\DESKTOP-U06DLQD\Projects\Project Bitmaps\2024_Images\EmmStop60pixel.png
  5ce3da45-db07-42e7-a21c-a00fff4ed8f6|\\DESKTOP-U06DLQD\Projects\Project Bitmaps\2024_Images\DPF Icon 60pixel.png
  5ce3da45-db07-42e7-a21c-a00fff4ed8f6|\\DESKTOP-U06DLQD\Projects\Project Bitmaps\2024_Images\DPF Disabled Lamp60pixel.png
  5ce3da45-db07-42e7-a21c-a00fff4ed8f6|\\DESKTOP-U06DLQD\Projects\Project Bitmaps\2024_Images\Dpf Regen Active60pixel.png
  5ce3da45-db07-42e7-a21c-a00fff4ed8f6|\\DESKTOP-U06DLQD\Projects\Project Bitmaps\2024_Images\DPF Icon2_60pixel.png
  5ce3da45-db07-42e7-a21c-a00fff4ed8f6|\\DESKTOP-U06DLQD\Projects\Project Bitmaps\Stop 60x60.bmp
  5ce3da45-db07-42e7-a21c-a00fff4ed8f6|\\DESKTOP-U06DLQD\Projects\Project Bitmaps\2024_Images\Engine IconAmber60pixel.png
  5ce3da45-db07-42e7-a21c-a00fff4ed8f6|\\DESKTOP-U06DLQD\Projects\Project Bitmaps\2024_Images\Engine IconRed60pixel.png
  5ce3da45-db07-42e7-a21c-a00fff4ed8f6|\\DESKTOP-U06DLQD\Projects\Project Bitmaps\2024_Images\Right Arrow Simple 30 pixel wide.png
  5ce3da45-db07-42e7-a21c-a00fff4ed8f6|\\DESKTOP-U06DLQD\Projects\Project Bitmaps\2024_Images\Right Arrow Simple Green 30pixel.png
  5ce3da45-db07-42e7-a21c-a00fff4ed8f6|\\DESKTOP-U06DLQD\Projects\Project Bitmaps\2024_Images\Rotating Arrow30pixel.png
  5ce3da45-db07-42e7-a21c-a00fff4ed8f6|\\DESKTOP-U06DLQD\Projects\Project Bitmaps\2024_Images\Engine Icon90pixel.png
  5ce3da45-db07-42e7-a21c-a00fff4ed8f6|C:\Project Briefcase\Project Bitmaps\Petrol Pump60pixel.png
  5ce3da45-db07-42e7-a21c-a00fff4ed8f6|C:\Project Briefcase\Project Bitmaps\Petrol PumpRed60pixel.png
  5ce3da45-db07-42e7-a21c-a00fff4ed8f6|\\DESKTOP-U06DLQD\Projects\Project Bitmaps\2024_Images\arrow2_60pixel.png
  5ce3da45-db07-42e7-a21c-a00fff4ed8f6|\\DESKTOP-U06DLQD\Projects\Project Bitmaps\2024_Images\arrow60pixel.png
  5ce3da45-db07-42e7-a21c-a00fff4ed8f6|\\DESKTOP-U06DLQD\Projects\Project Bitmaps\2024_Images\start50pixel.png
  5ce3da45-db07-42e7-a21c-a00fff4ed8f6|\\DESKTOP-U06DLQD\Projects\Project Bitmaps\2024_Images\EngineInfo_7inch.png
  5ce3da45-db07-42e7-a21c-a00fff4ed8f6|\\DESKTOP-U06DLQD\Projects\Project Bitmaps\2024_Images\ArrowLeft50pixel.png
  5ce3da45-db07-42e7-a21c-a00fff4ed8f6|\\DESKTOP-U06DLQD\Projects\Project Bitmaps\2024_Images\ArrowRight50pixel.png
  5ce3da45-db07-42e7-a21c-a00fff4ed8f6|\\DESKTOP-U06DLQD\Projects\Project Bitmaps\2024_Images\DPF Man Regen 50 pixelhigh.png
  5ce3da45-db07-42e7-a21c-a00fff4ed8f6|\\DESKTOP-U06DLQD\Projects\Project Bitmaps\2024_Images\Hand50pixel.png
  5ce3da45-db07-42e7-a21c-a00fff4ed8f6|\\DESKTOP-U06DLQD\Projects\Project Bitmaps\2024_Images\LeverValve50pixel.png
  5ce3da45-db07-42e7-a21c-a00fff4ed8f6|\\DESKTOP-U06DLQD\Projects\Project Bitmaps\2024_Images\speedometer50pixel.png
  5ce3da45-db07-42e7-a21c-a00fff4ed8f6|\\DESKTOP-U06DLQD\Projects\Project Bitmaps\2024_Images\Engine Icon50pixel.png
  5ce3da45-db07-42e7-a21c-a00fff4ed8f6|\\DESKTOP-U06DLQD\Projects\Project Bitmaps\2024_Images\Maintenance50pixel.png
  5ce3da45-db07-42e7-a21c-a00fff4ed8f6|\\DESKTOP-U06DLQD\Projects\Project Bitmaps\2024_Images\AdBlue Icon On Black60pixel.png
  5ce3da45-db07-42e7-a21c-a00fff4ed8f6|\\DESKTOP-U06DLQD\Projects\Project Bitmaps\2024_Images\Stop Button50pixel.png
  5ce3da45-db07-42e7-a21c-a00fff4ed8f6|\\DESKTOP-U06DLQD\Projects\Project Bitmaps\2024_Images\padlock_JPG.jpg
  5ce3da45-db07-42e7-a21c-a00fff4ed8f6|\\DESKTOP-U06DLQD\Projects\Project Bitmaps\2024_Images\padlockOpen_JPG.jpg
  5ce3da45-db07-42e7-a21c-a00fff4ed8f6|\\DESKTOP-U06DLQD\Projects\Project Bitmaps\HydOil Warning 60 pixel.bmp
  5ce3da45-db07-42e7-a21c-a00fff4ed8f6|\\DESKTOP-U06DLQD\Projects\Project Bitmaps\2024_Images\mtech_800480.jpg
  5ce3da45-db07-42e7-a21c-a00fff4ed8f6|C:\Dev\Boeing_Rnd\Software\LIBS\images\net_cr0709.png
  5ce3da45-db07-42e7-a21c-a00fff4ed8f6|images\engine_hours.png
  5ce3da45-db07-42e7-a21c-a00fff4ed8f6|images\Battery.png
  5ce3da45-db07-42e7-a21c-a00fff4ed8f6|images\engine_temp.png
  5ce3da45-db07-42e7-a21c-a00fff4ed8f6|images\oil.png
  5ce3da45-db07-42e7-a21c-a00fff4ed8f6|C:\Dev\Boeing_Rnd\Software\LIBS\images\net_cr721s.png
  5ce3da45-db07-42e7-a21c-a00fff4ed8f6|C:\Dev\Boeing_Rnd\Software\LIBS\images\net_o3m.png
  5ce3da45-db07-42e7-a21c-a00fff4ed8f6|C:\Dev\Boeing_Rnd\Software\LIBS\images\net_switch.png
  5ce3da45-db07-42e7-a21c-a00fff4ed8f6|C:\Dev\Boeing_Rnd\Software\LIBS\images\net_cr1140.png
  5ce3da45-db07-42e7-a21c-a00fff4ed8f6|C:\Dev\Boeing_Rnd\Software\LIBS\images\settings_32_32_green.png
  5ce3da45-db07-42e7-a21c-a00fff4ed8f6|C:\Users\adam.watson\Downloads\Codesys_Logo.svg
  5ce3da45-db07-42e7-a21c-a00fff4ed8f6|C:\Dev\Boeing_CT6000\Software\LIBS\images\Header_Beacon.png
  5ce3da45-db07-42e7-a21c-a00fff4ed8f6|C:\Dev\Boeing_CT6000\Software\LIBS\images\Header_Siren.png
  5ce3da45-db07-42e7-a21c-a00fff4ed8f6|C:\Dev\Boeing_CT6000\Software\LIBS\images\red-cross.png
  5ce3da45-db07-42e7-a21c-a00fff4ed8f6|C:\Dev\Boeing_CT6000\Software\LIBS\images\circle.png
  5ce3da45-db07-42e7-a21c-a00fff4ed8f6|C:\Dev\Boeing_CT6000\Software\LIBS\images\circle_34_32.png
  5ce3da45-db07-42e7-a21c-a00fff4ed8f6|C:\Dev\Boeing_CT6000\Software\LIBS\images\warning_28_28_dull.png
  5ce3da45-db07-42e7-a21c-a00fff4ed8f6|C:\Dev\Boeing_CT6000\Software\LIBS\images\Hazard_31_28_dull.png
  5ce3da45-db07-42e7-a21c-a00fff4ed8f6|C:\Dev\CT6000_Flex_Compare\Software\LIBS\images\hydraulic_oil_0_0.png
  5ce3da45-db07-42e7-a21c-a00fff4ed8f6|C:\Dev\CT6000_Flex_Compare\Software\LIBS\images\hydraulic_oil_0_1.png
  5ce3da45-db07-42e7-a21c-a00fff4ed8f6|C:\Dev\CT6000_Flex_MAIN\Software\LIBS\images\home_32_32_green.png
  5ce3da45-db07-42e7-a21c-a00fff4ed8f6|D:\dev_plc\SLL\SLL_Truck_Demo\LIBS\images\CR1076_240_200.png
  5ce3da45-db07-42e7-a21c-a00fff4ed8f6|..\LIBS\images\settings_32_32_white.png
  5ce3da45-db07-42e7-a21c-a00fff4ed8f6|..\LIBS\images\home_32_32_white.png
  5ce3da45-db07-42e7-a21c-a00fff4ed8f6|..\LIBS\images\Page_nav_left.png
  5ce3da45-db07-42e7-a21c-a00fff4ed8f6|..\LIBS\images\Page_nav_right.png
  5ce3da45-db07-42e7-a21c-a00fff4ed8f6|..\LIBS\images\Hazard_31_28.png
  5ce3da45-db07-42e7-a21c-a00fff4ed8f6|..\LIBS\images\warning_28_28.png
  5ce3da45-db07-42e7-a21c-a00fff4ed8f6|..\LIBS\images\website.bmp
  5ce3da45-db07-42e7-a21c-a00fff4ed8f6|C:\Dev\Boeing_Rnd\Software\LIBS\images\net_cr0709.png
  5ce3da45-db07-42e7-a21c-a00fff4ed8f6|C:\Dev\Boeing_Rnd\Software\LIBS\images\net_cr721s.png
  5ce3da45-db07-42e7-a21c-a00fff4ed8f6|C:\Dev\Boeing_Rnd\Software\LIBS\images\net_o3m.png
  5ce3da45-db07-42e7-a21c-a00fff4ed8f6|C:\Dev\Boeing_Rnd\Software\LIBS\images\net_switch.png
  5ce3da45-db07-42e7-a21c-a00fff4ed8f6|C:\Dev\Boeing_Rnd\Software\LIBS\images\net_cr1140.png
  5ce3da45-db07-42e7-a21c-a00fff4ed8f6|C:\Dev\Boeing_Rnd\Software\LIBS\images\settings_32_32_green.png
  5ce3da45-db07-42e7-a21c-a00fff4ed8f6|C:\Users\adam.watson\Downloads\Codesys_Logo.svg
  5ce3da45-db07-42e7-a21c-a00fff4ed8f6|C:\Dev\Boeing_CT6000\Software\LIBS\images\Header_Beacon.png
  5ce3da45-db07-42e7-a21c-a00fff4ed8f6|C:\Dev\Boeing_CT6000\Software\LIBS\images\Header_Siren.png
  5ce3da45-db07-42e7-a21c-a00fff4ed8f6|C:\Dev\Boeing_CT6000\Software\LIBS\images\red-cross.png
  5ce3da45-db07-42e7-a21c-a00fff4ed8f6|C:\Dev\Boeing_CT6000\Software\LIBS\images\circle.png
  5ce3da45-db07-42e7-a21c-a00fff4ed8f6|C:\Dev\Boeing_CT6000\Software\LIBS\images\circle_34_32.png
  5ce3da45-db07-42e7-a21c-a00fff4ed8f6|C:\Dev\Boeing_CT6000\Software\LIBS\images\warning_28_28_dull.png
  5ce3da45-db07-42e7-a21c-a00fff4ed8f6|C:\Dev\Boeing_CT6000\Software\LIBS\images\Hazard_31_28_dull.png
  5ce3da45-db07-42e7-a21c-a00fff4ed8f6|C:\Dev\CT6000_Flex_Compare\Software\LIBS\images\hydraulic_oil_0_0.png
  5ce3da45-db07-42e7-a21c-a00fff4ed8f6|C:\Dev\CT6000_Flex_Compare\Software\LIBS\images\hydraulic_oil_0_1.png
  5ce3da45-db07-42e7-a21c-a00fff4ed8f6|C:\Dev\CT6000_Flex_MAIN\Software\LIBS\images\home_32_32_green.png
  5ce3da45-db07-42e7-a21c-a00fff4ed8f6|D:\dev_plc\SLL\SLL_Truck_Demo\LIBS\images\CR1076_240_200.png
  5ce3da45-db07-42e7-a21c-a00fff4ed8f6|C:\Users\indongpa\Downloads\Visu_Global_BG_ecomatDisplay43Inch_V1\Visu_Global_BG_WithKeys_ecomatDisplay43Inch.png
  5ce3da45-db07-42e7-a21c-a00fff4ed8f6|\\DESKTOP-U06DLQD\Projects\Project Bitmaps\2024_Images\batteryREDonBlack60pixel.png
  5ce3da45-db07-42e7-a21c-a00fff4ed8f6|\\DESKTOP-U06DLQD\Projects\Project Bitmaps\2024_Images\HOL60pixel.png
  5ce3da45-db07-42e7-a21c-a00fff4ed8f6|\\DESKTOP-U06DLQD\Projects\Project Bitmaps\2024_Images\HydOilTemp60pixel.png
  5ce3da45-db07-42e7-a21c-a00fff4ed8f6|\\DESKTOP-U06DLQD\Projects\Project Bitmaps\2024_Images\temperatureREDonBlack60pixel.png
  5ce3da45-db07-42e7-a21c-a00fff4ed8f6|\\DESKTOP-U06DLQD\Projects\Project Bitmaps\2024_Images\OilCanREDonBlack60pixel.png
  5ce3da45-db07-42e7-a21c-a00fff4ed8f6|\\DESKTOP-U06DLQD\Projects\Project Bitmaps\2024_Images\EmmStop60pixel.png
  5ce3da45-db07-42e7-a21c-a00fff4ed8f6|\\DESKTOP-U06DLQD\Projects\Project Bitmaps\2024_Images\DPF Icon 60pixel.png
  5ce3da45-db07-42e7-a21c-a00fff4ed8f6|\\DESKTOP-U06DLQD\Projects\Project Bitmaps\2024_Images\DPF Disabled Lamp60pixel.png
  5ce3da45-db07-42e7-a21c-a00fff4ed8f6|\\DESKTOP-U06DLQD\Projects\Project Bitmaps\2024_Images\Dpf Regen Active60pixel.png
  5ce3da45-db07-42e7-a21c-a00fff4ed8f6|\\DESKTOP-U06DLQD\Projects\Project Bitmaps\2024_Images\DPF Icon2_60pixel.png
  5ce3da45-db07-42e7-a21c-a00fff4ed8f6|\\DESKTOP-U06DLQD\Projects\Project Bitmaps\Stop 60x60.bmp
  5ce3da45-db07-42e7-a21c-a00fff4ed8f6|\\DESKTOP-U06DLQD\Projects\Project Bitmaps\2024_Images\Engine IconAmber60pixel.png
  5ce3da45-db07-42e7-a21c-a00fff4ed8f6|\\DESKTOP-U06DLQD\Projects\Project Bitmaps\2024_Images\Engine IconRed60pixel.png
  5ce3da45-db07-42e7-a21c-a00fff4ed8f6|\\DESKTOP-U06DLQD\Projects\Project Bitmaps\2024_Images\Right Arrow Simple 30 pixel wide.png
  5ce3da45-db07-42e7-a21c-a00fff4ed8f6|\\DESKTOP-U06DLQD\Projects\Project Bitmaps\2024_Images\Right Arrow Simple Green 30pixel.png
  5ce3da45-db07-42e7-a21c-a00fff4ed8f6|\\DESKTOP-U06DLQD\Projects\Project Bitmaps\2024_Images\Rotating Arrow30pixel.png
  5ce3da45-db07-42e7-a21c-a00fff4ed8f6|\\DESKTOP-U06DLQD\Projects\Project Bitmaps\2024_Images\Engine Icon90pixel.png
  5ce3da45-db07-42e7-a21c-a00fff4ed8f6|C:\Project Briefcase\Project Bitmaps\Petrol Pump60pixel.png
  5ce3da45-db07-42e7-a21c-a00fff4ed8f6|C:\Project Briefcase\Project Bitmaps\Petrol PumpRed60pixel.png
  5ce3da45-db07-42e7-a21c-a00fff4ed8f6|\\DESKTOP-U06DLQD\Projects\MTech Solutions Ireland\297 - EzyStk TR620X Fully Auto Trommel\Technical Information\TR620X Images\TR620X Images\Trommel.png
  5ce3da45-db07-42e7-a21c-a00fff4ed8f6|\\DESKTOP-U06DLQD\Projects\Project Bitmaps\2024_Images\arrow2_60pixel.png
  5ce3da45-db07-42e7-a21c-a00fff4ed8f6|\\DESKTOP-U06DLQD\Projects\Project Bitmaps\2024_Images\arrow60pixel.png
  5ce3da45-db07-42e7-a21c-a00fff4ed8f6|\\DESKTOP-U06DLQD\Projects\Project Bitmaps\2024_Images\start50pixel.png
  5ce3da45-db07-42e7-a21c-a00fff4ed8f6|\\DESKTOP-U06DLQD\Projects\Project Bitmaps\2024_Images\EngineInfo_7inch.png
  5ce3da45-db07-42e7-a21c-a00fff4ed8f6|\\DESKTOP-U06DLQD\Projects\Project Bitmaps\2024_Images\ArrowLeft50pixel.png
  5ce3da45-db07-42e7-a21c-a00fff4ed8f6|\\DESKTOP-U06DLQD\Projects\Project Bitmaps\2024_Images\ArrowRight50pixel.png
  5ce3da45-db07-42e7-a21c-a00fff4ed8f6|\\DESKTOP-U06DLQD\Projects\Project Bitmaps\2024_Images\DPF Man Regen 50 pixelhigh.png
  5ce3da45-db07-42e7-a21c-a00fff4ed8f6|\\DESKTOP-U06DLQD\Projects\Project Bitmaps\2024_Images\Hand50pixel.png
  5ce3da45-db07-42e7-a21c-a00fff4ed8f6|\\DESKTOP-U06DLQD\Projects\Project Bitmaps\2024_Images\LeverValve50pixel.png
  5ce3da45-db07-42e7-a21c-a00fff4ed8f6|\\DESKTOP-U06DLQD\Projects\Project Bitmaps\2024_Images\speedometer50pixel.png
  5ce3da45-db07-42e7-a21c-a00fff4ed8f6|\\DESKTOP-U06DLQD\Projects\Project Bitmaps\2024_Images\Engine Icon50pixel.png
  5ce3da45-db07-42e7-a21c-a00fff4ed8f6|\\DESKTOP-U06DLQD\Projects\Project Bitmaps\2024_Images\Maintenance50pixel.png
  5ce3da45-db07-42e7-a21c-a00fff4ed8f6|\\DESKTOP-U06DLQD\Projects\Project Bitmaps\2024_Images\AdBlue Icon On Black60pixel.png
  5ce3da45-db07-42e7-a21c-a00fff4ed8f6|\\DESKTOP-U06DLQD\Projects\Project Bitmaps\2024_Images\Stop Button50pixel.png
  5ce3da45-db07-42e7-a21c-a00fff4ed8f6|\\DESKTOP-U06DLQD\Projects\Project Bitmaps\2024_Images\padlock_JPG.jpg
  5ce3da45-db07-42e7-a21c-a00fff4ed8f6|\\DESKTOP-U06DLQD\Projects\Project Bitmaps\2024_Images\padlockOpen_JPG.jpg
  5ce3da45-db07-42e7-a21c-a00fff4ed8f6|\\DESKTOP-U06DLQD\Projects\Project Bitmaps\HydOil Warning 60 pixel.bmp
  5ce3da45-db07-42e7-a21c-a00fff4ed8f6|\\DESKTOP-U06DLQD\Projects\Project Bitmaps\2024_Images\mtech_800480.jpg
  5ce3da45-db07-42e7-a21c-a00fff4ed8f6|images\engine_hours.png
  5ce3da45-db07-42e7-a21c-a00fff4ed8f6|images\Battery.png
  5ce3da45-db07-42e7-a21c-a00fff4ed8f6|images\engine_temp.png
  5ce3da45-db07-42e7-a21c-a00fff4ed8f6|images\oil.png
  5ce3da45-db07-42e7-a21c-a00fff4ed8f6|images\Nav_Down_17_18.png
  5ce3da45-db07-42e7-a21c-a00fff4ed8f6|images\Nav_Up_17_18.png
  5ce3da45-db07-42e7-a21c-a00fff4ed8f6|images\NavCircle_18_18.png
  5ce3da45-db07-42e7-a21c-a00fff4ed8f6|images\Nav_Left_17_18.png
  5ce3da45-db07-42e7-a21c-a00fff4ed8f6|images\Nav_Right_17_18.png
  visualisation Visualization
  visualisation Visualization_1
  5ce3da45-db07-42e7-a21c-a00fff4ed8f6|images\Tracks_51_15_orange.png
  5ce3da45-db07-42e7-a21c-a00fff4ed8f6|images\Tracks_51_15_white.png
  5ce3da45-db07-42e7-a21c-a00fff4ed8f6|images\clock_50_50.png
  5ce3da45-db07-42e7-a21c-a00fff4ed8f6|images\swt_50_50.png
  5ce3da45-db07-42e7-a21c-a00fff4ed8f6|images\iso_radial_720_338.png
  5ce3da45-db07-42e7-a21c-a00fff4ed8f6|images\iso_T620X_720_387.png
  5ce3da45-db07-42e7-a21c-a00fff4ed8f6|images\Green_Arrow_Left_38_24.png
  5ce3da45-db07-42e7-a21c-a00fff4ed8f6|images\Green_Arrow_Right_38_24.png
  5ce3da45-db07-42e7-a21c-a00fff4ed8f6|images\radial_left.png
  5ce3da45-db07-42e7-a21c-a00fff4ed8f6|images\radial_right.png
  5ce3da45-db07-42e7-a21c-a00fff4ed8f6|images\side_conv_down.png
  5ce3da45-db07-42e7-a21c-a00fff4ed8f6|images\side_conv_up.png
*)

// Device/Application/LIBS/HMI/HMI_TASKS_INFO_STRUCT
TYPE HMI_TASKS_INFO_STRUCT :
STRUCT
	Size: INT:=20;
	Tasks: ARRAY [0..19] OF HMI_TASK_INFO_STRUCT;
END_STRUCT
END_TYPE

// Device/Application/App_CODE_GEN/MAIN_CODE_GEN/App_CODE_GEN/Machine IO/Structs/T620X_Radial_Outputs
TYPE T620X_Radial_Outputs :
STRUCT
// Machine_IO_Outputs_STRUCT_CODE_GEN_START

// generated (UTC): 2024-07-23 18:31:25.208393+00:00

TAILCONVSPD_MA:OpCom; // CHASSIS.OUT0000
RHS_JACKLEGLOWER_OP:OpCom; // CHASSIS.OUT0001
SIDECONVSPD_MA:OpCom; // CHASSIS.OUT0002
LHS_JACKLEGRAISE_OP:OpCom; // CHASSIS.OUT0003
SIDETRANSFERSPD_MA:OpCom; // CHASSIS.OUT0004
LHS_JACKLEGLOWER_OP:OpCom; // CHASSIS.OUT0005
SETUPDUMPVALVE_OP:OpCom; // CHASSIS.OUT0006
COLLECTIONCONVSPD_MA:OpCom; // CHASSIS.OUT0007
COLLECTIONCONVON_OP:OpCom; // CHASSIS.OUT0008
SUPPLY_GROUP0:OpGrpCom; // CHASSIS.GROUP0
DRUMSPD_MA_RAMP_LIMIT:OpCom; // CHASSIS.OUT0100
TRACKINGMODE:OpCom; // CHASSIS.OUT0101
FEEDERSPD_MA:OpCom; // CHASSIS.OUT0102
CRANKENABLE:OpCom; // CHASSIS.OUT0103
DIVERTOILTOTRACK_OP:OpCom; // CHASSIS.OUT0104
RHS_JACKLEGRAISE_OP:OpCom; // CHASSIS.OUT0105
TAILCONVON_OP:OpCom; // CHASSIS.OUT0106
SIDECONVON_OP:OpCom; // CHASSIS.OUT0107
SIDETRANSFERON_OP:OpCom; // CHASSIS.OUT0108
SUPPLY_GROUP1:OpGrpCom; // CHASSIS.GROUP1
LEFTTRACKDIVERT_OP:OpCom; // CHASSIS.OUT0200
LTF_OP:OpCom; // CHASSIS.OUT0201
LTR_OP:OpCom; // CHASSIS.OUT0202
RIGHTTRACKDIVERT_OP:OpCom; // CHASSIS.OUT0203
RTF_OP:OpCom; // CHASSIS.OUT0204
RTR_OP:OpCom; // CHASSIS.OUT0205
DRUMONOFF_OP:OpCom; // CHASSIS.OUT0206
FEEDERONOFF_OP:OpCom; // CHASSIS.OUT0207
ECUENABLE:OpCom; // CHASSIS.OUT0208
SUPPLY_GROUP2:OpGrpCom; // CHASSIS.GROUP2
SPARE_OUT3000:OpCom; // CHASSIS.OUT3000
SPARE_OUT3001:OpCom; // CHASSIS.OUT3001


// Machine_IO_Outputs_STRUCT_CODE_GEN_STOP
Siren:  OpCom_CR0403; // AUX_OP0 
AUX_OP1: OpCom_CR0403; // AUX_OP1
AUX_OP2: OpCom_CR0403; // AUX_OP2
FanFwd_OP:  OpCom_CR0403; // AUX_OP3
FanRev_OP:  OpCom_CR0403; // AUX_OP4
SideConvRaise_RadialLeft_OP:  OpCom_CR0403; // AUX_OP5
SideConvLower_RadialRight_OP:  OpCom_CR0403; // AUX_OP6
DivertValve: OpCom_CR0403; // AUX_OP7

END_STRUCT
END_TYPE

// Device/Application/LIBS/IO Diagnostics/HMI_PLC_CR721S_IO
TYPE HMI_PLC_CR721S_IO :
STRUCT
	IN0100: CRXXXX_Input_Display;
	IN0101: CRXXXX_Input_Display;
	IN0102: CRXXXX_Input_Display;
	IN0103: CRXXXX_Input_Display;
	IN0200: CRXXXX_Input_Display;
	IN0201: CRXXXX_Input_Display;
	IN0202: CRXXXX_Input_Display;
	IN0203: CRXXXX_Input_Display;
	IN0600: CRXXXX_Input_Display;
	IN0601: CRXXXX_Input_Display;
	IN0602: CRXXXX_Input_Display;
	IN0603: CRXXXX_Input_Display;
	IN0700: CRXXXX_Input_Display;
	IN0701: CRXXXX_Input_Display;
	IN0702: CRXXXX_Input_Display;
	IN0703: CRXXXX_Input_Display;

	IN0000: CRXXXX_Input_Display;
	IN0001: CRXXXX_Input_Display;
	IN0002: CRXXXX_Input_Display;
	IN0003: CRXXXX_Input_Display;
	IN0500: CRXXXX_Input_Display;
	IN0501: CRXXXX_Input_Display;
	IN0502: CRXXXX_Input_Display;
	IN0503: CRXXXX_Input_Display;

	IN0400: CRXXXX_Input_Display;
	IN0401: CRXXXX_Input_Display;
	IN0900: CRXXXX_Input_Display;
	IN0901: CRXXXX_Input_Display;
	
	IN0300: CRXXXX_Input_Display;
	IN0301: CRXXXX_Input_Display;
	IN0800: CRXXXX_Input_Display;
	IN0801: CRXXXX_Input_Display;
	
	IN1100: CRXXXX_Input_Display;
	IN1101: CRXXXX_Input_Display;
	IN1102: CRXXXX_Input_Display;
	IN1103: CRXXXX_Input_Display;
	IN1600: CRXXXX_Input_Display;
	IN1601: CRXXXX_Input_Display;
	IN1602: CRXXXX_Input_Display;
	IN1603: CRXXXX_Input_Display;
	
	IN1000: CRXXXX_Input_Display;
	IN1001: CRXXXX_Input_Display;
	IN1002: CRXXXX_Input_Display;
	IN1003: CRXXXX_Input_Display;
	IN1500: CRXXXX_Input_Display;
	IN1501: CRXXXX_Input_Display;
	IN1502: CRXXXX_Input_Display;
	IN1503: CRXXXX_Input_Display;

	IN1200: CRXXXX_Input_Display;
	IN1201: CRXXXX_Input_Display;
	IN1202: CRXXXX_Input_Display;
	IN1203: CRXXXX_Input_Display;
	IN1400: CRXXXX_Input_Display;
	IN1401: CRXXXX_Input_Display;
	IN1402: CRXXXX_Input_Display;
	IN1403: CRXXXX_Input_Display;
	IN1700: CRXXXX_Input_Display;
	IN1701: CRXXXX_Input_Display;
	IN1702: CRXXXX_Input_Display;
	IN1703: CRXXXX_Input_Display;
	IN1800: CRXXXX_Input_Display;
	IN1801: CRXXXX_Input_Display;
	IN1802: CRXXXX_Input_Display;
	IN1803: CRXXXX_Input_Display;
	
	IN1300: CRXXXX_Input_Display;
	IN1301: CRXXXX_Input_Display;
	IN1302: CRXXXX_Input_Display;
	IN1303: CRXXXX_Input_Display;	

	OUT0000: CRXXXX_Output_Display;
	OUT0001: CRXXXX_Output_Display;
	OUT0002: CRXXXX_Output_Display;
	OUT0003: CRXXXX_Output_Display;
	OUT0004: CRXXXX_Output_Display;
	OUT0005: CRXXXX_Output_Display;
	OUT0006: CRXXXX_Output_Display;
	OUT0007: CRXXXX_Output_Display;
	OUT0008: CRXXXX_Output_Display;
	
	OUT0100: CRXXXX_Output_Display;
	OUT0101: CRXXXX_Output_Display;
	OUT0102: CRXXXX_Output_Display;
	OUT0103: CRXXXX_Output_Display;
	OUT0104: CRXXXX_Output_Display;
	OUT0105: CRXXXX_Output_Display;
	OUT0106: CRXXXX_Output_Display;
	OUT0107: CRXXXX_Output_Display;
	OUT0108: CRXXXX_Output_Display;
	
	OUT0200: CRXXXX_Output_Display;
	OUT0201: CRXXXX_Output_Display;
	OUT0202: CRXXXX_Output_Display;
	OUT0203: CRXXXX_Output_Display;
	OUT0204: CRXXXX_Output_Display;
	OUT0205: CRXXXX_Output_Display;
	OUT0206: CRXXXX_Output_Display;
	OUT0207: CRXXXX_Output_Display;
	OUT0208: CRXXXX_Output_Display;

	OUT3000: CRXXXX_Output_Display;
	OUT3001: CRXXXX_Output_Display;
	
	OUT0300: CRXXXX_Output_Display;
	OUT0301: CRXXXX_Output_Display;
	OUT0302: CRXXXX_Output_Display;
	OUT0303: CRXXXX_Output_Display;
	OUT0304: CRXXXX_Output_Display;
	OUT0305: CRXXXX_Output_Display;
	OUT0306: CRXXXX_Output_Display;
	OUT0307: CRXXXX_Output_Display;
	OUT0308: CRXXXX_Output_Display;
	
	OUT0400: CRXXXX_Output_Display;
	OUT0401: CRXXXX_Output_Display;
	OUT0402: CRXXXX_Output_Display;
	OUT0403: CRXXXX_Output_Display;
	OUT0404: CRXXXX_Output_Display;
	OUT0405: CRXXXX_Output_Display;
	OUT0406: CRXXXX_Output_Display;
	OUT0407: CRXXXX_Output_Display;
	OUT0408: CRXXXX_Output_Display;

	OUT0500: CRXXXX_Output_Display;
	OUT0501: CRXXXX_Output_Display;
	OUT0502: CRXXXX_Output_Display;
	OUT0503: CRXXXX_Output_Display;
	OUT0504: CRXXXX_Output_Display;
	OUT0505: CRXXXX_Output_Display;
	OUT0506: CRXXXX_Output_Display;
	OUT0507: CRXXXX_Output_Display;
	OUT0508: CRXXXX_Output_Display;
	
	OUT3002: CRXXXX_Output_Display;
	
	GROUP0: CRXXXX_Output_Group_Display;
	GROUP1: CRXXXX_Output_Group_Display;
	GROUP2: CRXXXX_Output_Group_Display;
	GROUP3: CRXXXX_Output_Group_Display;
	GROUP4: CRXXXX_Output_Group_Display;
	GROUP5: CRXXXX_Output_Group_Display;	
END_STRUCT
END_TYPE

// Device/Application/LIBS/IO Diagnostics/HMI_PLC_CR0709_IO
TYPE HMI_PLC_CR0709_IO :
STRUCT
	IN0100: CRXXXX_Input_Display;
	IN0101: CRXXXX_Input_Display;
	IN0102: CRXXXX_Input_Display;
	IN0103: CRXXXX_Input_Display;
	IN0200: CRXXXX_Input_Display;
	IN0201: CRXXXX_Input_Display;
	IN0202: CRXXXX_Input_Display;
	IN0203: CRXXXX_Input_Display;
	IN0600: CRXXXX_Input_Display;
	IN0601: CRXXXX_Input_Display;
	IN0602: CRXXXX_Input_Display;
	IN0603: CRXXXX_Input_Display;
	IN0700: CRXXXX_Input_Display;
	IN0701: CRXXXX_Input_Display;
	IN0702: CRXXXX_Input_Display;
	IN0703: CRXXXX_Input_Display;

	IN0000: CRXXXX_Input_Display;
	IN0001: CRXXXX_Input_Display;
	IN0002: CRXXXX_Input_Display;
	IN0003: CRXXXX_Input_Display;
	IN0500: CRXXXX_Input_Display;
	IN0501: CRXXXX_Input_Display;
	IN0502: CRXXXX_Input_Display;
	IN0503: CRXXXX_Input_Display;

	IN0400: CRXXXX_Input_Display;
	IN0401: CRXXXX_Input_Display;
	IN0900: CRXXXX_Input_Display;
	IN0901: CRXXXX_Input_Display;
	
	IN0300: CRXXXX_Input_Display;
	IN0301: CRXXXX_Input_Display;
	IN0800: CRXXXX_Input_Display;
	IN0801: CRXXXX_Input_Display;

	OUT0000: CRXXXX_Output_Display;
	OUT0001: CRXXXX_Output_Display;
	OUT0002: CRXXXX_Output_Display;
	OUT0003: CRXXXX_Output_Display;
	OUT0004: CRXXXX_Output_Display;
	OUT0005: CRXXXX_Output_Display;
	OUT0006: CRXXXX_Output_Display;
	OUT0007: CRXXXX_Output_Display;
	OUT0008: CRXXXX_Output_Display;
	
	OUT0100: CRXXXX_Output_Display;
	OUT0101: CRXXXX_Output_Display;
	OUT0102: CRXXXX_Output_Display;
	OUT0103: CRXXXX_Output_Display;
	OUT0104: CRXXXX_Output_Display;
	OUT0105: CRXXXX_Output_Display;
	OUT0106: CRXXXX_Output_Display;
	OUT0107: CRXXXX_Output_Display;
	OUT0108: CRXXXX_Output_Display;
	
	OUT0200: CRXXXX_Output_Display;
	OUT0201: CRXXXX_Output_Display;
	OUT0202: CRXXXX_Output_Display;
	OUT0203: CRXXXX_Output_Display;
	OUT0204: CRXXXX_Output_Display;
	OUT0205: CRXXXX_Output_Display;
	OUT0206: CRXXXX_Output_Display;
	OUT0207: CRXXXX_Output_Display;
	OUT0208: CRXXXX_Output_Display;

	OUT3000: CRXXXX_Output_Display;
	OUT3001: CRXXXX_Output_Display;	
	
	GROUP0: CRXXXX_Output_Group_Display;
	GROUP1: CRXXXX_Output_Group_Display;
	GROUP2: CRXXXX_Output_Group_Display;
END_STRUCT
END_TYPE

// Device/Application/LIBS/HMI/HMI_TASK_INFO_STRUCT
TYPE HMI_TASK_INFO_STRUCT :
STRUCT
    dwCycleTimeTask: DWORD;       
    dwIntervalTask: DWORD;
    fTaskCpuLoad: REAL;
    sNameTask: STRING(20);	
END_STRUCT
END_TYPE

// Device/Application/App_Common/Vizualisations/Viz_Structures/Viz_Footer_Struct
TYPE Viz_Footer_Struct :
STRUCT
	SystemVoltageStrFormat:STRING:='%.1fv';
	SystemVoltageStr: STRING;
	SystemVoltageColour: DWORD;
	SystemVoltageVisable: BOOL;

	Siren: BOOL;
	Beacon: BOOL;
	
	DisplayDateTimeString: STRING(30);
	
	Header_Message_Show:BOOL;
	Header_Message_Str: STRING;
	Header_Message_Colour: DWORD;
	Header_Message_Show_Flash:BOOL;
	Header_Message_Show_RTC:BOOL;
	
	NumberErrors:WORD;
	NumberWarnings:WORD;
	ShowErrorIcon:BOOL;
	ShowWarningIcon:BOOL;	
END_STRUCT
END_TYPE

// Device/Application/App_Common/Vizualisations/Viz_Structures/Viz_Misc_Status_Struct
TYPE Viz_Misc_Status_Struct :
STRUCT
END_STRUCT
END_TYPE

// Device/Application/App_Common/Vizualisations/Viz_Structures/Viz_Sections
TYPE Viz_Sections :
STRUCT
	System_Header: IFM_HMI_Version_System_Header;
	Footer: Viz_Footer_Struct;
	Options: Viz_Options_Struct;
END_STRUCT
END_TYPE

// Device/Application/App_Common/Vizualisations/Viz_Structures/Viz_Options_Struct
TYPE Viz_Options_Struct :
STRUCT
	Imperial_Readings: BOOL:=TRUE;
	USA_Time_Format: BOOL := FALSE;
END_STRUCT
END_TYPE

// Device/Application/App_CODE_GEN/MAIN_CODE_GEN/App_CODE_GEN/Machine IO/Structs/T620X_Radial_Inputs
TYPE T620X_Radial_Inputs :
STRUCT
// Machine_IO_Inputs_STRUCT_CODE_GEN_START

// generated (UTC): 2024-07-23 18:31:25.192393+00:00

ESTOP_OK:IpCom; // CHASSIS IN0100
DRUM_PRESSURE:IpCom; // CHASSIS IN0101
Radial_RightLimitSwitch:IpCom; // CHASSIS IN0102
Radial_LeftLimitSwitch:IpCom; // CHASSIS IN0103
MachineMode:IpCom; // CHASSIS IN0200 - LOW Standard, High Radial Machine
KeySwitchCranking:IpCom; // CHASSIS IN0201
SPARE_IN0202:IpCom; // CHASSIS IN0202
SPARE_IN0203:IpCom; // CHASSIS IN0203
SPARE_IN0600:IpCom; // CHASSIS IN0600
SPARE_IN0601:IpCom; // CHASSIS IN0601
SPARE_IN0602:IpCom; // CHASSIS IN0602
SPARE_IN0603:IpCom; // CHASSIS IN0603
SPARE_IN0700:IpCom; // CHASSIS IN0700
RADIORHS_JACKLEGRAISE_REQ:IpCom; // CHASSIS IN0701
RHS_TROMMELDOORSW:IpCom; // CHASSIS IN0702
LHS_TROMMELDOORSW:IpCom; // CHASSIS IN0703
HYDOILTEMP_SW:IpCom; // CHASSIS IN0000
HYDOILLEVEL_SW:IpCom; // CHASSIS IN0001
THERMOSTAT:IpCom; // CHASSIS IN0002
RADIORHS_JACKLEGLOWER_REQ:IpCom; // CHASSIS IN0003
RADIOLHS_JACKLEGRAISE_REQ:IpCom; // CHASSIS IN0500
RADIOLHS_JACKLEGLOWER_REQ:IpCom; // CHASSIS IN0501
SideConvRaise_RadialMoveRight:IpCom; // CHASSIS IN0502
SideConvLower_RadialMoveLeft:IpCom; // CHASSIS IN0503
SPARE_IN0400:IpCom; // CHASSIS IN0400
FUELLEVEL_PERCENT:IpCom; // CHASSIS IN0401
UMBTRACKREQ:IpCom; // CHASSIS IN0900
UMBMACHINESTOP:IpCom; // CHASSIS IN0901
RTF_REQ:IpCom; // CHASSIS IN0300
RTR_REQ:IpCom; // CHASSIS IN0301
LTF_REQ:IpCom; // CHASSIS IN0800
LTR_REQ:IpCom; // CHASSIS IN0801


// Machine_IO_Inputs_STRUCT_CODE_GEN_STOP 

END_STRUCT
END_TYPE

// Device/Application/App_Common/GVLS/NV_Sys_Settings_Struct
TYPE NV_Sys_Settings_Struct :
STRUCT
	Engine_Start_Charge_Battery_Voltage : REAL:=11.7*2; //(12v to 15v)
	Engine_Start_Charge_Battery_Time_mins: WORD:=1; //(1 to 30 mins)
	Engine_Stop_Charge_Battery_Voltage: REAL:=14.0*2; //(12v to 15v)
	Engine_Stop_Charge_Battery_Time_mins:WORD:=10; //(1 to 30 mins)
	
	Battery_Warning_Voltage:REAL:=11.8*2;
	Battery_Warning_Time: WORD:=1;
	Battery_Warning_Reset_Voltage:REAL:=12.0*2;
	Battery_Warning_Reset_Time: WORD:=1;
	Engine_Battery_Warning_Enable:BOOL :=FALSE;	
	Engine_Battery_Charge_Enable:BOOL :=FALSE;
	
	Imperial_Readings: BOOL:=TRUE;
	USA_Time_Format: BOOL:=FALSE;	
END_STRUCT
END_TYPE

// Device/Application/App_Common/Nav/TX_TO_MAIN_HMI_STRUCT
TYPE TX_TO_MAIN_HMI_STRUCT :
STRUCT
	Alarms_Clear_All: BOOL;
	Alarms_Clear_Inactive: BOOL;	
END_STRUCT
END_TYPE

// Device/Application/LIBS/Alarms/Struct/SLL_LOGGER_ITEM_GROUP
TYPE SLL_LOGGER_ITEM_GROUP :
STRUCT
	ErrorApp:BOOL;
	ErrorIO:BOOL;
	WarningApp:BOOL;
	WarningIO:BOOL;
	HushOption:BOOL;	
END_STRUCT
END_TYPE

// Device/Application/LIBS/Alarms/Struct/SLL_LOGGER_MAIN_SRUCT
TYPE SLL_LOGGER_MAIN_SRUCT:
STRUCT
	LOGGER_LIST_SIZE: WORD:=50;
	LOGGER_LIST: ARRAY [0..49] OF SLL_LOGGER_ITEM;
END_STRUCT
END_TYPE

// Device/Application/LIBS/Alarms/Struct/SLL_LOGGER_ITEM_UDP
TYPE SLL_LOGGER_ITEM_UDP :
STRUCT
	START_INDEX:WORD;
	TOTAL_ITEMS:WORD;
	ITEMS: ARRAY [0..9] OF SLL_LOGGER_ITEM;
	NUMBER_ITEMS:WORD:=10;
END_STRUCT
END_TYPE

// Device/Application/LIBS/Alarms/Struct/SLL_LOGGER_ITEM_FLAGS
TYPE SLL_LOGGER_ITEM_FLAGS :
STRUCT
	Active:BOOL;
	Acknowledged:BOOL;
END_STRUCT
END_TYPE

// Device/Application/LIBS/Alarms/Struct/SLL_LOGGER_ITEM
TYPE SLL_LOGGER_ITEM :
STRUCT
	ID:WORD;
	Empty:BOOL;
	TimeDateTriggered:SYSTIME; // milli-seconds since 1.1.1970 00:00:000 UTC
	Group:SLL_LOGGER_ITEM_GROUP;
	Flags:SLL_LOGGER_ITEM_FLAGS;
	Addtional_Info:STRING(50);
END_STRUCT
END_TYPE

// Device/Application/LIBS/Alarms/Struct/SENSOR_SCALE
(*
For OSCAT_BASIC.SCALE to store device scaling and limit information
*)
TYPE SENSOR_SCALE :
STRUCT
	K_FACTOR: REAL;
	OFFSET: REAL;
	MAXIMUM: REAL;
	MINIMUM: REAL;
	UNIT_IN: STRING(10);
	UNIT_OUT: STRING(10);
END_STRUCT
END_TYPE

// Device/Application/App_Common/GVLS/T620X_SETTINGS
TYPE T620X_SETTINGS :
STRUCT
	FwdTime_sec: WORD;
	RevTime_sec: WORD;
	TailConvSpd_Percent: BYTE:=100;
	SideConvSpd_Percent: BYTE:=100;
	SideTransferConvSpd_Percent: BYTE:=100;
	CollectConvSpd_Percent: BYTE:=100;
	DrumSpd_Percent: BYTE:=100;
	FeederSpd_Percent: BYTE:=100;
	TailConvSpd_Min_mA: INT:=500;
	TailConvSpd_Max_mA: INT:=1450;
	SideConvSpd_Min_mA: INT:=500;
	SideConvSpd_Max_mA: INT:=1450;
	SideTransferConvSpd_Min_mA: INT:=500;
	SideTransferConvSpd_Max_mA: INT:=1450;
	CollectConvSpd_Min_mA: INT:=500;
	CollectConvSpd_Max_mA: INT:=1450;
	DrumSpd_Min_mA: INT:=500;
	DrumSpd_Max_mA: INT:=1450;
	FeederSpd_Min_mA: INT:=500;
	FeederSpd_Max_mA: INT:=1450;
	EnableDrumPressCutOut: BOOL:=TRUE;
	
	DrumPressReset_SP: INT:=150; // 150 Bar reset level
	DrumPressHi_SP: INT:=160; // 160 Bar warning level
	DrumPressHiHi_SP: INT:=165; // 165 Bar error level
		
	RadialTimeDelay_SP: DWORD:=60; // used in the switch mode
	RadialTimeOut_SP: DWORD := 70; // used in pure timer mode
	
	Fan_FwdTime_mins:DWORD:=20;
	Fan_RevTime_secs:DWORD:=30;
	
	// can be set by tech logged in - with limits!
	AutoRunningRpm:WORD:=2200;
	TrackModeRpm:WORD:=1400;

	// Not Accesable - used as limit in the tech view
	TrackModeRpmMin:WORD:=1200;
	TrackModeRpmMax:WORD:=1400;
	
	AutoRunningRpmMin:WORD:=800;
	AutoRunningRpmMax:WORD:=2200;

	Valve_mA_Max:WORD:=1500;
	
	DrumPressMax: INT:= 230;	
END_STRUCT
END_TYPE

// Device/Application/LIBS/IO Diagnostics/HMI_PLC_CR0403_IO
TYPE HMI_PLC_CR0403_IO :
STRUCT
	OP0: CR0403_Output_Display;
	OP1: CR0403_Output_Display;
	OP2: CR0403_Output_Display;
	OP3: CR0403_Output_Display;
	OP4: CR0403_Output_Display;
	OP5: CR0403_Output_Display;
	OP6: CR0403_Output_Display;
	OP7: CR0403_Output_Display;	
END_STRUCT
END_TYPE

// Device/Application/App_Common/Vizualisations/DIAG_IO/CR0403/CR0403_OUTPUTS_STATES
TYPE CR0403_OUTPUTS_STATES :
STRUCT
	OP0 : CRXXXX_OUTPUT_STATE_DATA;
	OP1 : CRXXXX_OUTPUT_STATE_DATA;
	OP2 : CRXXXX_OUTPUT_STATE_DATA;
	OP3 : CRXXXX_OUTPUT_STATE_DATA;
	OP4 : CRXXXX_OUTPUT_STATE_DATA;
	OP5 : CRXXXX_OUTPUT_STATE_DATA;
	OP6 : CRXXXX_OUTPUT_STATE_DATA;
	OP7 : CRXXXX_OUTPUT_STATE_DATA;	
END_STRUCT
END_TYPE

// Device/Application/App_Common/GVLS/T620X_Running_Varaibles
TYPE T620X_Running_Varaibles :
STRUCT
	Fan_FwdTime_secs_Current:WORD:=0;
	Fan_Reverse_Latch:BOOL;
END_STRUCT
END_TYPE

// GVL
{attribute 'qualified_only'}
VAR_GLOBAL
END_VAR

// Device/Application/LIBS/HMI/GVL_KeyList_RT
{attribute 'qualified_only'}

(* 

!!! This GVL list is from project template !!!

The following variables returns a pulse for one scan cycle when a respective key is pressed (i.e. at rising trigger)
These key press event is detected by the state of variables in GVL GVL_KeyList.

For example, F1 function key of standard keyboard (MFII) is pressed, xF1 bit in this list will become TRUE for one scan cycle.

*)

VAR_GLOBAL

(*Display system key press event rising trigger pulse *)
	xF1 		: BOOL;		(* Event status of F1 function key *)
	xF2 		: BOOL;		(* Event status of F2 function key *)
	xF3 		: BOOL;		(* Event status of F3 function key *)
	xF4 		: BOOL;		(* Event status of F4 function key *)
	xF5 		: BOOL;		(* Event status of F5 function key *)
	xF6 		: BOOL;		(* Event status of F6 function key *)
	xF7 		: BOOL;		(* Event status of F7 function key *)
	xF8 		: BOOL;		(* Event status of F8 function key *)
	xF9 		: BOOL;		(* Event status of F9 function key *)
	xF10 		: BOOL;		(* Event status of F10 function key *)
	xUp 		: BOOL;		(* Event status of Up arrow key *)
	xDown		: BOOL;		(* Event status of Down arrow key *)
	xLeft 		: BOOL;		(* Event status of Left arrow key *)
	xRight 		: BOOL;		(* Event status of Right arrow key *)
	xKey_Return : BOOL;		(* Event status of Return (or Enter) key *)
END_VAR

// Device/Application/App_Common/GVLS/Net UDP RX TX/NVL_IO_CHASSIS
//This gobal variable list is received via the network.
//Sender: Imported from file '..\GVLS\NVL_UDP_CR711S_TO_HMI.gvl'
//Protocol: UDP

{attribute 'qualified_only'}
VAR_GLOBAL
	Version: SLL_IFM_Version.PLC_Version;
	System: SLL_IFM_CRXXXX.IFM_CRXXXX_System_STRUCT;
	All_Inputs: SLL_IFM_IO.CR0709_ALL_INPUTS_DATA;
	All_Outputs_Diag: SLL_IFM_IO.CR0709_ALL_OUTPUTS_DATA;	
	UDP_HB_RX_STATS: UDP_RX_STATS_HB_STRUCT;	
END_VAR

// Device/Application/App_Common/GVLS/Net UDP RX TX/NVL_Outputs_States_Chassis
{attribute 'qualified_only'}
VAR_GLOBAL
	Header: IFM_HMI_Version_System_Header;
	All: SLL_IFM_IO.CR0709_ALL_OUTPUT_STATES;
	App_Settings: T620X_SETTINGS;
END_VAR

// Device/Application/App_Common/GVLS/GVL_Versions
{attribute 'qualified_only'}
VAR_GLOBAL
	MAIN_HMI: SLL_IFM_Version.PLC_Version;	
	CHASSIS_PLC: SLL_IFM_Version.PLC_Version;	
END_VAR

// Device/Application/App_Common/GVLS/GVL_System
{attribute 'qualified_only'}
VAR_GLOBAL
	Password:STRING(20);
	
	Access_Level_Tech: BOOL;	
	
	IP_SETTINGS_WRONG:BOOL;
	
	MacAsString:STRING;
	MacAslword: LWORD;
	
	HMI_OP_FORCE_DISABLE:BOOL;
	HMI_ALARMS_ACK_DISABLE:BOOL;
	
	SIM_ENABLE: BOOL:=FALSE;
	SIM_DISABLE_UDP_IO:BOOL:=FALSE;
	SIM_CAS_PRIME_PULSE: BOOL:=FALSE;
	SIM_PRIME_PULSE: BOOL:=FALSE;
	
	SIM_IO_TAB_ENABLE: BOOL:=FALSE;
	SIM_IO_TAB_INDEX: INT;	
	
	ALARMS_PU_WAIT_MS: DWORD:= 7000;
	
	USA_Time_Format:BOOL;
	
	CLOSE_DLGS: BOOL;
END_VAR

// Device/Application/App_Common/GVLS/Machine_IO
{attribute 'qualified_only'}
VAR_GLOBAL
	Node_CHASSIS: NodeComFB;
	Node_AUX: NodeComFB;

	Inputs: T620X_Radial_Inputs;
	Outputs: T620X_Radial_Outputs;
END_VAR

// Device/Application/LIBS/HMI/GVL_KeyList
{attribute 'qualified_only'}

(* 

!!! This GVL list is from project template !!!

The following variables are controlled by key events mapped at Default Hotkey mapping list in Visualization Manager.

For example, F1 function key of standard keyboard (MFII) is pressed, xF1 bit in this list will become TRUE; when the same 
key is released then xF1 become FALSE.

*)

VAR_GLOBAL

(* Display system key press / release event status. TRUE = Key Pressed, FALSE = Key Released  *)
	xF1 		: BOOL;		(* Event status of F1 function key *)
	xF2 		: BOOL;		(* Event status of F2 function key *)
	xF3 		: BOOL;		(* Event status of F3 function key *)
	xF4 		: BOOL;		(* Event status of F4 function key *)
	xF5 		: BOOL;		(* Event status of F5 function key *)
	xF6 		: BOOL;		(* Event status of F6 function key *)
	xF7 		: BOOL;		(* Event status of F7 function key *)
	xF8 		: BOOL;		(* Event status of F8 function key *)
	xF9 		: BOOL;		(* Event status of F9 function key *)
	xF10 		: BOOL;		(* Event status of F10 function key *)
	xUp 		: BOOL;		(* Event status of Up arrow key *)
	xDown		: BOOL;		(* Event status of Down arrow key *)
	xLeft 		: BOOL;		(* Event status of Left arrow key *)
	xRight 		: BOOL;		(* Event status of Right arrow key *)
	xKey_Return : BOOL;		(* Event status of Return (or Enter) key *)
END_VAR

// Device/Application/App_CODE_GEN/MAIN_CODE_GEN/App_CODE_GEN/Alarms/GVL_Alarms
{attribute 'qualified_only'}
VAR_GLOBAL
// GVL_Alarms_Declare_CODE_GEN_START

// generated (UTC): 2024-07-23 18:31:25.263396+00:00

	EMERGENCY_STOP_COMMON: BOOL; // ID=101
	ETHERNET_PLC_COMMON_FAILURE: BOOL; // ID=102
	ETHERNET_CHASSIS_PLC_MISSING: BOOL; // ID=104
	ETHERNET_CHASSIS_PLC_ERROR_LT: BOOL; // ID=106
	ETHERNET_CHASSIS_PLC_ERROR_DIFF: BOOL; // ID=108
	ETHERNET_CHASSIS_PLC_ERROR_FROZEN: BOOL; // ID=110
	ETHERNET_CHASSIS_PLC_WARNING_DIFF: BOOL; // ID=112
	ETHERNET_CHASSIS_PLC_WARNING_FROZEN: BOOL; // ID=114
	Battery_Voltage_Warning: BOOL; // ID=118
// GVL_Alarms_Declare_CODE_GEN_STOP

	LowFuelWarn: BOOL;
	DrumHighPress_Warn: BOOL;
	DrumHighPress_Warn_Counter: WORD;
	
	LowHydOilAlarm: BOOL; // 120
	HydTempAlarm: BOOL; // 121
	DrumHighPress_Alarm: BOOL; // 122
	LowFuelAlarm: BOOL;	// 123
	AutoShutdownAlarm: BOOL; // 124
	LowOilPressAlarm: BOOL; // 125
	EngineHiTempAlarm: BOOL; //126
END_VAR

// Device/Application/LIBS/HMI/GVL_KeyList_FT
{attribute 'qualified_only'}

(* 

!!! This GVL list is from project template !!!

The following variables returns a pulse for one scan cycle when a respective key is released (i.e. at falling trigger).
These key release event is detected by the state of variables in GVL GVL_KeyList.

For example, F1 function key of standard keyboard (MFII) is released, xF1 bit in this list will become TRUE for one scan cycle.

*)

VAR_GLOBAL

(* Display system key release event falling trigger pulse. *)
	xF1 		: BOOL;		(* Event status of F1 function key *)
	xF2 		: BOOL;		(* Event status of F2 function key *)
	xF3 		: BOOL;		(* Event status of F3 function key *)
	xF4 		: BOOL;		(* Event status of F4 function key *)
	xF5 		: BOOL;		(* Event status of F5 function key *)
	xF6 		: BOOL;		(* Event status of F6 function key *)
	xF7 		: BOOL;		(* Event status of F7 function key *)
	xF8 		: BOOL;		(* Event status of F8 function key *)
	xF9 		: BOOL;		(* Event status of F9 function key *)
	xF10 		: BOOL;		(* Event status of F10 function key *)
	xUp 		: BOOL;		(* Event status of Up arrow key *)
	xDown		: BOOL;		(* Event status of Down arrow key *)
	xLeft 		: BOOL;		(* Event status of Left arrow key *)
	xRight 		: BOOL;		(* Event status of Right arrow key *)
	xKey_Return : BOOL;		(* Event status of Return (or Enter) key *)
END_VAR

// Device/Application/App_Common/GVLS/Viz/GVL_Viz
{attribute 'qualified_only'}
VAR_GLOBAL
	
	TextList_IFM_Diag_Codes: STRING:='TextList_IFM_Diag_Codes';
	TextList_IO_Diag: STRING:='TextList_IO_Diag';
	TextList_IO_Mimics_Inputs: STRING:='TextList_IO_Mimics_Inputs';
	TextList_IO_Mimics_Outputs: STRING:='TextList_IO_Mimics_Outputs';
	TextList_IO_Mimics_Com: STRING:='TextList_IO_Mimics_Com';
	
	TextList_Allow_Update: BOOL:=TRUE;
	
	Diag_Signal_Name_Toggle:BOOL:=TRUE; // true for simple signal name, flase to use Mimic_IO_GetText(GVL_Viz.TextList_IO_Diag,IpREF.PLC_IO_Ref);

	Input_Fault_Flash_Fast:BOOL;
	Input_Fault_Flash_Slow:BOOL;

	Output_Fault_Flash_Fast:BOOL;
	Output_Fault_Flash_Slow:BOOL;

	Estop_Fault_Flash_Fast:BOOL;
	Estop_Fault_Flash_Slow:BOOL;
	
	Estop_COLOUR_HEALTHY: 	DWORD:=16#FF009000;
	Estop_COLOUR_OTHER_ID: 	DWORD:=16#FF009000;
	Estop_COLOUR_THIS_ID: 	DWORD:=16#FFFF0000;
	Estop_COLOUR_FLASH_OFF: 	DWORD:=16#FF7F7F7F;
	Estop_COLOUR_ID_MISSING: 	DWORD:=16#FFFFA500;
	Estop_COLOUR_ID_UNAVAIL: 	DWORD:=16#FFFFA500;

	Diag_Input_Font_Colour_OK: DWORD:=16#FFFFFFFF;
	Diag_Input_Font_Colour_Fault: DWORD:=16#FFFF0000;	
	Diag_Input_Font_Colour_Unavail: DWORD:=16#FFFFA500;
	Diag_Input_Pin_Fault_Text: STRING := 'Input Pin Fault';
	Diag_Input_Unavailable_Text:STRING := 'Input Unavailable';

	Diag_Output_Font_Colour_OK: DWORD:=16#FFFFFFFF;
	Diag_Output_Font_Colour_Error: DWORD:=16#FFFF0000;	
	Diag_Output_Font_Colour_Warn: DWORD:=16#FFFFA500;
	Diag_Output_Font_Colour_Other: DWORD:=16#FF800080;
	Diag_Output_Font_Colour_Unavail: DWORD:=16#FFFFA500;

	IFM_IO_Output_DigRectColour_ON:DWORD:=16#FF00FF00;
	IFM_IO_Output_DigRectColour_OFF:DWORD:=16#FF7F7F7F;

	IFM_IO_Output_DigRectColour_ManOn:DWORD:=16#FFFFA500;
	IFM_IO_Output_DigRectColour_ManOff:DWORD:=16#FFA50000;

//	Diag_Output_Font_Fill_Colour_OK: DWORD:=16#FF000000;
//	Diag_Output_Font_Fill_Colour_Fault: DWORD:=16#FFFF0000;	
//	Diag_Output_Font_Fill_Colour_Warn: DWORD:=16#FFFFA500;
//	Diag_Output_Font_Fill_Colour_Unavail: DWORD:=16#FFFFA500;
	
//	Diag_Output_Pin_Fault_Text: STRING := 'Output Pin Fault';
	Diag_Output_Unavailable_Text: STRING := 'Output Unavailable';
//	Diag_Output_Group_Fault_Text: STRING := 'Supply Group Fault';
//	Diag_Output_Group_Off_Text: STRING := 'Supply Group OFF';
//	Diag_Output_Group_Off_Fault_Text: STRING := 'Supply Group OFF Fault';

	Input_Unavailable_Text: STRING:='Unavail';
	Input_Fault_Text: STRING:='Fault';

	Input_Pin_Fault_Text: STRING:='Fault';
	Input_Group_Fault_Text: STRING:='Fault';
	
	
	Output_Unavailable_Text: STRING:='Unavail';
	Output_Fault_Text: STRING:='Fault';

	
	
	
	Estop_Healthy: STRING:='Healthy';
	Estop_Not_Pressed: STRING:='Not Pressed';
	Estop_Pressed: STRING:='PRESSED';
	Estop_ID_Missing: STRING:='ID MISS';
	Estop_ID_Unavail: STRING:='Unavail.';	

	Input_Active_Frame_Colour: DWORD:=16#FF00FF00;
	Input_Active_Fill_Colour: DWORD:=16#FF000000;	
	Input_Active_Font_Colour: DWORD:=16#FF00FF00;	

	Input_Inactive_Frame_Colour: DWORD:=16#FF7F7F7F;
	Input_Inactive_Fill_Colour: DWORD:=16#FF000000;
	Input_Inactive_Font_Colour: DWORD:=16#FF7F7F7F;
	
	Input_Unavail_Frame_Colour: DWORD:=16#FFFFA500;
	Input_Unavail_Fill_Colour: DWORD:=16#FF000000;
	Input_Unavail_Font_Colour: DWORD:=16#FFFFA500;

	Input_Fault_Frame_Colour: DWORD:=16#FFFF0000;
	Input_Fault_Fill_Colour: DWORD:=16#FF000000;
	Input_Fault_Font_Colour: DWORD:=16#FFFF0000;
	
	Output_Active_Frame_Colour: DWORD:=16#FF00FF00;
	Output_Active_Fill_Colour: DWORD:=16#FF00FF00;	
	Output_Active_Font_Colour: DWORD:=16#FF000000;	

	Output_Inactive_Frame_Colour: DWORD:=16#FF7F7F7F;
	Output_Inactive_Fill_Colour: DWORD:=16#FF7F7F7F;
	Output_Inactive_Font_Colour: DWORD:=16#FF000000;
	
	Output_Unavail_Frame_Colour: DWORD:=16#FFFFA500;
	Output_Unavail_Fill_Colour: DWORD:=16#FFFFA500;
	Output_Unavail_Font_Colour: DWORD:=16#FF000000;

	Output_Fault_Frame_Colour: DWORD:=16#FFFF0000;
	Output_Fault_Fill_Colour: DWORD:=16#FFFF0000;
	Output_Fault_Font_Colour: DWORD:=16#FF000000;		

	Button_Active_Colour: DWORD:=16#FF00FF00;
	Button_Inactive_Colour: DWORD:=16#FF7F7F7F;
	Button_Font_Colour: DWORD:=16#FF000000;
	
	IFM_IO_Input_DigRectColour_ON:DWORD:=16#FF00FF00;
	IFM_IO_Input_DigRectColour_OFF:DWORD:=16#FF7F7F7F;
	
	Common_Flash_Fast: BOOL;
	Common_Flash_Slow: BOOL;

	Alarm_Log_Active_Colour: DWORD:=16#FFFF0000;
	Alarm_Log_InActive_Colour: DWORD:=16#FF555555;
	Alarm_Log_None_Colour: DWORD:=16#FF000000;
	

	PrestartColor_DWORD: DWORD := 16#FFE59400;
	RunningColor_DWORD: DWORD := 16#FF00E000;
	IdleColor_DWORD: DWORD := 16#FF000000;
		
	SelColor_DWORD: DWORD := 16#FF84DE02; // 132,222,2
	SelColor_DWORD_DEFAULT: DWORD := 16#FF84DE02; // 132,222,2	
END_VAR

// Device/Application/App_Common/GVLS/Viz/NVL_Viz
{attribute 'qualified_only'}
VAR_GLOBAL
	Sections: Viz_Sections;
END_VAR

// Device/Application/App_Common/GVLS/GVL_Persistant_Defaults
{attribute 'qualified_only'}
VAR_GLOBAL
	System_Settings: NV_Sys_Settings_Struct; // dumy structure used to prime varaibles
	App_Settings: T620X_SETTINGS;
END_VAR

// Device/Application/LIBS/Logging/GVL_Logging
{attribute 'qualified_only'}
VAR_GLOBAL
	Main_Log_Filename: STRING;
	Main_Log_Filename_Updated: INT:=0;
	Main_Log_Filename_Updated_Prev: INT:=0;	
END_VAR

// Device/Application/App_Common/GVLS/GVL_Persistant
{attribute 'qualified_only'}
VAR_GLOBAL PERSISTENT RETAIN
	gl_SerialNumber: STRING := '2117343.00';
	Sys_Settings: NV_Sys_Settings_Struct;
	App_Settings: T620X_SETTINGS;
	App_Run_Vars: T620X_Running_Varaibles;
	ALARM_LOGGER_LIST: SLL_LOGGER_MAIN_SRUCT;
	Brightness: USINT (0..100):=80;	
END_VAR

// Device/Application/App_Common/GVLS/GVL_Machine
{attribute 'qualified_only'}
VAR_GLOBAL
	ChargeLamp: BOOL;	
	ECUenable: BOOL;
	UmbMachineShutdown: BOOL;
	
	
	AutoMode: BOOL;	
	AutoModeAllow: BOOL;	
	
	AutoStarting: BOOL;	
	AutoStopping: BOOL;	

	TrackingOn: BOOL;

	TailConvOn: BOOL;
	TailConvPreStart: BOOL;
	
	SideConvOn: BOOL;
	SideConvPreStart: BOOL;

	SideTransferOn: BOOL;
	SideTransferPreStart: BOOL;	
	
	CollectConvOn: BOOL;
	CollectConvPreStart: BOOL;
	
	DrumOn: BOOL;
	DrumPreStart: BOOL;

	FeederOn: BOOL;
	FeederPreStart: BOOL;
	
	SetupDumpValveOn: BOOL;
	SetupDumpValvePreStart: BOOL;
	SetupDumpValveIcon: BOOL;
		
	PreSiren: BOOL;
	PreSirenBlink: BOOL;
	
	EngineRunning: BOOL; // basic engine above 500rpm
	
	TrackingModeAllow: BOOL;
	TrackingModeStarted: BOOL;	
	TrackingMode: BOOL;
	TrackPreSiren: BOOL;
	TrackPreSiren_Flash: BOOL;
	
	CriticalShutdown: BOOL;	
	EngineRunningForce: BOOL:=TRUE;
	
	DrumPressMsg: STRING;
END_VAR

// Device/Application/App_PLC/SIM_APP
{attribute 'qualified_only'}
VAR_GLOBAL
	SIM_SETUP: BOOL;
	UNLINK_INPUTS:BOOL;
	
	SIM_SKIP_IO_CONFIG: BOOL;
	
	ESTOP_VALUE: BOOL:=TRUE;
	
	RPM_LOOPBACK: BOOL:=TRUE;
	SIM_THERMOSTAT: BOOL;
	
	DRUM_PRESSURE_SIM: BOOL;
	
	FUEL_LEVEL_SIM_ENA: BOOL;
END_VAR

// Device/Application/App_PLC/GVL_APP
{attribute 'qualified_only'}
VAR_GLOBAL
	HalfSecBlink: BOOL;
	OneSecBlink: BOOL;
	Reset: BOOL; // pressing the auto stop button on main page

	ReqJackLegs: BOOL;
	ReqHydSetup: BOOL;
	ManualMode: BOOL;
	
	AutoRadialEnabled: BOOL;
	AutoRadialModeActive: BOOL;
	AutoRadialTimed: BOOL;
	AutoRadialModeIcon: BOOL;
	
	RadialTimeOutFlag: BOOL;
	
	MachineModelRadial: BOOL;	
END_VAR

// Device/Application/App_Common/GVLS/GVL_Engine
{attribute 'qualified_only'}
VAR_GLOBAL
	EngineRPM: WORD;
	EngineLoad: WORD;
	
	EngineRpmPerctangeString: STRING;
	
	RequestedRPM: WORD;
	
	ElevateRpmAllowed: BOOL;
	
	DM1_Index: BYTE;
	DM1_Index_SPN: DWORD;
	DM1_Index_FMI: BYTE;
	DM1_Index_OC: BYTE;
	QtyOf_SPN_Codes: BYTE;	
	
	EngineWarningLamp: BOOL;
	EngineProtectLamp: BOOL;
	EngineStopLamp: BOOL;
	MILamp: BOOL;
	
	DisplayEngineStopLamp: BOOL;	
	
	EngineLowOilPressAlarm: BOOL;
	EngineHiTempAlarm: BOOL;	

	DPF_RegenActive: BOOL; // not writen to yet!
	DPF_Lamp: BOOL;
	
	DPF_Lamp_Status: USINT;
	DPF_Regen_Inhibit1: BOOL;
	DPF_Regen_Inhibit2: BOOL;
	DPF_Regen_Inhibit3: BOOL;
	DPF_Regen_Inhibited: BOOL;
	DPF_Regen_Status: WORD;
	DPF_Regen_Status_String: STRING;
	
	Def_Lamp_Status: BYTE;
	Def_LowLevLamp: BOOL;		
	Def_TankLevelPercent: BYTE;
			
	CoolantTemperature_degC: INT;
	OilPress_bar: REAL;
	
	EngineHrs: REAL;
	
	EngineVoltage: REAL;
	
	FuelRate_LHr: REAL;		
END_VAR

// Device/Application/App_Common/GVLS/GVL_CAN_TX_AUX
{attribute 'qualified_only'}
VAR_GLOBAL
	OUTPUTS: CR0403_OUTPUTS_STATES;	
END_VAR

// Device/Application/App_Common/GVLS/GVL_J1939
{attribute 'qualified_only'}
VAR_GLOBAL
	EEC1_ActualEngPercentTorque:INT; // SPN:513
	EEC1_EngSpeed:REAL; // SPN:190
	EEC2_EngPercentLoadAtCurrentSpeed:USINT; // SPN:92
	EEC2_SCRThermalManagementActive:USINT; // SPN:5400
	EEC2_ActlMxAvailableEngPercentTorque:REAL; // SPN:3357
	EEC3_NominalFrictionPercentTorque:INT; // SPN:514
	EEC3_EngsDesiredOperatingSpeed:REAl; // SPN:515
	EEC5_EngExhstGsRcrculation1ValveCtrl:REAL; // SPN:2791
	ET1_EngCoolantTemp:INT; // SPN:1637
	ET1_EngFuelTemp1:INT; // SPN:174
	EFL_P1_EngOilPress:UINT; // SPN:100
	EFL_P1_EngCoolantLevel:REAL; // SPN:111
	EFL_P2_EngInjectorMeteringRail1Press:LREAL; // SPN:157
	LFC_EngTotalFuelUsed:REAL; // SPN:250
	AMB_BarometricPress:REAL; // SPN:108
	AMB_AmbientAirTemp:REAL; // SPN:171
	AMB_EngAirIntakeTemp:INT; // SPN:172
	IC1_EngIntakeManifold1Press:UINT; // SPN:102
	IC1_EngIntakeManifold1Temp:INT; // SPN:105
	IC1_EngAirIntakePress:UINT; // SPN:106
	VEP1_BatteryPotential_PowerInput1:REAL; // SPN:168
	VEP1_KeyswitchBatteryPotential:REAL; // SPN:158
	EFS_EngOilPrimingState:USINT; // SPN:3551
	EFS_FuelPumpPrimerStatus:USINT; // SPN:4083
	DPFC1_DieselParticulateFilterLampCmd:USINT; // SPN:3697
	DPFC1_DslPrtcltFltrActvRgnrtionStatus:USINT; // SPN:3700
	DPFC1_DieselParticulateFilterStatus:USINT; // SPN:3701
	DPFC1_DslPrtcltFltrActvRgnrtnInhbtdDTI:USINT; // SPN:3703
	DPFC1_DslPrtcltFltrActvRgnrtnInhbtdDTT:USINT; // SPN:3714
	DPFC1_DslPrtcltFltrActvRgnrtnInhbtdDTP:USINT; // SPN:3715
	AT1IG2_Aftrtrtmnt1DslPrtcltFltrInt_0000:REAL; // SPN:3242
	AT1T1I_Aftrtrtmnt1SCRCatalystTankLevel:REAL; // SPN:1761
	AT1T1I_Aftrtrtment1SCRCatalystTankTemp:INT; // SPN:3031
	AT1T1I_Aftrtrtmnt1DEFTnkLwLvlIndicator:USINT; // SPN:5245
	AT1T1I_AftrtrtmntSCROprtrIndcmntSvrity:USINT; // SPN:5246
	A1SCRDSI1_Aftertreatment1SCRSystemState:USINT; // SPN:4332
	A1SCREGT_Aftrtrtmnt1SCRCtlystIntkGasTemp:REAL; // SPN:4360
	A1DOC_Aftrtrtmnt1DslOxdtnCtlystIn_0000:REAL; // SPN:4765
	WFI_WaterInFuelIndicator:USINT; // SPN:97
	DLCC1_EngAirFilterRestrictionLampCmd:USINT; // SPN:5086
	DLCD1_EngOilPressLowLampData:USINT; // SPN:5099
	DLCD1_EngCoolantLevelLowLampData:USINT; // SPN:5101
	HOURS_EngTotalHoursOfOperation: REAL;
END_VAR

// Device/Application/LIBS/HMI/HMI_KEYPAD

(* !!! This POU is from project template !!! *)

PROGRAM HMI_KEYPAD
VAR
(* Below is the FB instance with initial values to set default key mapping. The default key map is as per the default values set for ifmDevice.stKEY_MAP_LIST. *)
	fbSetKeyMapping		: ifmDevice.SetKeyMapping;
	
	iNumPad		: INT; (* interger value, set with the numpad. *)
	rNumPad		: REAL; (* real value, set with the numpad. *)
	sKeyPad		: STRING; (* string value, set with the keypad. *)
	
	iMinVal		: INT:=0; (* minimum value which can be set for the numpad.*)
	iMaxVal		: INT:=9999; (* maximum value which can be set for the numpad.*)
	sTitleNumpad	: STRING; (* The title of the numpad.*)
	sTitleKeypad	: STRING; (* The title of the keypad.*)	
	Temp_Local: LREAL;
	Setpoint_Local: LREAL;
END_VAR
VAR // added by the converter: edge detectors and wires of the graphical bodies
    _ft1, _ft2, _ft3, _ft4, _ft5, _ft6, _ft7, _ft8, _ft9, _ft10, _ft11, _ft12, _ft13, _ft14, _ft15 : F_TRIG;
    _rt1, _rt2, _rt3, _rt4, _rt5, _rt6, _rt7, _rt8, _rt9, _rt10, _rt11, _rt12, _rt13, _rt14, _rt15 : R_TRIG;
END_VAR

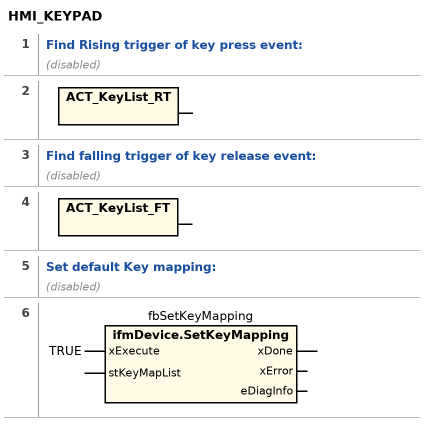
// NETWORK 1 (disabled)
// label: Find Rising trigger of key press event

// NETWORK 2
ACT_KeyList_RT();

// NETWORK 3 (disabled)
// label: Find falling trigger of key release event

// NETWORK 4
ACT_KeyList_FT();

// NETWORK 5 (disabled)
// label: Set default Key mapping

// NETWORK 6
fbSetKeyMapping(xExecute := TRUE); // ifmDevice.SetKeyMapping

ACTION ACT_KeyList_FT:
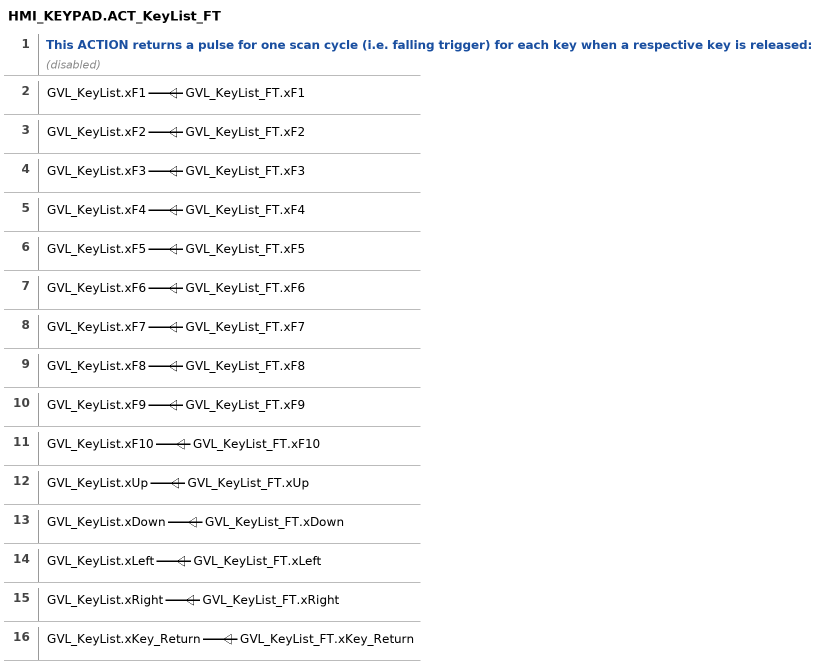
// NETWORK 1 (disabled)
// label: This ACTION returns a pulse for one scan cycle (i.e. falling trigger) for each key when a respective key is released

// NETWORK 2
_ft1(CLK := GVL_KeyList.xF1);
GVL_KeyList_FT.xF1 := _ft1.Q;

// NETWORK 3
_ft2(CLK := GVL_KeyList.xF2);
GVL_KeyList_FT.xF2 := _ft2.Q;

// NETWORK 4
_ft3(CLK := GVL_KeyList.xF3);
GVL_KeyList_FT.xF3 := _ft3.Q;

// NETWORK 5
_ft4(CLK := GVL_KeyList.xF4);
GVL_KeyList_FT.xF4 := _ft4.Q;

// NETWORK 6
_ft5(CLK := GVL_KeyList.xF5);
GVL_KeyList_FT.xF5 := _ft5.Q;

// NETWORK 7
_ft6(CLK := GVL_KeyList.xF6);
GVL_KeyList_FT.xF6 := _ft6.Q;

// NETWORK 8
_ft7(CLK := GVL_KeyList.xF7);
GVL_KeyList_FT.xF7 := _ft7.Q;

// NETWORK 9
_ft8(CLK := GVL_KeyList.xF8);
GVL_KeyList_FT.xF8 := _ft8.Q;

// NETWORK 10
_ft9(CLK := GVL_KeyList.xF9);
GVL_KeyList_FT.xF9 := _ft9.Q;

// NETWORK 11
_ft10(CLK := GVL_KeyList.xF10);
GVL_KeyList_FT.xF10 := _ft10.Q;

// NETWORK 12
_ft11(CLK := GVL_KeyList.xUp);
GVL_KeyList_FT.xUp := _ft11.Q;

// NETWORK 13
_ft12(CLK := GVL_KeyList.xDown);
GVL_KeyList_FT.xDown := _ft12.Q;

// NETWORK 14
_ft13(CLK := GVL_KeyList.xLeft);
GVL_KeyList_FT.xLeft := _ft13.Q;

// NETWORK 15
_ft14(CLK := GVL_KeyList.xRight);
GVL_KeyList_FT.xRight := _ft14.Q;

// NETWORK 16
_ft15(CLK := GVL_KeyList.xKey_Return);
GVL_KeyList_FT.xKey_Return := _ft15.Q;
END_ACTION

ACTION ACT_KeyList_RT:
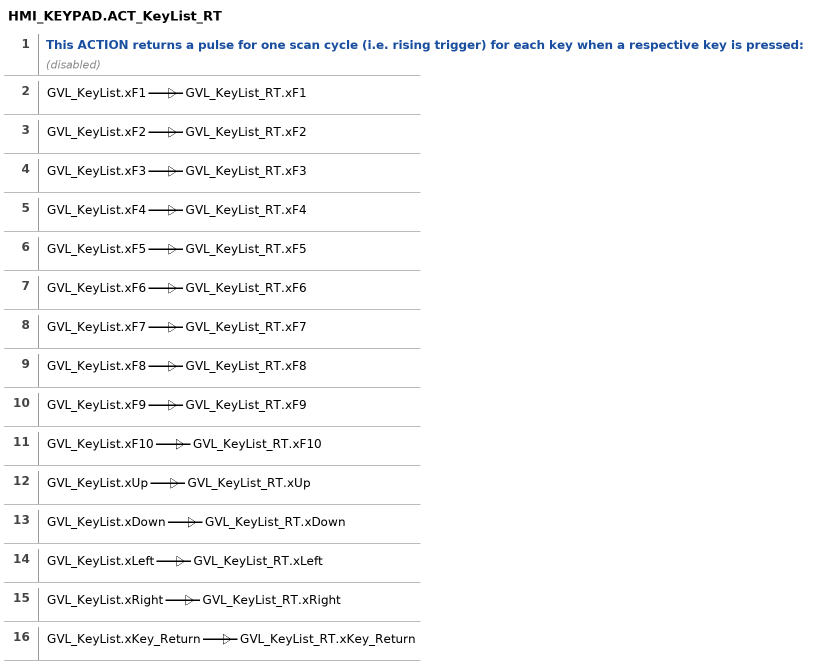
// NETWORK 1 (disabled)
// label: This ACTION returns a pulse for one scan cycle (i.e. rising trigger) for each key when a respective key is pressed

// NETWORK 2
_rt1(CLK := GVL_KeyList.xF1);
GVL_KeyList_RT.xF1 := _rt1.Q;

// NETWORK 3
_rt2(CLK := GVL_KeyList.xF2);
GVL_KeyList_RT.xF2 := _rt2.Q;

// NETWORK 4
_rt3(CLK := GVL_KeyList.xF3);
GVL_KeyList_RT.xF3 := _rt3.Q;

// NETWORK 5
_rt4(CLK := GVL_KeyList.xF4);
GVL_KeyList_RT.xF4 := _rt4.Q;

// NETWORK 6
_rt5(CLK := GVL_KeyList.xF5);
GVL_KeyList_RT.xF5 := _rt5.Q;

// NETWORK 7
_rt6(CLK := GVL_KeyList.xF6);
GVL_KeyList_RT.xF6 := _rt6.Q;

// NETWORK 8
_rt7(CLK := GVL_KeyList.xF7);
GVL_KeyList_RT.xF7 := _rt7.Q;

// NETWORK 9
_rt8(CLK := GVL_KeyList.xF8);
GVL_KeyList_RT.xF8 := _rt8.Q;

// NETWORK 10
_rt9(CLK := GVL_KeyList.xF9);
GVL_KeyList_RT.xF9 := _rt9.Q;

// NETWORK 11
_rt10(CLK := GVL_KeyList.xF10);
GVL_KeyList_RT.xF10 := _rt10.Q;

// NETWORK 12
_rt11(CLK := GVL_KeyList.xUp);
GVL_KeyList_RT.xUp := _rt11.Q;

// NETWORK 13
_rt12(CLK := GVL_KeyList.xDown);
GVL_KeyList_RT.xDown := _rt12.Q;

// NETWORK 14
_rt13(CLK := GVL_KeyList.xLeft);
GVL_KeyList_RT.xLeft := _rt13.Q;

// NETWORK 15
_rt14(CLK := GVL_KeyList.xRight);
GVL_KeyList_RT.xRight := _rt14.Q;

// NETWORK 16
_rt15(CLK := GVL_KeyList.xKey_Return);
GVL_KeyList_RT.xKey_Return := _rt15.Q;
END_ACTION

END_PROGRAM

// Device/Application/App_CODE_GEN/MAIN_CODE_GEN/App_CODE_GEN/Diag_IO/HMI_IO
PROGRAM HMI_IO
VAR
	Init_Link_Inputs: BOOL:=TRUE;
	Init_Link_Outputs: BOOL:=TRUE;
	Outputs_EnableAutoMan:BOOL:=TRUE;// AW TEMP 02-03-2024
	Wait_For_UDP_TON: TON;
END_VAR
VAR_INPUT
	CHASSIS: HMI_PLC_CR0709_IO;
	AUX: HMI_PLC_CR0403_IO;
END_VAR

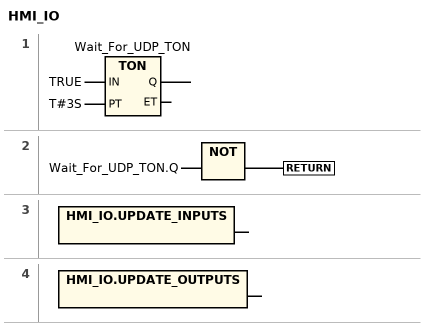
// NETWORK 1
Wait_For_UDP_TON(IN := TRUE, PT := T#3S); // TON

// NETWORK 2
IF NOT Wait_For_UDP_TON.Q THEN RETURN; END_IF

// NETWORK 3
HMI_IO.UPDATE_INPUTS();

// NETWORK 4
HMI_IO.UPDATE_OUTPUTS();

METHOD Update_Outputs
VAR
END_VAR
IF Init_Link_Outputs THEN
	Init_Output_Links();
END_IF
Init_Link_Outputs:=FALSE;

// HMI_IO_Update_Outputs_CODE_GEN_START

// generated (UTC): 2024-07-23 18:31:25.349399+00:00

CHASSIS.OUT0000();
CHASSIS.OUT0001();
CHASSIS.OUT0002();
CHASSIS.OUT0003();
CHASSIS.OUT0004();
CHASSIS.OUT0005();
CHASSIS.OUT0006();
CHASSIS.OUT0007();
CHASSIS.OUT0008();
CHASSIS.GROUP0();
CHASSIS.OUT0100();
CHASSIS.OUT0101();
CHASSIS.OUT0102();
CHASSIS.OUT0103();
CHASSIS.OUT0104();
CHASSIS.OUT0105();
CHASSIS.OUT0106();
CHASSIS.OUT0107();
CHASSIS.OUT0108();
CHASSIS.GROUP1();
CHASSIS.OUT0200();
CHASSIS.OUT0201();
CHASSIS.OUT0202();
CHASSIS.OUT0203();
CHASSIS.OUT0204();
CHASSIS.OUT0205();
CHASSIS.OUT0206();
CHASSIS.OUT0207();
CHASSIS.OUT0208();
CHASSIS.GROUP2();
CHASSIS.OUT3000();
CHASSIS.OUT3001();
// HMI_IO_Update_Outputs_CODE_GEN_STOP

AUX.OP0();
AUX.OP1();
AUX.OP2();
AUX.OP3();
AUX.OP4();
AUX.OP5();
AUX.OP6();
AUX.OP7();
END_METHOD

METHOD Init_Input_Links
VAR
END_VAR

// HMI_IO_Init_Input_Links_CODE_GEN_START

// generated (UTC): 2024-07-23 18:31:25.317398+00:00
CHASSIS.IN0100.Init(Machine_IO.Inputs.ESTOP_OK);
CHASSIS.IN0101.Init(Machine_IO.Inputs.DRUM_PRESSURE);
CHASSIS.IN0102.Init(Machine_IO.Inputs.Radial_RightLimitSwitch);
CHASSIS.IN0103.Init(Machine_IO.Inputs.Radial_LeftLimitSwitch);
CHASSIS.IN0200.Init(Machine_IO.Inputs.MachineMode);
CHASSIS.IN0201.Init(Machine_IO.Inputs.KeySwitchCranking);
CHASSIS.IN0202.Init(Machine_IO.Inputs.SPARE_IN0202);
CHASSIS.IN0203.Init(Machine_IO.Inputs.SPARE_IN0203);
CHASSIS.IN0600.Init(Machine_IO.Inputs.SPARE_IN0600);
CHASSIS.IN0601.Init(Machine_IO.Inputs.SPARE_IN0601);
CHASSIS.IN0602.Init(Machine_IO.Inputs.SPARE_IN0602);
CHASSIS.IN0603.Init(Machine_IO.Inputs.SPARE_IN0603);
CHASSIS.IN0700.Init(Machine_IO.Inputs.SPARE_IN0700);
CHASSIS.IN0701.Init(Machine_IO.Inputs.RADIORHS_JACKLEGRAISE_REQ);
CHASSIS.IN0702.Init(Machine_IO.Inputs.RHS_TROMMELDOORSW);
CHASSIS.IN0703.Init(Machine_IO.Inputs.LHS_TROMMELDOORSW);
CHASSIS.IN0000.Init(Machine_IO.Inputs.HYDOILTEMP_SW);
CHASSIS.IN0001.Init(Machine_IO.Inputs.HYDOILLEVEL_SW);
CHASSIS.IN0002.Init(Machine_IO.Inputs.THERMOSTAT);
CHASSIS.IN0003.Init(Machine_IO.Inputs.RADIORHS_JACKLEGLOWER_REQ);
CHASSIS.IN0500.Init(Machine_IO.Inputs.RADIOLHS_JACKLEGRAISE_REQ);
CHASSIS.IN0501.Init(Machine_IO.Inputs.RADIOLHS_JACKLEGLOWER_REQ);
CHASSIS.IN0502.Init(Machine_IO.Inputs.SideConvRaise_RadialMoveRight);
CHASSIS.IN0503.Init(Machine_IO.Inputs.SideConvLower_RadialMoveLeft);
CHASSIS.IN0400.Init(Machine_IO.Inputs.SPARE_IN0400);
CHASSIS.IN0401.Init(Machine_IO.Inputs.FUELLEVEL_PERCENT);
CHASSIS.IN0900.Init(Machine_IO.Inputs.UMBTRACKREQ);
CHASSIS.IN0901.Init(Machine_IO.Inputs.UMBMACHINESTOP);
CHASSIS.IN0300.Init(Machine_IO.Inputs.RTF_REQ);
CHASSIS.IN0301.Init(Machine_IO.Inputs.RTR_REQ);
CHASSIS.IN0800.Init(Machine_IO.Inputs.LTF_REQ);
CHASSIS.IN0801.Init(Machine_IO.Inputs.LTR_REQ);

// HMI_IO_Init_Input_Links_CODE_GEN_STOP
END_METHOD

METHOD Init_Output_Links
VAR
END_VAR

// HMI_IO_Init_Output_Links_CODE_GEN_START

// generated (UTC): 2024-07-23 18:31:25.327399+00:00
CHASSIS.OUT0000.Init(Machine_IO.Outputs.TAILCONVSPD_MA);
CHASSIS.OUT0001.Init(Machine_IO.Outputs.RHS_JACKLEGLOWER_OP);
CHASSIS.OUT0002.Init(Machine_IO.Outputs.SIDECONVSPD_MA);
CHASSIS.OUT0003.Init(Machine_IO.Outputs.LHS_JACKLEGRAISE_OP);
CHASSIS.OUT0004.Init(Machine_IO.Outputs.SIDETRANSFERSPD_MA);
CHASSIS.OUT0005.Init(Machine_IO.Outputs.LHS_JACKLEGLOWER_OP);
CHASSIS.OUT0006.Init(Machine_IO.Outputs.SETUPDUMPVALVE_OP);
CHASSIS.OUT0007.Init(Machine_IO.Outputs.COLLECTIONCONVSPD_MA);
CHASSIS.OUT0008.Init(Machine_IO.Outputs.COLLECTIONCONVON_OP);
CHASSIS.GROUP0.Init(Machine_IO.Outputs.SUPPLY_GROUP0);
CHASSIS.OUT0100.Init(Machine_IO.Outputs.DRUMSPD_MA_RAMP_LIMIT);
CHASSIS.OUT0101.Init(Machine_IO.Outputs.TRACKINGMODE);
CHASSIS.OUT0102.Init(Machine_IO.Outputs.FEEDERSPD_MA);
CHASSIS.OUT0103.Init(Machine_IO.Outputs.CRANKENABLE);
CHASSIS.OUT0104.Init(Machine_IO.Outputs.DIVERTOILTOTRACK_OP);
CHASSIS.OUT0105.Init(Machine_IO.Outputs.RHS_JACKLEGRAISE_OP);
CHASSIS.OUT0106.Init(Machine_IO.Outputs.TAILCONVON_OP);
CHASSIS.OUT0107.Init(Machine_IO.Outputs.SIDECONVON_OP);
CHASSIS.OUT0108.Init(Machine_IO.Outputs.SIDETRANSFERON_OP);
CHASSIS.GROUP1.Init(Machine_IO.Outputs.SUPPLY_GROUP1);
CHASSIS.OUT0200.Init(Machine_IO.Outputs.LEFTTRACKDIVERT_OP);
CHASSIS.OUT0201.Init(Machine_IO.Outputs.LTF_OP);
CHASSIS.OUT0202.Init(Machine_IO.Outputs.LTR_OP);
CHASSIS.OUT0203.Init(Machine_IO.Outputs.RIGHTTRACKDIVERT_OP);
CHASSIS.OUT0204.Init(Machine_IO.Outputs.RTF_OP);
CHASSIS.OUT0205.Init(Machine_IO.Outputs.RTR_OP);
CHASSIS.OUT0206.Init(Machine_IO.Outputs.DRUMONOFF_OP);
CHASSIS.OUT0207.Init(Machine_IO.Outputs.FEEDERONOFF_OP);
CHASSIS.OUT0208.Init(Machine_IO.Outputs.ECUENABLE);
CHASSIS.GROUP2.Init(Machine_IO.Outputs.SUPPLY_GROUP2);
CHASSIS.OUT3000.Init(Machine_IO.Outputs.SPARE_OUT3000);
CHASSIS.OUT3001.Init(Machine_IO.Outputs.SPARE_OUT3001);

// HMI_IO_Init_Output_Links_CODE_GEN_STOP

AUX.OP0.Init(Machine_IO.Outputs.Siren);
AUX.OP1.Init(Machine_IO.Outputs.AUX_OP1);
AUX.OP2.Init(Machine_IO.Outputs.AUX_OP2);
AUX.OP3.Init(Machine_IO.Outputs.DivertValve);
AUX.OP4.Init(Machine_IO.Outputs.FanFwd_OP);
AUX.OP5.Init(Machine_IO.Outputs.FanRev_OP);
AUX.OP6.Init(Machine_IO.Outputs.SideConvRaise_RadialLeft_OP);
AUX.OP7.Init(Machine_IO.Outputs.SideConvLower_RadialRight_OP);
END_METHOD

METHOD Update_Inputs
VAR	
END_VAR
IF Init_Link_Inputs THEN
	Init_Input_Links();
END_IF
Init_Link_Inputs:=FALSE;

// HMI_IO_Update_Inputs_CODE_GEN_START

// generated (UTC): 2024-07-23 18:31:25.338400+00:00

CHASSIS.IN0100();
CHASSIS.IN0101();
CHASSIS.IN0102();
CHASSIS.IN0103();
CHASSIS.IN0200();
CHASSIS.IN0201();
CHASSIS.IN0202();
CHASSIS.IN0203();
CHASSIS.IN0600();
CHASSIS.IN0601();
CHASSIS.IN0602();
CHASSIS.IN0603();
CHASSIS.IN0700();
CHASSIS.IN0701();
CHASSIS.IN0702();
CHASSIS.IN0703();
CHASSIS.IN0000();
CHASSIS.IN0001();
CHASSIS.IN0002();
CHASSIS.IN0003();
CHASSIS.IN0500();
CHASSIS.IN0501();
CHASSIS.IN0502();
CHASSIS.IN0503();
CHASSIS.IN0400();
CHASSIS.IN0401();
CHASSIS.IN0900();
CHASSIS.IN0901();
CHASSIS.IN0300();
CHASSIS.IN0301();
CHASSIS.IN0800();
CHASSIS.IN0801();
// HMI_IO_Update_Inputs_CODE_GEN_STOP
END_METHOD

END_PROGRAM

// Device/Application/App_PLC/PLC_PRG_MAIN
PROGRAM PLC_PRG_MAIN
VAR
	init: BOOL := TRUE;
	Blink_0: Blink;
	Blink_1: Blink;
	
	fbSetKeyMapping		: ifmDevice.SetKeyMapping;
	fbSetBtnLEDcolour: ifmDevice.SetKeyLED;		
	PreSiren_DUTY: DUTY_CYCLE;
	TEST_SIREN: BOOL;
END_VAR

// TODO
// set up ip address
// tracking interlocks in the PLC
// task for CAN AUX IO and J1939
// Siren power up blip
// Setup dump valves icon feedback to say presiren and on
// T620X - side transfer / side conveyor issues on shutdown?
// feedback of the mA for each function on the main screen
// check the estop button feeback on each screen
// need to check each alarm trhou to the logger after addign the FB's
// link up the warnings in the logger
// mode to bypass engien started for manual testing?
// misc / amin settigns duplication when logged in
// cehck the diagnostics on teh io alarms
// tracking PLC interlocks in the PLC with buttons and estop
// main mimic graphic switching?
// side conveyor graphic not good
// check the auto start stop buttons in the manual mode
// do we need a password to allow the manual mode? - interlock with the setup?

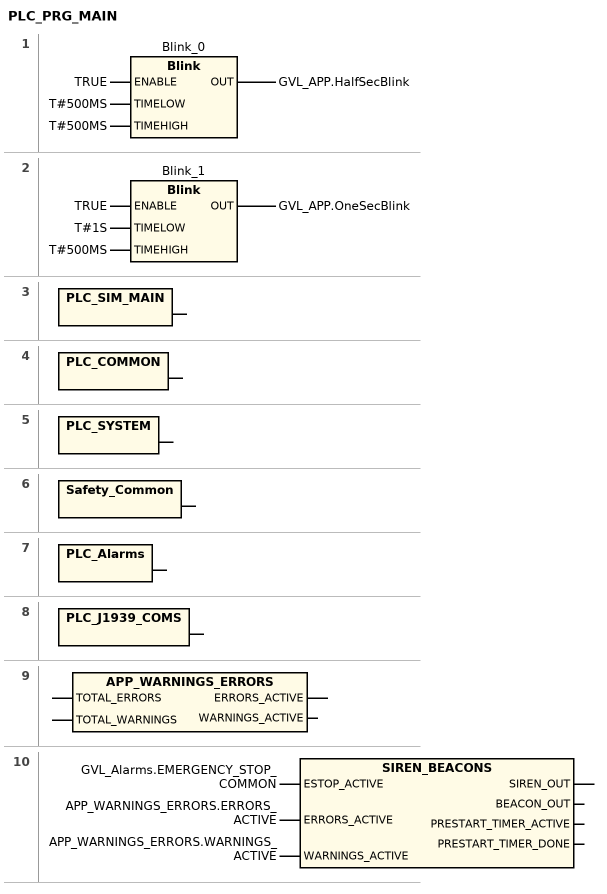
// NETWORK 1
Blink_0(ENABLE := TRUE, TIMELOW := T#500MS, TIMEHIGH := T#500MS); // Blink
GVL_APP.HalfSecBlink := Blink_0.OUT;

// NETWORK 2
Blink_1(ENABLE := TRUE, TIMELOW := T#1S, TIMEHIGH := T#500MS); // Blink
GVL_APP.OneSecBlink := Blink_1.OUT;

// NETWORK 3
PLC_SIM_MAIN();

// NETWORK 4
PLC_COMMON();

// NETWORK 5
PLC_SYSTEM();

// NETWORK 6
Safety_Common();

// NETWORK 7
PLC_Alarms();

// NETWORK 8
PLC_J1939_COMS();

// NETWORK 9
APP_WARNINGS_ERRORS();

